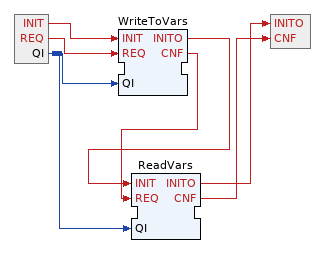
        [picture p71: application OpcUaBothWorking.WorkingWithoutSubscription.folderTestRemote_1]
        SUBAPPLICATION WriteToVars
          EVENT_INPUT
            INIT;
            REQ;
          END_EVENT
          EVENT_OUTPUT
            INITO;
            CNF;
          END_EVENT
          VAR_INPUT
            QI : BOOL;
          END_VAR
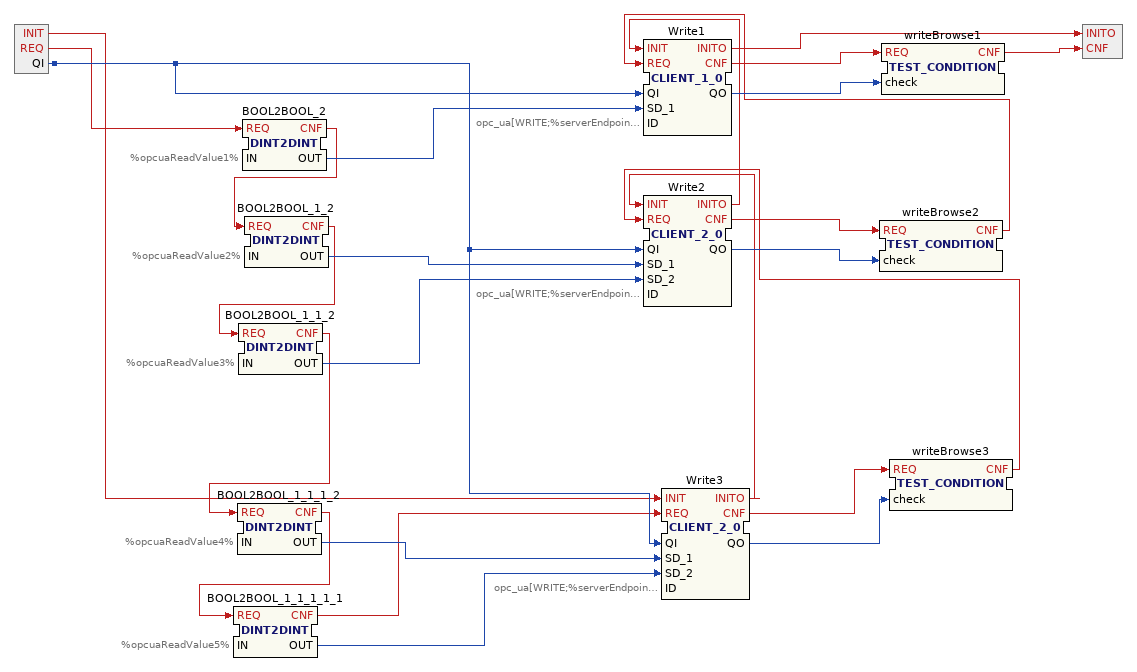
          FBS
            BOOL2BOOL_1_1_2 : DINT2DINT(IN := %opcuaReadValue3%);
            BOOL2BOOL_1_1_1_1_1 : DINT2DINT(IN := %opcuaReadValue5%);
            BOOL2BOOL_1_1_1_2 : DINT2DINT(IN := %opcuaReadValue4%);
            BOOL2BOOL_2 : DINT2DINT(IN := %opcuaReadValue1%);
            BOOL2BOOL_1_2 : DINT2DINT(IN := %opcuaReadValue2%);
            Write1 : CLIENT_1_0(ID := opc_ua[WRITE;%serverEndpoint%;%opcuaFolderTestOnlyBroseName1%]);
            Write3 : CLIENT_2_0(ID := opc_ua[WRITE;%serverEndpoint%;%opcuaFolderTestOnlyBroseName3%]);
            Write2 : CLIENT_2_0(ID := opc_ua[WRITE;%serverEndpoint%;%opcuaFolderTestOnlyBroseName2%]);
            writeBrowse1 : TEST_CONDITION;
            writeBrowse2 : TEST_CONDITION;
            writeBrowse3 : TEST_CONDITION;
          END_FBS
          EVENT_CONNECTIONS
            BOOL2BOOL_1_2.CNF TO BOOL2BOOL_1_1_2.REQ;
            BOOL2BOOL_1_1_2.CNF TO BOOL2BOOL_1_1_1_2.REQ;
            BOOL2BOOL_1_1_1_2.CNF TO BOOL2BOOL_1_1_1_1_1.REQ;
            BOOL2BOOL_2.CNF TO BOOL2BOOL_1_2.REQ;
            REQ TO BOOL2BOOL_2.REQ;
            Write1.INITO TO INITO;
            INIT TO Write3.INIT;
            BOOL2BOOL_1_1_1_1_1.CNF TO Write3.REQ;
            Write3.INITO TO Write2.INIT;
            Write2.INITO TO Write1.INIT;
            writeBrowse3.CNF TO Write2.REQ;
            Write3.CNF TO writeBrowse3.REQ;
            writeBrowse2.CNF TO Write1.REQ;
            Write2.CNF TO writeBrowse2.REQ;
            writeBrowse1.CNF TO CNF;
            Write1.CNF TO writeBrowse1.REQ;
          END_CONNECTIONS
          DATA_CONNECTIONS
            QI TO Write1.QI;
            BOOL2BOOL_2.OUT TO Write1.SD_1;
            QI TO Write3.QI;
            BOOL2BOOL_1_1_1_2.OUT TO Write3.SD_1;
            BOOL2BOOL_1_1_1_1_1.OUT TO Write3.SD_2;
            QI TO Write2.QI;
            BOOL2BOOL_1_2.OUT TO Write2.SD_1;
            BOOL2BOOL_1_1_2.OUT TO Write2.SD_2;
            Write1.QO TO writeBrowse1.check;
            Write2.QO TO writeBrowse2.check;
            Write3.QO TO writeBrowse3.check;
          END_CONNECTIONS
        END_SUBAPPLICATION
        SUBAPPLICATION ReadVars
          EVENT_INPUT
            INIT;
            REQ;
          END_EVENT
          EVENT_OUTPUT
            INITO;
            CNF;
          END_EVENT
          VAR_INPUT
            QI : BOOL;
          END_VAR
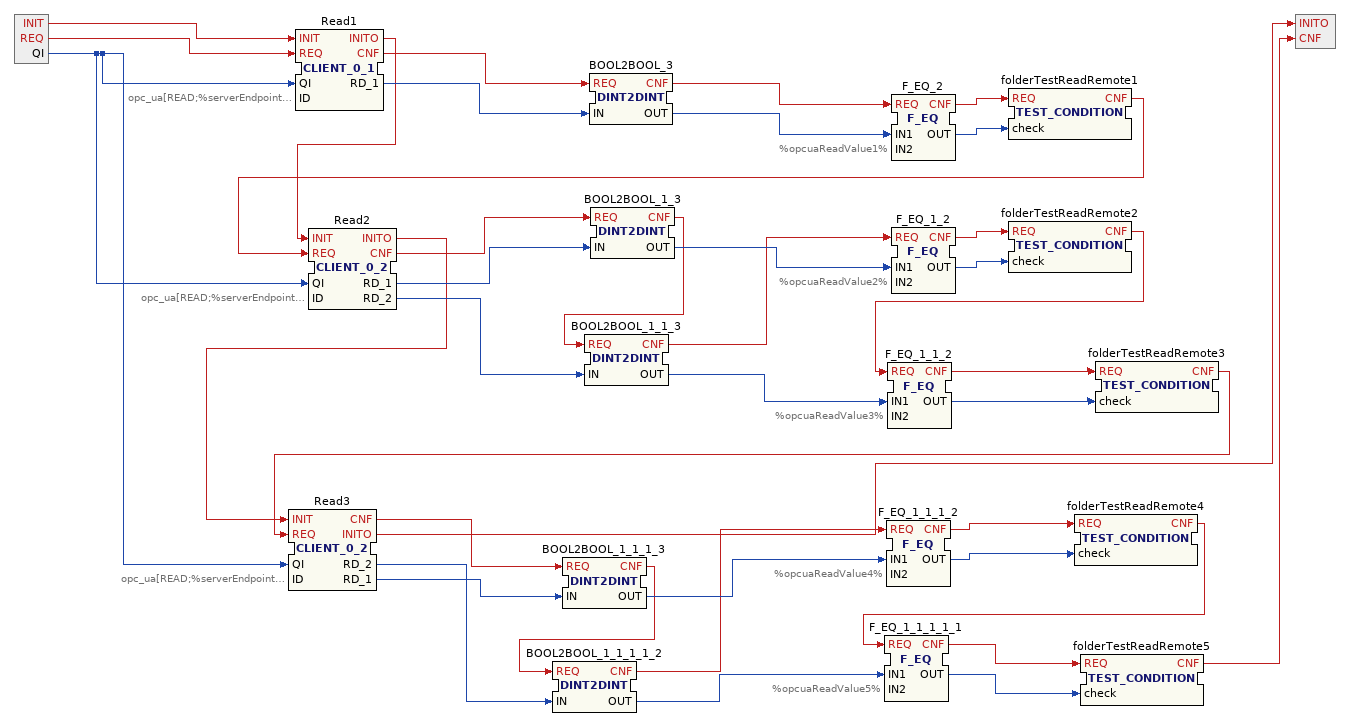
          FBS
            Read1 : CLIENT_0_1(ID := opc_ua[READ;%serverEndpoint%;%opcuaFolderTestOnlyBroseName1%]);
            Read2 : CLIENT_0_2(ID := opc_ua[READ;%serverEndpoint%;%opcuaFolderTestOnlyBroseName2%]);
            F_EQ_1_1_1_2 : F_EQ(IN2 := %opcuaReadValue4%);
            folderTestReadRemote4 : TEST_CONDITION;
            BOOL2BOOL_1_3 : DINT2DINT;
            F_EQ_1_1_1_1_1 : F_EQ(IN2 := %opcuaReadValue5%);
            folderTestReadRemote3 : TEST_CONDITION;
            BOOL2BOOL_1_1_3 : DINT2DINT;
            BOOL2BOOL_1_1_1_1_2 : DINT2DINT;
            BOOL2BOOL_1_1_1_3 : DINT2DINT;
            folderTestReadRemote2 : TEST_CONDITION;
            F_EQ_1_1_2 : F_EQ(IN2 := %opcuaReadValue3%);
            F_EQ_2 : F_EQ(IN2 := %opcuaReadValue1%);
            F_EQ_1_2 : F_EQ(IN2 := %opcuaReadValue2%);
            Read3 : CLIENT_0_2(ID := opc_ua[READ;%serverEndpoint%;%opcuaFolderTestOnlyBroseName3%]);
            folderTestReadRemote5 : TEST_CONDITION;
            folderTestReadRemote1 : TEST_CONDITION;
            BOOL2BOOL_3 : DINT2DINT;
          END_FBS
          EVENT_CONNECTIONS
            Read1.INITO TO Read2.INIT;
            Read1.CNF TO BOOL2BOOL_3.REQ;
            folderTestReadRemote1.CNF TO Read2.REQ;
            Read2.INITO TO Read3.INIT;
            Read2.CNF TO BOOL2BOOL_1_3.REQ;
            BOOL2BOOL_1_1_1_1_2.CNF TO F_EQ_1_1_1_2.REQ;
            F_EQ_1_1_1_2.CNF TO folderTestReadRemote4.REQ;
            folderTestReadRemote4.CNF TO F_EQ_1_1_1_1_1.REQ;
            BOOL2BOOL_1_3.CNF TO BOOL2BOOL_1_1_3.REQ;
            F_EQ_1_1_1_1_1.CNF TO folderTestReadRemote5.REQ;
            F_EQ_1_1_2.CNF TO folderTestReadRemote3.REQ;
            folderTestReadRemote3.CNF TO Read3.REQ;
            BOOL2BOOL_1_1_3.CNF TO F_EQ_1_2.REQ;
            BOOL2BOOL_1_1_1_3.CNF TO BOOL2BOOL_1_1_1_1_2.REQ;
            Read3.CNF TO BOOL2BOOL_1_1_1_3.REQ;
            F_EQ_1_2.CNF TO folderTestReadRemote2.REQ;
            folderTestReadRemote2.CNF TO F_EQ_1_1_2.REQ;
            BOOL2BOOL_3.CNF TO F_EQ_2.REQ;
            F_EQ_2.CNF TO folderTestReadRemote1.REQ;
            INIT TO Read1.INIT;
            REQ TO Read1.REQ;
            Read3.INITO TO INITO;
            folderTestReadRemote5.CNF TO CNF;
          END_CONNECTIONS
          DATA_CONNECTIONS
            Read1.RD_1 TO BOOL2BOOL_3.IN;
            Read2.RD_1 TO BOOL2BOOL_1_3.IN;
            Read2.RD_2 TO BOOL2BOOL_1_1_3.IN;
            BOOL2BOOL_1_1_1_3.OUT TO F_EQ_1_1_1_2.IN1;
            F_EQ_1_1_1_2.OUT TO folderTestReadRemote4.check;
            BOOL2BOOL_1_3.OUT TO F_EQ_1_2.IN1;
            BOOL2BOOL_1_1_1_1_2.OUT TO F_EQ_1_1_1_1_1.IN1;
            F_EQ_1_1_1_1_1.OUT TO folderTestReadRemote5.check;
            F_EQ_1_1_2.OUT TO folderTestReadRemote3.check;
            BOOL2BOOL_1_1_3.OUT TO F_EQ_1_1_2.IN1;
            Read3.RD_2 TO BOOL2BOOL_1_1_1_1_2.IN;
            Read3.RD_1 TO BOOL2BOOL_1_1_1_3.IN;
            F_EQ_1_2.OUT TO folderTestReadRemote2.check;
            BOOL2BOOL_3.OUT TO F_EQ_2.IN1;
            F_EQ_2.OUT TO folderTestReadRemote1.check;
            QI TO Read1.QI;
            QI TO Read2.QI;
            QI TO Read3.QI;
          END_CONNECTIONS
        END_SUBAPPLICATION
        EVENT_CONNECTIONS
          WriteToVars.INITO TO ReadVars.INIT;
          INIT TO WriteToVars.INIT;
          REQ TO WriteToVars.REQ;
          ReadVars.CNF TO CNF;
          WriteToVars.CNF TO ReadVars.REQ;
          ReadVars.INITO TO INITO;
        END_CONNECTIONS
        DATA_CONNECTIONS
          QI TO ReadVars.QI;
          QI TO WriteToVars.QI;
        END_CONNECTIONS
      END_SUBAPPLICATION
      SUBAPPLICATION bytestringNodeIdTestRemote_1
        EVENT_INPUT
          INIT;
          REQ;
        END_EVENT
        EVENT_OUTPUT
          INITO;
          CNF;
        END_EVENT
        VAR_INPUT
          QI : BOOL;
        END_VAR
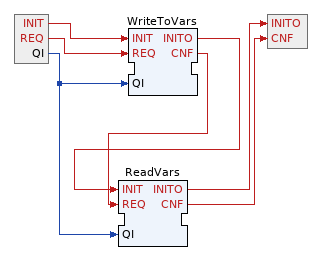
        SUBAPPLICATION WriteToVars
          EVENT_INPUT
            INIT;
            REQ;
          END_EVENT
          EVENT_OUTPUT
            INITO;
            CNF;
          END_EVENT
          VAR_INPUT
            QI : BOOL;
          END_VAR
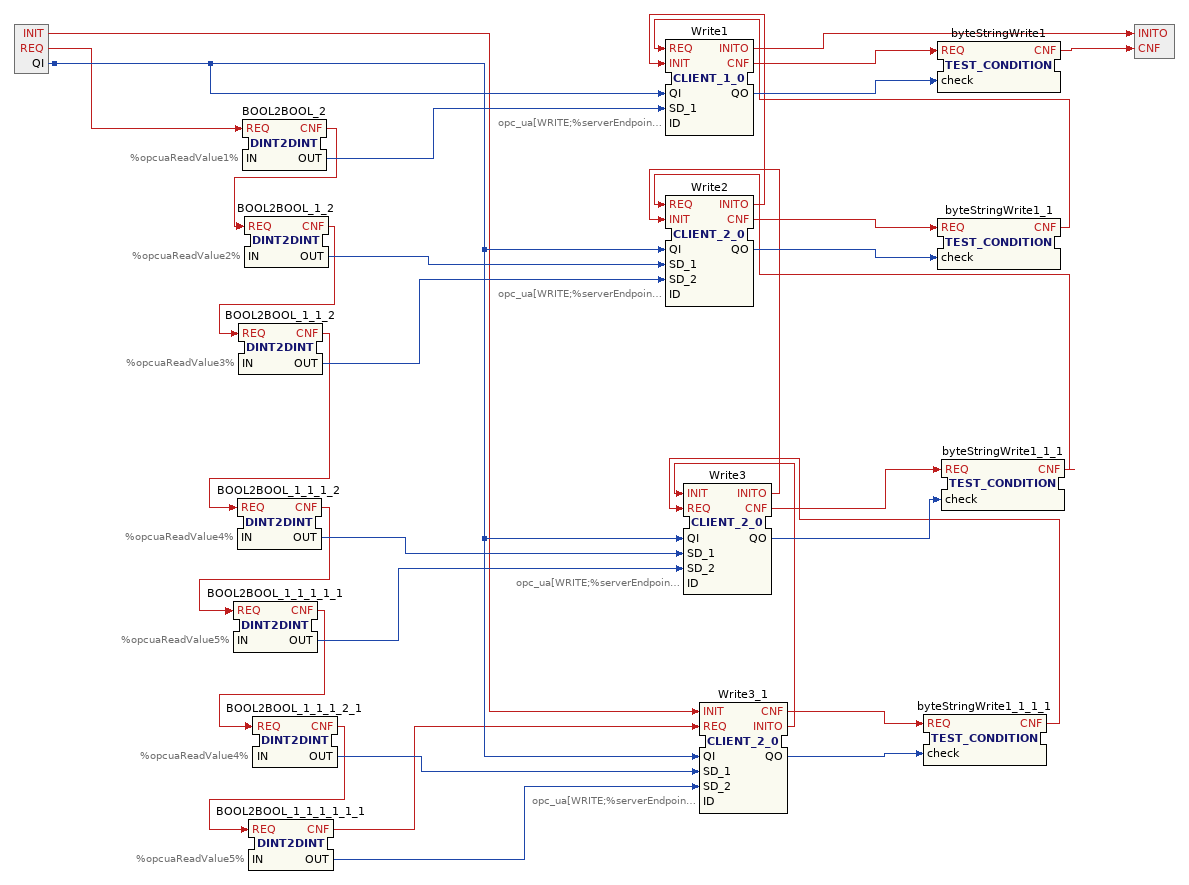
          FBS
            BOOL2BOOL_1_1_2 : DINT2DINT(IN := %opcuaReadValue3%);
            BOOL2BOOL_1_1_1_1_1 : DINT2DINT(IN := %opcuaReadValue5%);
            BOOL2BOOL_1_1_1_2 : DINT2DINT(IN := %opcuaReadValue4%);
            BOOL2BOOL_2 : DINT2DINT(IN := %opcuaReadValue1%);
            BOOL2BOOL_1_2 : DINT2DINT(IN := %opcuaReadValue2%);
            BOOL2BOOL_1_1_1_1_1_1 : DINT2DINT(IN := %opcuaReadValue5%);
            BOOL2BOOL_1_1_1_2_1 : DINT2DINT(IN := %opcuaReadValue4%);
            byteStringWrite1 : TEST_CONDITION;
            byteStringWrite1_1 : TEST_CONDITION;
            byteStringWrite1_1_1 : TEST_CONDITION;
            byteStringWrite1_1_1_1 : TEST_CONDITION;
            Write1 : CLIENT_1_0(ID := opc_ua[WRITE;%serverEndpoint%;%opcuaFolderTestWithNodeIdByteString1%]);
            Write2 : CLIENT_2_0(ID := opc_ua[WRITE;%serverEndpoint%;%opcuaFolderTestWithNodeIdByteString2%]);
            Write3_1 : CLIENT_2_0(ID := opc_ua[WRITE;%serverEndpoint%;,1:b=byteStringNodeId3;,1:b=byteStringNodeId4]);
            Write3 : CLIENT_2_0(ID := opc_ua[WRITE;%serverEndpoint%;%opcuaFolderTestWithNodeIdByteString3%]);
          END_FBS
          EVENT_CONNECTIONS
            BOOL2BOOL_1_2.CNF TO BOOL2BOOL_1_1_2.REQ;
            BOOL2BOOL_1_1_2.CNF TO BOOL2BOOL_1_1_1_2.REQ;
            BOOL2BOOL_1_1_1_2.CNF TO BOOL2BOOL_1_1_1_1_1.REQ;
            BOOL2BOOL_2.CNF TO BOOL2BOOL_1_2.REQ;
            REQ TO BOOL2BOOL_2.REQ;
            BOOL2BOOL_1_1_1_2_1.CNF TO BOOL2BOOL_1_1_1_1_1_1.REQ;
            BOOL2BOOL_1_1_1_1_1.CNF TO BOOL2BOOL_1_1_1_2_1.REQ;
            byteStringWrite1.CNF TO CNF;
            byteStringWrite1_1.CNF TO Write1.REQ;
            Write1.INITO TO INITO;
            Write1.CNF TO byteStringWrite1.REQ;
            byteStringWrite1_1_1.CNF TO Write2.REQ;
            Write2.INITO TO Write1.INIT;
            Write2.CNF TO byteStringWrite1_1.REQ;
            INIT TO Write3_1.INIT;
            BOOL2BOOL_1_1_1_1_1_1.CNF TO Write3_1.REQ;
            Write3_1.CNF TO byteStringWrite1_1_1_1.REQ;
            Write3_1.INITO TO Write3.INIT;
            byteStringWrite1_1_1_1.CNF TO Write3.REQ;
            Write3.INITO TO Write2.INIT;
            Write3.CNF TO byteStringWrite1_1_1.REQ;
          END_CONNECTIONS
          DATA_CONNECTIONS
            QI TO Write1.QI;
            BOOL2BOOL_2.OUT TO Write1.SD_1;
            Write1.QO TO byteStringWrite1.check;
            QI TO Write2.QI;
            BOOL2BOOL_1_2.OUT TO Write2.SD_1;
            BOOL2BOOL_1_1_2.OUT TO Write2.SD_2;
            Write2.QO TO byteStringWrite1_1.check;
            QI TO Write3_1.QI;
            BOOL2BOOL_1_1_1_2_1.OUT TO Write3_1.SD_1;
            BOOL2BOOL_1_1_1_1_1_1.OUT TO Write3_1.SD_2;
            Write3_1.QO TO byteStringWrite1_1_1_1.check;
            QI TO Write3.QI;
            BOOL2BOOL_1_1_1_2.OUT TO Write3.SD_1;
            BOOL2BOOL_1_1_1_1_1.OUT TO Write3.SD_2;
            Write3.QO TO byteStringWrite1_1_1.check;
          END_CONNECTIONS
        END_SUBAPPLICATION
        SUBAPPLICATION ReadVars
          EVENT_INPUT
            INIT;
            REQ;
          END_EVENT
          EVENT_OUTPUT
            INITO;
            CNF;
          END_EVENT
          VAR_INPUT
            QI : BOOL;
          END_VAR
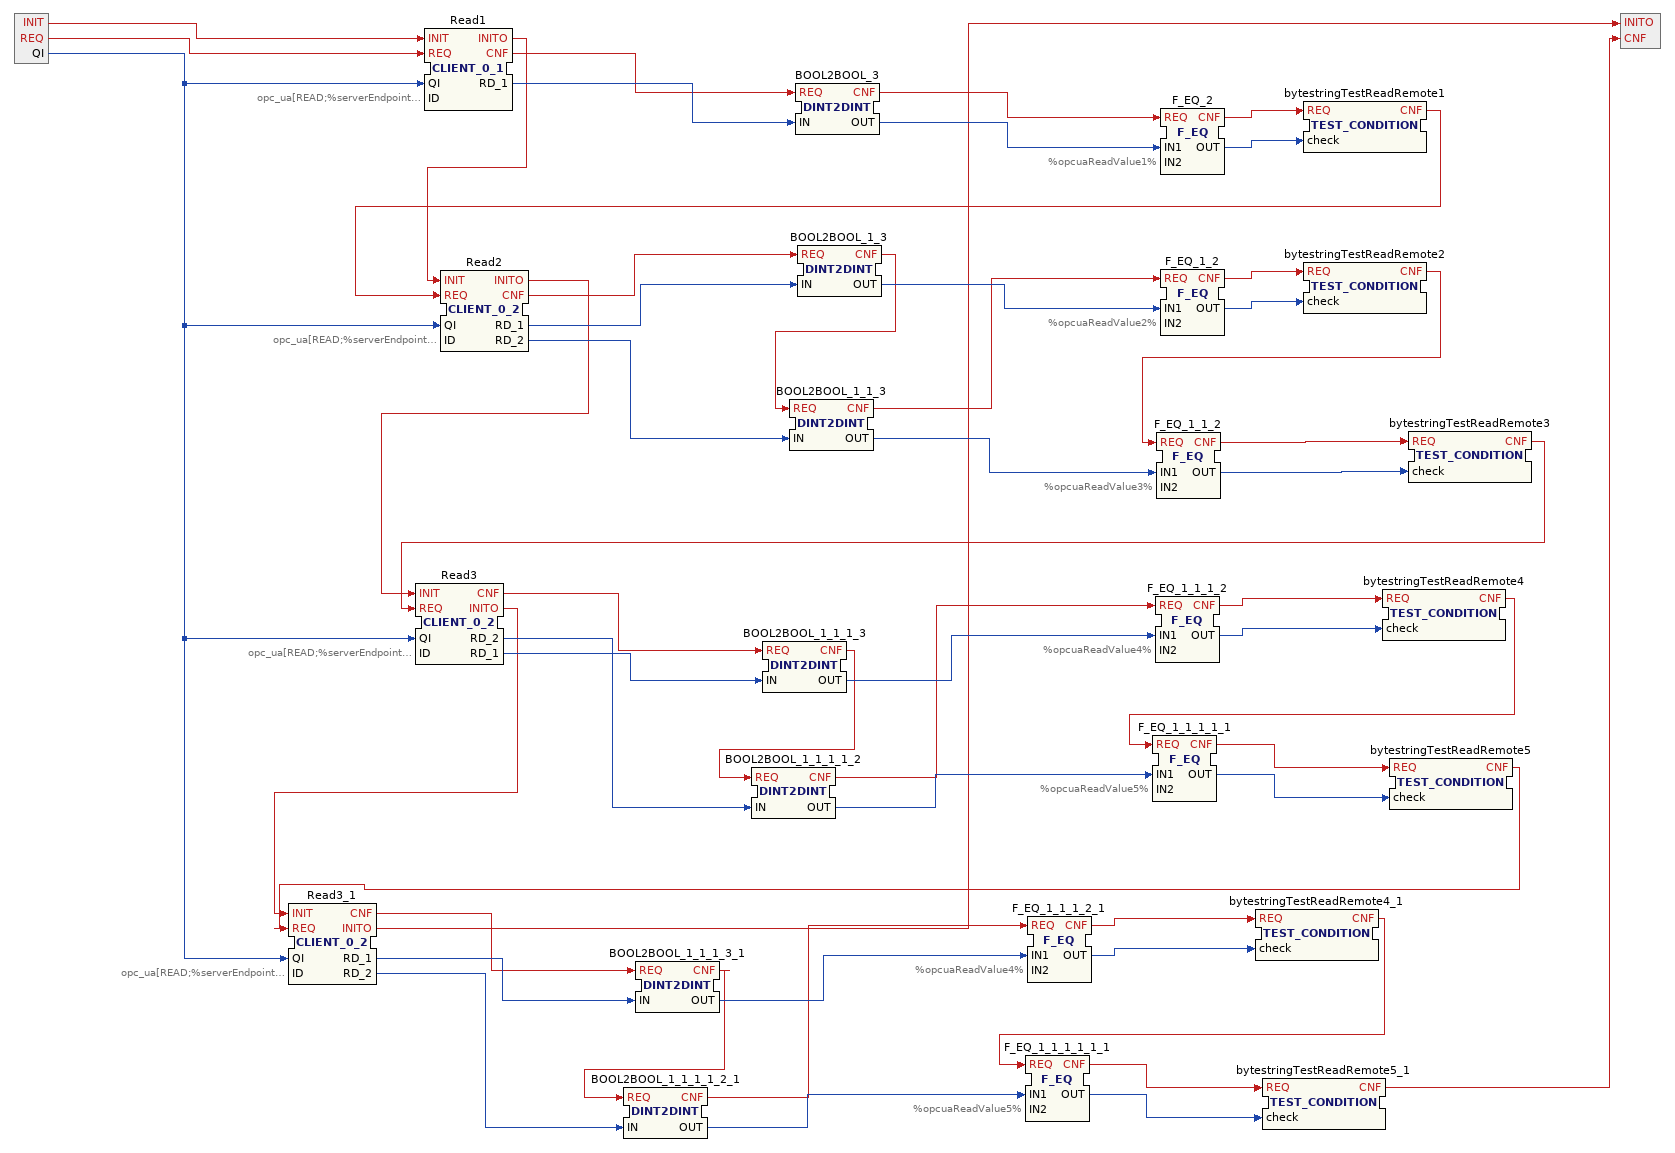
          FBS
            Read1 : CLIENT_0_1(ID := opc_ua[READ;%serverEndpoint%;%opcuaFolderTestWithNodeIdByteString1%]);
            Read2 : CLIENT_0_2(ID := opc_ua[READ;%serverEndpoint%;%opcuaFolderTestWithNodeIdByteString2%]);
            F_EQ_1_1_1_2 : F_EQ(IN2 := %opcuaReadValue4%);
            bytestringTestReadRemote4 : TEST_CONDITION;
            BOOL2BOOL_1_3 : DINT2DINT;
            F_EQ_1_1_1_1_1 : F_EQ(IN2 := %opcuaReadValue5%);
            bytestringTestReadRemote3 : TEST_CONDITION;
            BOOL2BOOL_1_1_3 : DINT2DINT;
            BOOL2BOOL_1_1_1_1_2 : DINT2DINT;
            BOOL2BOOL_1_1_1_3 : DINT2DINT;
            bytestringTestReadRemote2 : TEST_CONDITION;
            F_EQ_1_1_2 : F_EQ(IN2 := %opcuaReadValue3%);
            F_EQ_2 : F_EQ(IN2 := %opcuaReadValue1%);
            F_EQ_1_2 : F_EQ(IN2 := %opcuaReadValue2%);
            Read3 : CLIENT_0_2(ID := opc_ua[READ;%serverEndpoint%;%opcuaFolderTestWithNodeIdByteString3%]);
            bytestringTestReadRemote5 : TEST_CONDITION;
            bytestringTestReadRemote1 : TEST_CONDITION;
            BOOL2BOOL_3 : DINT2DINT;
            BOOL2BOOL_1_1_1_3_1 : DINT2DINT;
            Read3_1 : CLIENT_0_2(ID := opc_ua[READ;%serverEndpoint%;,1:b=byteStringNodeId3;,1:b=byteStringNodeId4]);
            bytestringTestReadRemote4_1 : TEST_CONDITION;
            F_EQ_1_1_1_2_1 : F_EQ(IN2 := %opcuaReadValue4%);
            BOOL2BOOL_1_1_1_1_2_1 : DINT2DINT;
            bytestringTestReadRemote5_1 : TEST_CONDITION;
            F_EQ_1_1_1_1_1_1 : F_EQ(IN2 := %opcuaReadValue5%);
          END_FBS
          EVENT_CONNECTIONS
            Read1.INITO TO Read2.INIT;
            Read1.CNF TO BOOL2BOOL_3.REQ;
            bytestringTestReadRemote1.CNF TO Read2.REQ;
            Read2.INITO TO Read3.INIT;
            Read2.CNF TO BOOL2BOOL_1_3.REQ;
            BOOL2BOOL_1_1_1_1_2.CNF TO F_EQ_1_1_1_2.REQ;
            F_EQ_1_1_1_2.CNF TO bytestringTestReadRemote4.REQ;
            bytestringTestReadRemote4.CNF TO F_EQ_1_1_1_1_1.REQ;
            BOOL2BOOL_1_3.CNF TO BOOL2BOOL_1_1_3.REQ;
            F_EQ_1_1_1_1_1.CNF TO bytestringTestReadRemote5.REQ;
            F_EQ_1_1_2.CNF TO bytestringTestReadRemote3.REQ;
            bytestringTestReadRemote3.CNF TO Read3.REQ;
            BOOL2BOOL_1_1_3.CNF TO F_EQ_1_2.REQ;
            BOOL2BOOL_1_1_1_3.CNF TO BOOL2BOOL_1_1_1_1_2.REQ;
            Read3.CNF TO BOOL2BOOL_1_1_1_3.REQ;
            F_EQ_1_2.CNF TO bytestringTestReadRemote2.REQ;
            bytestringTestReadRemote2.CNF TO F_EQ_1_1_2.REQ;
            BOOL2BOOL_3.CNF TO F_EQ_2.REQ;
            F_EQ_2.CNF TO bytestringTestReadRemote1.REQ;
            INIT TO Read1.INIT;
            REQ TO Read1.REQ;
            bytestringTestReadRemote4_1.CNF TO F_EQ_1_1_1_1_1_1.REQ;
            BOOL2BOOL_1_1_1_1_2_1.CNF TO F_EQ_1_1_1_2_1.REQ;
            F_EQ_1_1_1_1_1_1.CNF TO bytestringTestReadRemote5_1.REQ;
            F_EQ_1_1_1_2_1.CNF TO bytestringTestReadRemote4_1.REQ;
            BOOL2BOOL_1_1_1_3_1.CNF TO BOOL2BOOL_1_1_1_1_2_1.REQ;
            Read3_1.CNF TO BOOL2BOOL_1_1_1_3_1.REQ;
            Read3_1.INITO TO INITO;
            Read3.INITO TO Read3_1.INIT;
            bytestringTestReadRemote5_1.CNF TO CNF;
            bytestringTestReadRemote5.CNF TO Read3_1.REQ;
          END_CONNECTIONS
          DATA_CONNECTIONS
            Read1.RD_1 TO BOOL2BOOL_3.IN;
            Read2.RD_1 TO BOOL2BOOL_1_3.IN;
            Read2.RD_2 TO BOOL2BOOL_1_1_3.IN;
            BOOL2BOOL_1_1_1_3.OUT TO F_EQ_1_1_1_2.IN1;
            F_EQ_1_1_1_2.OUT TO bytestringTestReadRemote4.check;
            BOOL2BOOL_1_3.OUT TO F_EQ_1_2.IN1;
            BOOL2BOOL_1_1_1_1_2.OUT TO F_EQ_1_1_1_1_1.IN1;
            F_EQ_1_1_1_1_1.OUT TO bytestringTestReadRemote5.check;
            F_EQ_1_1_2.OUT TO bytestringTestReadRemote3.check;
            BOOL2BOOL_1_1_3.OUT TO F_EQ_1_1_2.IN1;
            Read3.RD_2 TO BOOL2BOOL_1_1_1_1_2.IN;
            Read3.RD_1 TO BOOL2BOOL_1_1_1_3.IN;
            F_EQ_1_2.OUT TO bytestringTestReadRemote2.check;
            BOOL2BOOL_3.OUT TO F_EQ_2.IN1;
            F_EQ_2.OUT TO bytestringTestReadRemote1.check;
            QI TO Read1.QI;
            QI TO Read2.QI;
            QI TO Read3.QI;
            BOOL2BOOL_1_1_1_1_2_1.OUT TO F_EQ_1_1_1_1_1_1.IN1;
            BOOL2BOOL_1_1_1_3_1.OUT TO F_EQ_1_1_1_2_1.IN1;
            F_EQ_1_1_1_2_1.OUT TO bytestringTestReadRemote4_1.check;
            Read3_1.RD_1 TO BOOL2BOOL_1_1_1_3_1.IN;
            F_EQ_1_1_1_1_1_1.OUT TO bytestringTestReadRemote5_1.check;
            Read3_1.RD_2 TO BOOL2BOOL_1_1_1_1_2_1.IN;
            QI TO Read3_1.QI;
          END_CONNECTIONS
        END_SUBAPPLICATION
        EVENT_CONNECTIONS
          WriteToVars.INITO TO ReadVars.INIT;
          INIT TO WriteToVars.INIT;
          REQ TO WriteToVars.REQ;
          ReadVars.CNF TO CNF;
          WriteToVars.CNF TO ReadVars.REQ;
          ReadVars.INITO TO INITO;
        END_CONNECTIONS
        DATA_CONNECTIONS
          QI TO ReadVars.QI;
          QI TO WriteToVars.QI;
        END_CONNECTIONS
      END_SUBAPPLICATION
      SUBAPPLICATION RemoteMethods_1
        EVENT_INPUT
          INIT;
          REQ;
        END_EVENT
        EVENT_OUTPUT
          INITO;
          CNF;
        END_EVENT
        VAR_INPUT
          QI : BOOL;
        END_VAR
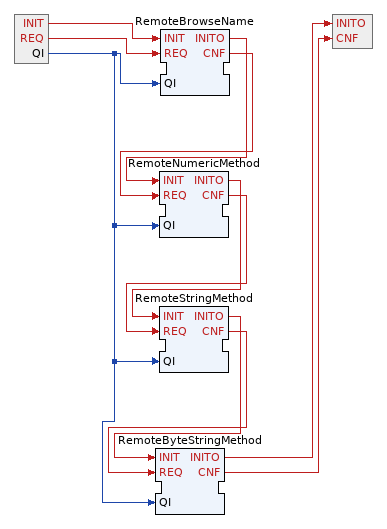
        SUBAPPLICATION RemoteBrowseName
          EVENT_INPUT
            INIT;
            REQ;
          END_EVENT
          EVENT_OUTPUT
            INITO;
            CNF;
          END_EVENT
          VAR_INPUT
            QI : BOOL;
          END_VAR
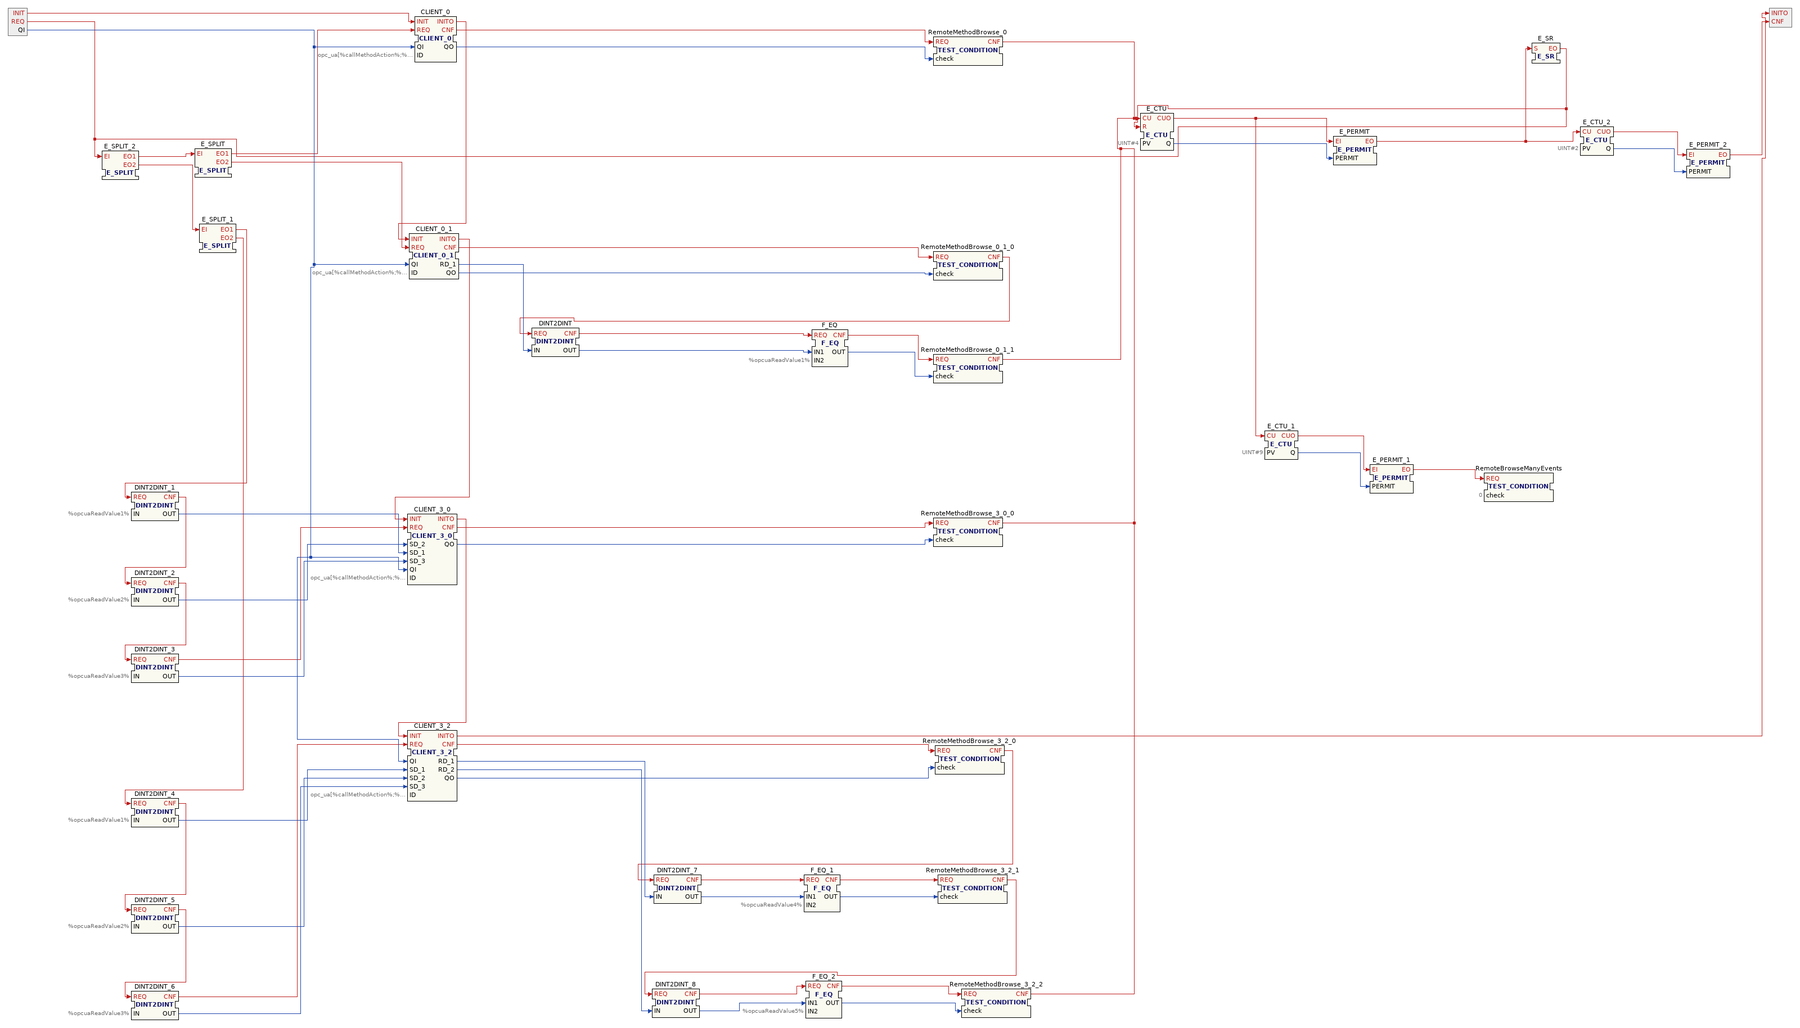
          FBS
            DINT2DINT_4 : DINT2DINT(IN := %opcuaReadValue1%);
            CLIENT_0 : CLIENT_0(ID := opc_ua[%callMethodAction%;%serverEndpoint%;%opcuaMethodCreation1%]);
            DINT2DINT_2 : DINT2DINT(IN := %opcuaReadValue2%);
            CLIENT_0_1 : CLIENT_0_1(ID := opc_ua[%callMethodAction%;%serverEndpoint%;%opcuaMethodCreation2%]);
            DINT2DINT : DINT2DINT;
            DINT2DINT_1 : DINT2DINT(IN := %opcuaReadValue1%);
            CLIENT_3_0 : CLIENT_3_0(ID := opc_ua[%callMethodAction%;%serverEndpoint%;%opcuaMethodCreation3%]);
            CLIENT_3_2 : CLIENT_3_2(ID := opc_ua[%callMethodAction%;%serverEndpoint%;%opcuaMethodCreation4%]);
            DINT2DINT_3 : DINT2DINT(IN := %opcuaReadValue3%);
            DINT2DINT_5 : DINT2DINT(IN := %opcuaReadValue2%);
            DINT2DINT_6 : DINT2DINT(IN := %opcuaReadValue3%);
            DINT2DINT_7 : DINT2DINT;
            DINT2DINT_8 : DINT2DINT;
            RemoteMethodBrowse_3_2_1 : TEST_CONDITION;
            RemoteMethodBrowse_3_2_2 : TEST_CONDITION;
            RemoteMethodBrowse_0 : TEST_CONDITION;
            RemoteMethodBrowse_0_1_0 : TEST_CONDITION;
            RemoteMethodBrowse_0_1_1 : TEST_CONDITION;
            RemoteMethodBrowse_3_2_0 : TEST_CONDITION;
            RemoteMethodBrowse_3_0_0 : TEST_CONDITION;
            F_EQ : F_EQ(IN2 := %opcuaReadValue1%);
            F_EQ_1 : F_EQ(IN2 := %opcuaReadValue4%);
            F_EQ_2 : F_EQ(IN2 := %opcuaReadValue5%);
            E_SPLIT : E_SPLIT;
            E_SPLIT_1 : E_SPLIT;
            E_CTU : E_CTU(PV := UINT#4);
            E_PERMIT : E_PERMIT;
            E_CTU_1 : E_CTU(PV := UINT#9);
            E_PERMIT_1 : E_PERMIT;
            RemoteBrowseManyEvents : TEST_CONDITION(check := 0);
            E_SPLIT_2 : E_SPLIT;
            E_PERMIT_2 : E_PERMIT;
            E_CTU_2 : E_CTU(PV := UINT#2);
            E_SR : E_SR;
          END_FBS
          EVENT_CONNECTIONS
            DINT2DINT_1.CNF TO DINT2DINT_2.REQ;
            DINT2DINT_2.CNF TO DINT2DINT_3.REQ;
            CLIENT_0_1.INITO TO CLIENT_3_0.INIT;
            INIT TO CLIENT_0.INIT;
            CLIENT_0.INITO TO CLIENT_0_1.INIT;
            CLIENT_3_0.INITO TO CLIENT_3_2.INIT;
            CLIENT_3_2.INITO TO INITO;
            CLIENT_0.CNF TO RemoteMethodBrowse_0.REQ;
            F_EQ.CNF TO RemoteMethodBrowse_0_1_1.REQ;
            CLIENT_3_0.CNF TO RemoteMethodBrowse_3_0_0.REQ;
            DINT2DINT_8.CNF TO F_EQ_2.REQ;
            DINT2DINT_7.CNF TO F_EQ_1.REQ;
            RemoteMethodBrowse_3_2_0.CNF TO DINT2DINT_7.REQ;
            F_EQ_1.CNF TO RemoteMethodBrowse_3_2_1.REQ;
            RemoteMethodBrowse_3_2_1.CNF TO DINT2DINT_8.REQ;
            F_EQ_2.CNF TO RemoteMethodBrowse_3_2_2.REQ;
            CLIENT_3_2.CNF TO RemoteMethodBrowse_3_2_0.REQ;
            DINT2DINT_4.CNF TO DINT2DINT_5.REQ;
            DINT2DINT_5.CNF TO DINT2DINT_6.REQ;
            DINT2DINT_6.CNF TO CLIENT_3_2.REQ;
            CLIENT_0_1.CNF TO RemoteMethodBrowse_0_1_0.REQ;
            RemoteMethodBrowse_0_1_0.CNF TO DINT2DINT.REQ;
            DINT2DINT.CNF TO F_EQ.REQ;
            DINT2DINT_3.CNF TO CLIENT_3_0.REQ;
            E_SPLIT.EO1 TO CLIENT_0.REQ;
            RemoteMethodBrowse_3_2_2.CNF TO E_CTU.CU;
            E_CTU.CUO TO E_CTU_1.CU;
            E_CTU.CUO TO E_PERMIT.EI;
            E_CTU_1.CUO TO E_PERMIT_1.EI;
            E_PERMIT_1.EO TO RemoteBrowseManyEvents.REQ;
            RemoteMethodBrowse_0.CNF TO E_CTU.CU;
            E_SPLIT.EO2 TO CLIENT_0_1.REQ;
            RemoteMethodBrowse_0_1_1.CNF TO E_CTU.CU;
            E_SPLIT_1.EO1 TO DINT2DINT_1.REQ;
            RemoteMethodBrowse_3_0_0.CNF TO E_CTU.CU;
            E_SPLIT_1.EO2 TO DINT2DINT_4.REQ;
            REQ TO E_SPLIT_2.EI;
            E_SPLIT_2.EO1 TO E_SPLIT.EI;
            E_SPLIT_2.EO2 TO E_SPLIT_1.EI;
            E_PERMIT.EO TO E_CTU_2.CU;
            E_CTU_2.CUO TO E_PERMIT_2.EI;
            E_PERMIT_2.EO TO CNF;
            E_PERMIT.EO TO E_SR.S;
            E_SR.EO TO E_CTU.R;
            E_SR.EO TO E_SPLIT_2.EI;
          END_CONNECTIONS
          DATA_CONNECTIONS
            DINT2DINT_2.OUT TO CLIENT_3_0.SD_2;
            CLIENT_0_1.RD_1 TO DINT2DINT.IN;
            DINT2DINT_1.OUT TO CLIENT_3_0.SD_1;
            DINT2DINT_3.OUT TO CLIENT_3_0.SD_3;
            QI TO CLIENT_0_1.QI;
            QI TO CLIENT_3_0.QI;
            QI TO CLIENT_3_2.QI;
            QI TO CLIENT_0.QI;
            DINT2DINT_4.OUT TO CLIENT_3_2.SD_1;
            DINT2DINT_5.OUT TO CLIENT_3_2.SD_2;
            CLIENT_3_2.RD_1 TO DINT2DINT_7.IN;
            CLIENT_3_2.RD_2 TO DINT2DINT_8.IN;
            DINT2DINT_6.OUT TO CLIENT_3_2.SD_3;
            CLIENT_0.QO TO RemoteMethodBrowse_0.check;
            CLIENT_0_1.QO TO RemoteMethodBrowse_0_1_0.check;
            F_EQ.OUT TO RemoteMethodBrowse_0_1_1.check;
            DINT2DINT.OUT TO F_EQ.IN1;
            CLIENT_3_0.QO TO RemoteMethodBrowse_3_0_0.check;
            DINT2DINT_7.OUT TO F_EQ_1.IN1;
            DINT2DINT_8.OUT TO F_EQ_2.IN1;
            F_EQ_1.OUT TO RemoteMethodBrowse_3_2_1.check;
            F_EQ_2.OUT TO RemoteMethodBrowse_3_2_2.check;
            CLIENT_3_2.QO TO RemoteMethodBrowse_3_2_0.check;
            E_CTU.Q TO E_PERMIT.PERMIT;
            E_CTU_1.Q TO E_PERMIT_1.PERMIT;
            E_CTU_2.Q TO E_PERMIT_2.PERMIT;
          END_CONNECTIONS
        END_SUBAPPLICATION
        SUBAPPLICATION RemoteNumericMethod
          EVENT_INPUT
            INIT;
            REQ;
          END_EVENT
          EVENT_OUTPUT
            INITO;
            CNF;
          END_EVENT
          VAR_INPUT
            QI : BOOL;
          END_VAR
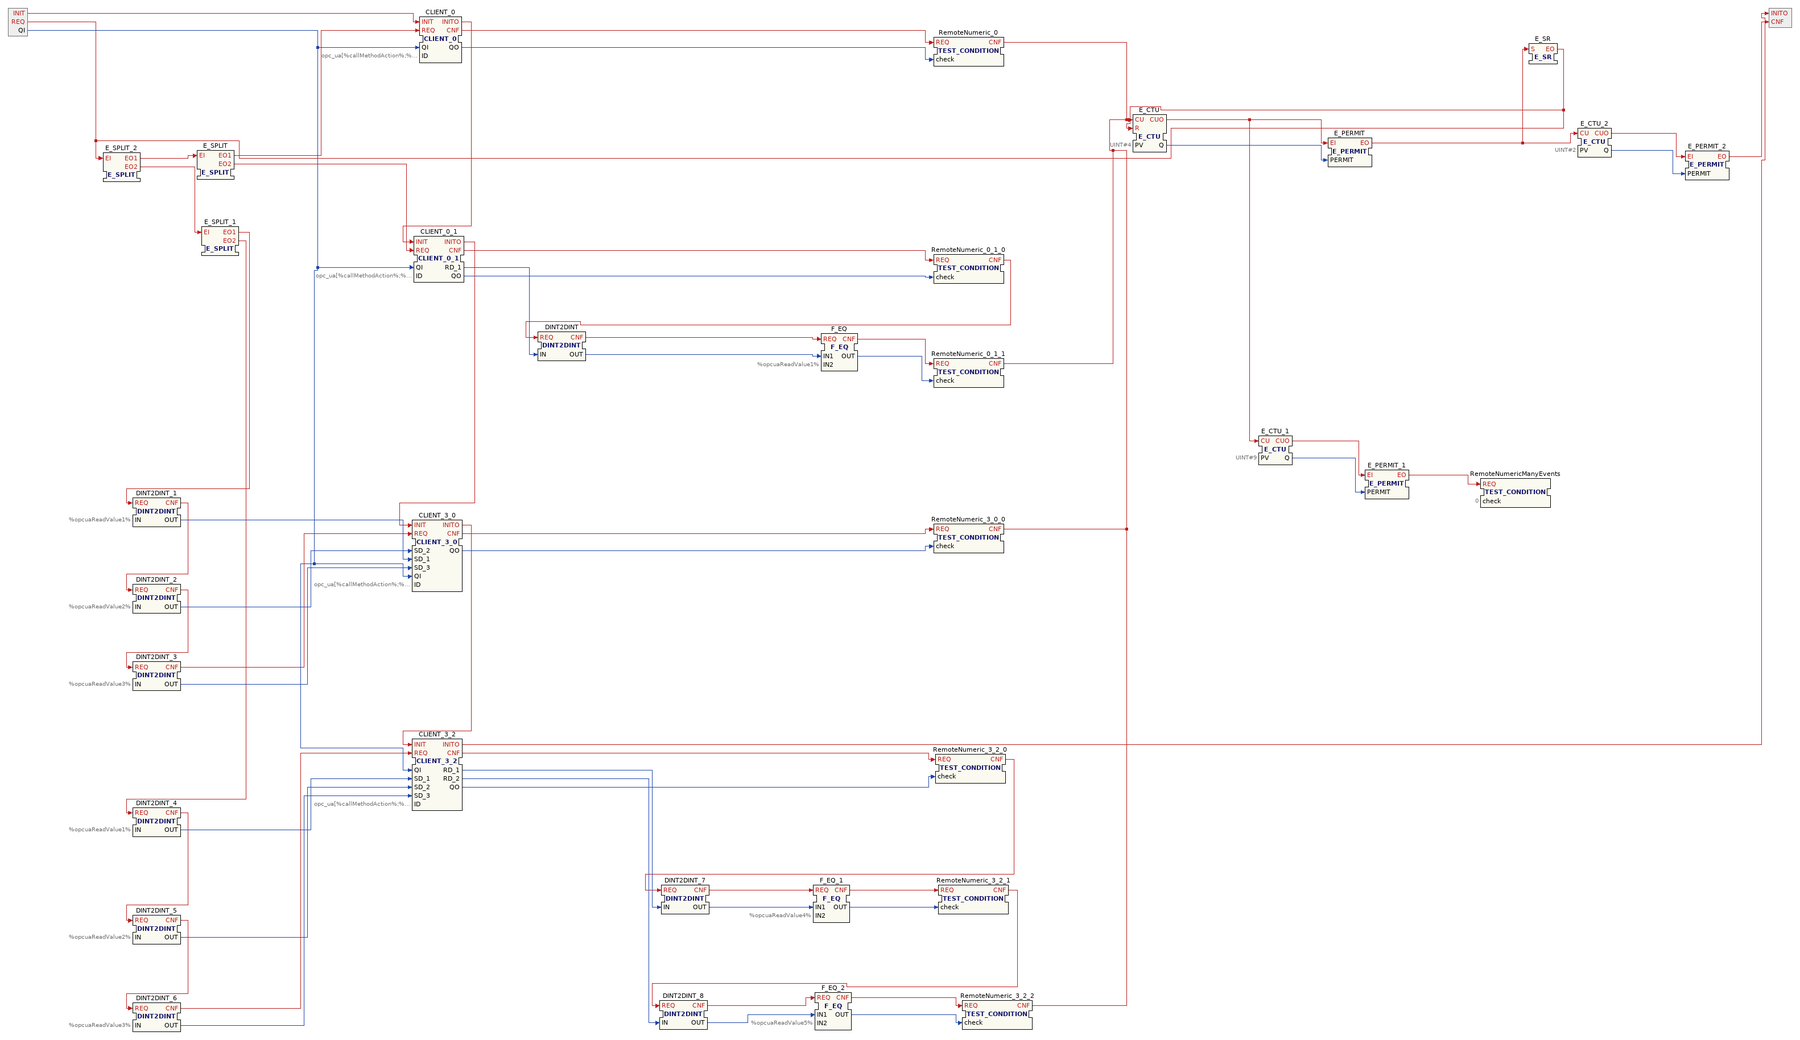
          FBS
            DINT2DINT_4 : DINT2DINT(IN := %opcuaReadValue1%);
            CLIENT_0 : CLIENT_0(ID := opc_ua[%callMethodAction%;%serverEndpoint%;%opcuaMethodCreation5%]);
            DINT2DINT_2 : DINT2DINT(IN := %opcuaReadValue2%);
            CLIENT_0_1 : CLIENT_0_1(ID := opc_ua[%callMethodAction%;%serverEndpoint%;%opcuaMethodCreation6%]);
            DINT2DINT : DINT2DINT;
            DINT2DINT_1 : DINT2DINT(IN := %opcuaReadValue1%);
            CLIENT_3_0 : CLIENT_3_0(ID := opc_ua[%callMethodAction%;%serverEndpoint%;%opcuaMethodCreation7%]);
            CLIENT_3_2 : CLIENT_3_2(ID := opc_ua[%callMethodAction%;%serverEndpoint%;%opcuaMethodCreation8%]);
            DINT2DINT_3 : DINT2DINT(IN := %opcuaReadValue3%);
            DINT2DINT_5 : DINT2DINT(IN := %opcuaReadValue2%);
            DINT2DINT_6 : DINT2DINT(IN := %opcuaReadValue3%);
            DINT2DINT_7 : DINT2DINT;
            DINT2DINT_8 : DINT2DINT;
            RemoteNumeric_3_2_1 : TEST_CONDITION;
            RemoteNumeric_3_2_2 : TEST_CONDITION;
            RemoteNumeric_0 : TEST_CONDITION;
            RemoteNumeric_0_1_0 : TEST_CONDITION;
            RemoteNumeric_0_1_1 : TEST_CONDITION;
            RemoteNumeric_3_2_0 : TEST_CONDITION;
            RemoteNumeric_3_0_0 : TEST_CONDITION;
            F_EQ : F_EQ(IN2 := %opcuaReadValue1%);
            F_EQ_1 : F_EQ(IN2 := %opcuaReadValue4%);
            F_EQ_2 : F_EQ(IN2 := %opcuaReadValue5%);
            E_SPLIT : E_SPLIT;
            E_SPLIT_1 : E_SPLIT;
            E_CTU : E_CTU(PV := UINT#4);
            E_PERMIT : E_PERMIT;
            E_CTU_1 : E_CTU(PV := UINT#9);
            E_PERMIT_1 : E_PERMIT;
            RemoteNumericManyEvents : TEST_CONDITION(check := 0);
            E_SPLIT_2 : E_SPLIT;
            E_PERMIT_2 : E_PERMIT;
            E_CTU_2 : E_CTU(PV := UINT#2);
            E_SR : E_SR;
          END_FBS
          EVENT_CONNECTIONS
            DINT2DINT_1.CNF TO DINT2DINT_2.REQ;
            DINT2DINT_2.CNF TO DINT2DINT_3.REQ;
            CLIENT_0_1.INITO TO CLIENT_3_0.INIT;
            INIT TO CLIENT_0.INIT;
            CLIENT_0.INITO TO CLIENT_0_1.INIT;
            CLIENT_3_0.INITO TO CLIENT_3_2.INIT;
            CLIENT_3_2.INITO TO INITO;
            CLIENT_0.CNF TO RemoteNumeric_0.REQ;
            F_EQ.CNF TO RemoteNumeric_0_1_1.REQ;
            CLIENT_3_0.CNF TO RemoteNumeric_3_0_0.REQ;
            DINT2DINT_8.CNF TO F_EQ_2.REQ;
            DINT2DINT_7.CNF TO F_EQ_1.REQ;
            RemoteNumeric_3_2_0.CNF TO DINT2DINT_7.REQ;
            F_EQ_1.CNF TO RemoteNumeric_3_2_1.REQ;
            RemoteNumeric_3_2_1.CNF TO DINT2DINT_8.REQ;
            F_EQ_2.CNF TO RemoteNumeric_3_2_2.REQ;
            CLIENT_3_2.CNF TO RemoteNumeric_3_2_0.REQ;
            DINT2DINT_4.CNF TO DINT2DINT_5.REQ;
            DINT2DINT_5.CNF TO DINT2DINT_6.REQ;
            DINT2DINT_6.CNF TO CLIENT_3_2.REQ;
            CLIENT_0_1.CNF TO RemoteNumeric_0_1_0.REQ;
            RemoteNumeric_0_1_0.CNF TO DINT2DINT.REQ;
            DINT2DINT.CNF TO F_EQ.REQ;
            DINT2DINT_3.CNF TO CLIENT_3_0.REQ;
            E_SPLIT.EO1 TO CLIENT_0.REQ;
            RemoteNumeric_3_2_2.CNF TO E_CTU.CU;
            E_CTU.CUO TO E_CTU_1.CU;
            E_CTU.CUO TO E_PERMIT.EI;
            E_CTU_1.CUO TO E_PERMIT_1.EI;
            E_PERMIT_1.EO TO RemoteNumericManyEvents.REQ;
            RemoteNumeric_0.CNF TO E_CTU.CU;
            E_SPLIT.EO2 TO CLIENT_0_1.REQ;
            RemoteNumeric_0_1_1.CNF TO E_CTU.CU;
            E_SPLIT_1.EO1 TO DINT2DINT_1.REQ;
            RemoteNumeric_3_0_0.CNF TO E_CTU.CU;
            E_SPLIT_1.EO2 TO DINT2DINT_4.REQ;
            REQ TO E_SPLIT_2.EI;
            E_SPLIT_2.EO1 TO E_SPLIT.EI;
            E_SPLIT_2.EO2 TO E_SPLIT_1.EI;
            E_PERMIT.EO TO E_CTU_2.CU;
            E_CTU_2.CUO TO E_PERMIT_2.EI;
            E_PERMIT_2.EO TO CNF;
            E_PERMIT.EO TO E_SR.S;
            E_SR.EO TO E_CTU.R;
            E_SR.EO TO E_SPLIT_2.EI;
          END_CONNECTIONS
          DATA_CONNECTIONS
            DINT2DINT_2.OUT TO CLIENT_3_0.SD_2;
            CLIENT_0_1.RD_1 TO DINT2DINT.IN;
            DINT2DINT_1.OUT TO CLIENT_3_0.SD_1;
            DINT2DINT_3.OUT TO CLIENT_3_0.SD_3;
            QI TO CLIENT_0_1.QI;
            QI TO CLIENT_3_0.QI;
            QI TO CLIENT_3_2.QI;
            QI TO CLIENT_0.QI;
            DINT2DINT_4.OUT TO CLIENT_3_2.SD_1;
            DINT2DINT_5.OUT TO CLIENT_3_2.SD_2;
            CLIENT_3_2.RD_1 TO DINT2DINT_7.IN;
            CLIENT_3_2.RD_2 TO DINT2DINT_8.IN;
            DINT2DINT_6.OUT TO CLIENT_3_2.SD_3;
            CLIENT_0.QO TO RemoteNumeric_0.check;
            CLIENT_0_1.QO TO RemoteNumeric_0_1_0.check;
            F_EQ.OUT TO RemoteNumeric_0_1_1.check;
            DINT2DINT.OUT TO F_EQ.IN1;
            CLIENT_3_0.QO TO RemoteNumeric_3_0_0.check;
            DINT2DINT_7.OUT TO F_EQ_1.IN1;
            DINT2DINT_8.OUT TO F_EQ_2.IN1;
            F_EQ_1.OUT TO RemoteNumeric_3_2_1.check;
            F_EQ_2.OUT TO RemoteNumeric_3_2_2.check;
            CLIENT_3_2.QO TO RemoteNumeric_3_2_0.check;
            E_CTU.Q TO E_PERMIT.PERMIT;
            E_CTU_1.Q TO E_PERMIT_1.PERMIT;
            E_CTU_2.Q TO E_PERMIT_2.PERMIT;
          END_CONNECTIONS
        END_SUBAPPLICATION
        SUBAPPLICATION RemoteStringMethod
          EVENT_INPUT
            INIT;
            REQ;
          END_EVENT
          EVENT_OUTPUT
            INITO;
            CNF;
          END_EVENT
          VAR_INPUT
            QI : BOOL;
          END_VAR
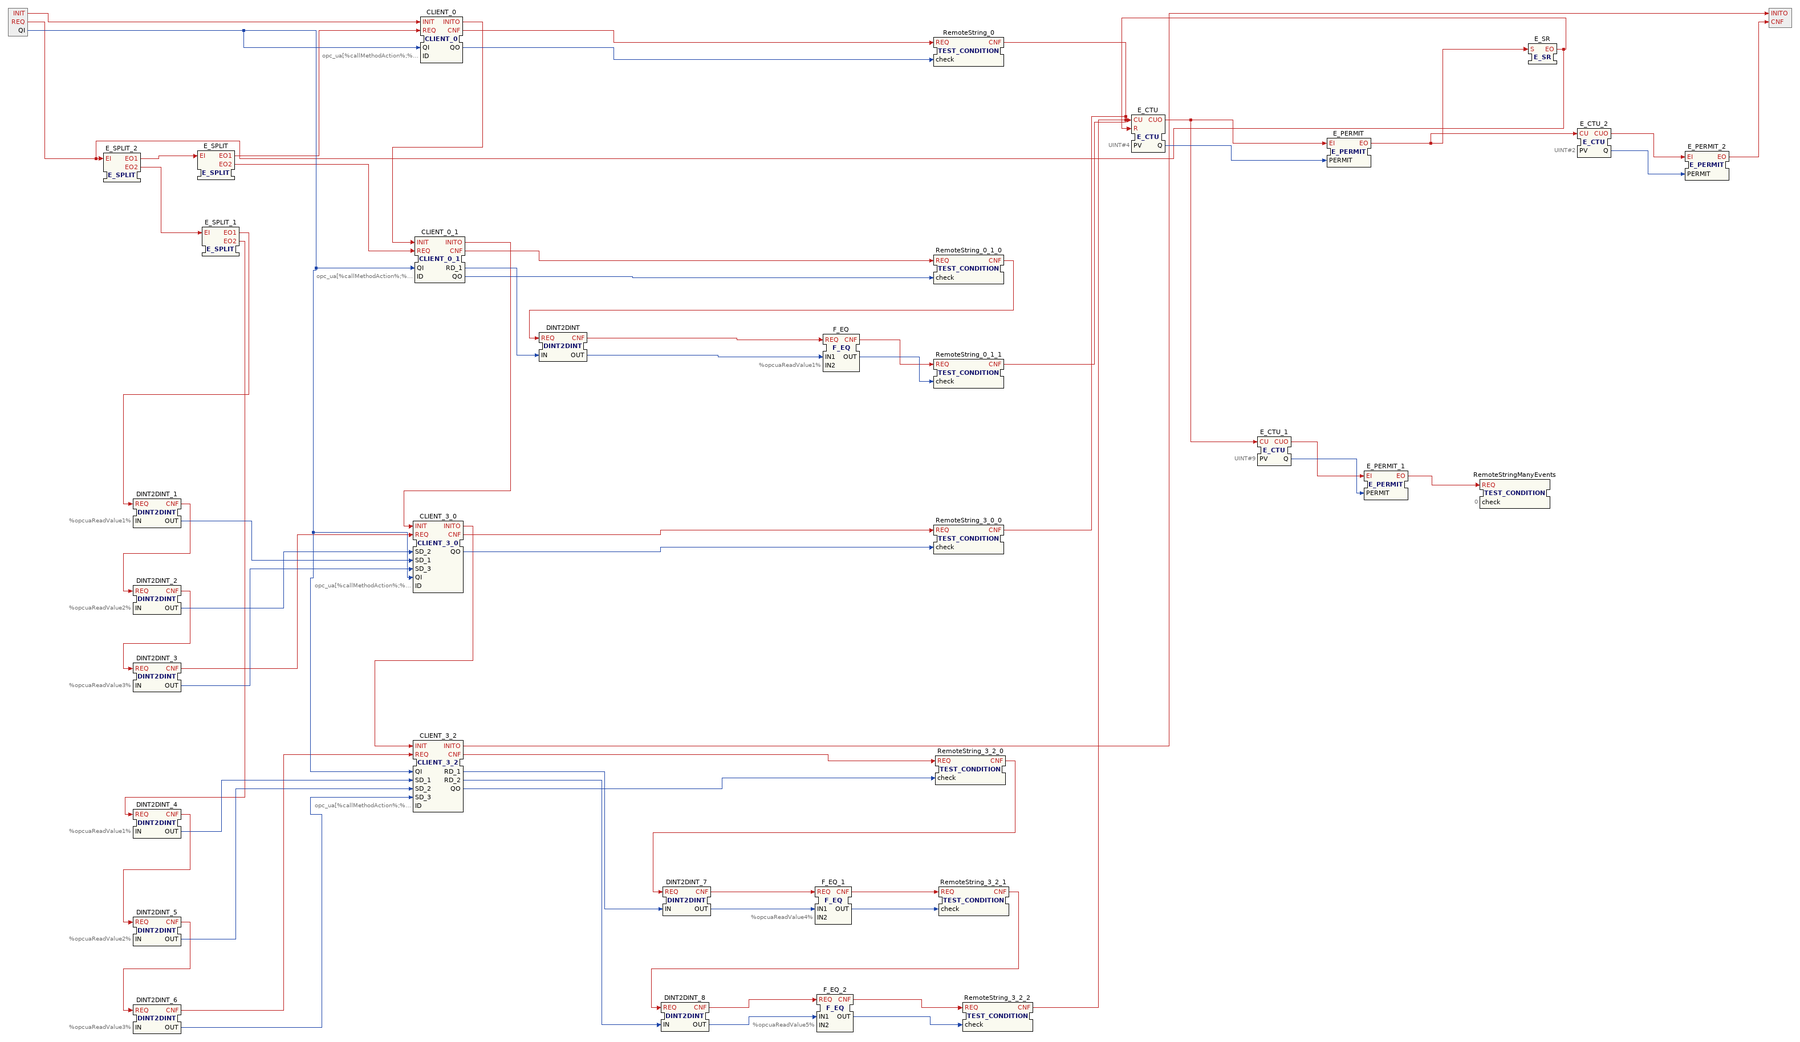
          FBS
            DINT2DINT_4 : DINT2DINT(IN := %opcuaReadValue1%);
            CLIENT_0 : CLIENT_0(ID := opc_ua[%callMethodAction%;%serverEndpoint%;%opcuaMethodCreation9%]);
            DINT2DINT_2 : DINT2DINT(IN := %opcuaReadValue2%);
            CLIENT_0_1 : CLIENT_0_1(ID := opc_ua[%callMethodAction%;%serverEndpoint%;%opcuaMethodCreation10%]);
            DINT2DINT : DINT2DINT;
            DINT2DINT_1 : DINT2DINT(IN := %opcuaReadValue1%);
            CLIENT_3_0 : CLIENT_3_0(ID := opc_ua[%callMethodAction%;%serverEndpoint%;%opcuaMethodCreation11%]);
            CLIENT_3_2 : CLIENT_3_2(ID := opc_ua[%callMethodAction%;%serverEndpoint%;%opcuaMethodCreation12%]);
            DINT2DINT_3 : DINT2DINT(IN := %opcuaReadValue3%);
            DINT2DINT_5 : DINT2DINT(IN := %opcuaReadValue2%);
            DINT2DINT_6 : DINT2DINT(IN := %opcuaReadValue3%);
            DINT2DINT_7 : DINT2DINT;
            DINT2DINT_8 : DINT2DINT;
            RemoteString_3_2_1 : TEST_CONDITION;
            RemoteString_3_2_2 : TEST_CONDITION;
            RemoteString_0 : TEST_CONDITION;
            RemoteString_0_1_0 : TEST_CONDITION;
            RemoteString_0_1_1 : TEST_CONDITION;
            RemoteString_3_2_0 : TEST_CONDITION;
            RemoteString_3_0_0 : TEST_CONDITION;
            F_EQ : F_EQ(IN2 := %opcuaReadValue1%);
            F_EQ_1 : F_EQ(IN2 := %opcuaReadValue4%);
            F_EQ_2 : F_EQ(IN2 := %opcuaReadValue5%);
            E_SPLIT : E_SPLIT;
            E_SPLIT_1 : E_SPLIT;
            E_CTU : E_CTU(PV := UINT#4);
            E_PERMIT : E_PERMIT;
            E_CTU_1 : E_CTU(PV := UINT#9);
            E_PERMIT_1 : E_PERMIT;
            RemoteStringManyEvents : TEST_CONDITION(check := 0);
            E_SPLIT_2 : E_SPLIT;
            E_PERMIT_2 : E_PERMIT;
            E_CTU_2 : E_CTU(PV := UINT#2);
            E_SR : E_SR;
          END_FBS
          EVENT_CONNECTIONS
            DINT2DINT_1.CNF TO DINT2DINT_2.REQ;
            DINT2DINT_2.CNF TO DINT2DINT_3.REQ;
            CLIENT_0_1.INITO TO CLIENT_3_0.INIT;
            INIT TO CLIENT_0.INIT;
            CLIENT_0.INITO TO CLIENT_0_1.INIT;
            CLIENT_3_0.INITO TO CLIENT_3_2.INIT;
            CLIENT_3_2.INITO TO INITO;
            CLIENT_0.CNF TO RemoteString_0.REQ;
            F_EQ.CNF TO RemoteString_0_1_1.REQ;
            CLIENT_3_0.CNF TO RemoteString_3_0_0.REQ;
            DINT2DINT_8.CNF TO F_EQ_2.REQ;
            DINT2DINT_7.CNF TO F_EQ_1.REQ;
            RemoteString_3_2_0.CNF TO DINT2DINT_7.REQ;
            F_EQ_1.CNF TO RemoteString_3_2_1.REQ;
            RemoteString_3_2_1.CNF TO DINT2DINT_8.REQ;
            F_EQ_2.CNF TO RemoteString_3_2_2.REQ;
            CLIENT_3_2.CNF TO RemoteString_3_2_0.REQ;
            DINT2DINT_4.CNF TO DINT2DINT_5.REQ;
            DINT2DINT_5.CNF TO DINT2DINT_6.REQ;
            DINT2DINT_6.CNF TO CLIENT_3_2.REQ;
            CLIENT_0_1.CNF TO RemoteString_0_1_0.REQ;
            RemoteString_0_1_0.CNF TO DINT2DINT.REQ;
            DINT2DINT.CNF TO F_EQ.REQ;
            DINT2DINT_3.CNF TO CLIENT_3_0.REQ;
            E_SPLIT.EO1 TO CLIENT_0.REQ;
            RemoteString_3_2_2.CNF TO E_CTU.CU;
            E_CTU.CUO TO E_CTU_1.CU;
            E_CTU.CUO TO E_PERMIT.EI;
            E_CTU_1.CUO TO E_PERMIT_1.EI;
            E_PERMIT_1.EO TO RemoteStringManyEvents.REQ;
            RemoteString_0.CNF TO E_CTU.CU;
            E_SPLIT.EO2 TO CLIENT_0_1.REQ;
            RemoteString_0_1_1.CNF TO E_CTU.CU;
            E_SPLIT_1.EO1 TO DINT2DINT_1.REQ;
            RemoteString_3_0_0.CNF TO E_CTU.CU;
            E_SPLIT_1.EO2 TO DINT2DINT_4.REQ;
            REQ TO E_SPLIT_2.EI;
            E_SPLIT_2.EO1 TO E_SPLIT.EI;
            E_SPLIT_2.EO2 TO E_SPLIT_1.EI;
            E_PERMIT.EO TO E_CTU_2.CU;
            E_CTU_2.CUO TO E_PERMIT_2.EI;
            E_PERMIT_2.EO TO CNF;
            E_PERMIT.EO TO E_SR.S;
            E_SR.EO TO E_CTU.R;
            E_SR.EO TO E_SPLIT_2.EI;
          END_CONNECTIONS
          DATA_CONNECTIONS
            DINT2DINT_2.OUT TO CLIENT_3_0.SD_2;
            CLIENT_0_1.RD_1 TO DINT2DINT.IN;
            DINT2DINT_1.OUT TO CLIENT_3_0.SD_1;
            DINT2DINT_3.OUT TO CLIENT_3_0.SD_3;
            QI TO CLIENT_0_1.QI;
            QI TO CLIENT_3_0.QI;
            QI TO CLIENT_3_2.QI;
            QI TO CLIENT_0.QI;
            DINT2DINT_4.OUT TO CLIENT_3_2.SD_1;
            DINT2DINT_5.OUT TO CLIENT_3_2.SD_2;
            CLIENT_3_2.RD_1 TO DINT2DINT_7.IN;
            CLIENT_3_2.RD_2 TO DINT2DINT_8.IN;
            DINT2DINT_6.OUT TO CLIENT_3_2.SD_3;
            CLIENT_0.QO TO RemoteString_0.check;
            CLIENT_0_1.QO TO RemoteString_0_1_0.check;
            F_EQ.OUT TO RemoteString_0_1_1.check;
            DINT2DINT.OUT TO F_EQ.IN1;
            CLIENT_3_0.QO TO RemoteString_3_0_0.check;
            DINT2DINT_7.OUT TO F_EQ_1.IN1;
            DINT2DINT_8.OUT TO F_EQ_2.IN1;
            F_EQ_1.OUT TO RemoteString_3_2_1.check;
            F_EQ_2.OUT TO RemoteString_3_2_2.check;
            CLIENT_3_2.QO TO RemoteString_3_2_0.check;
            E_CTU.Q TO E_PERMIT.PERMIT;
            E_CTU_1.Q TO E_PERMIT_1.PERMIT;
            E_CTU_2.Q TO E_PERMIT_2.PERMIT;
          END_CONNECTIONS
        END_SUBAPPLICATION
        SUBAPPLICATION RemoteByteStringMethod
          EVENT_INPUT
            INIT;
            REQ;
          END_EVENT
          EVENT_OUTPUT
            INITO;
            CNF;
          END_EVENT
          VAR_INPUT
            QI : BOOL;
          END_VAR
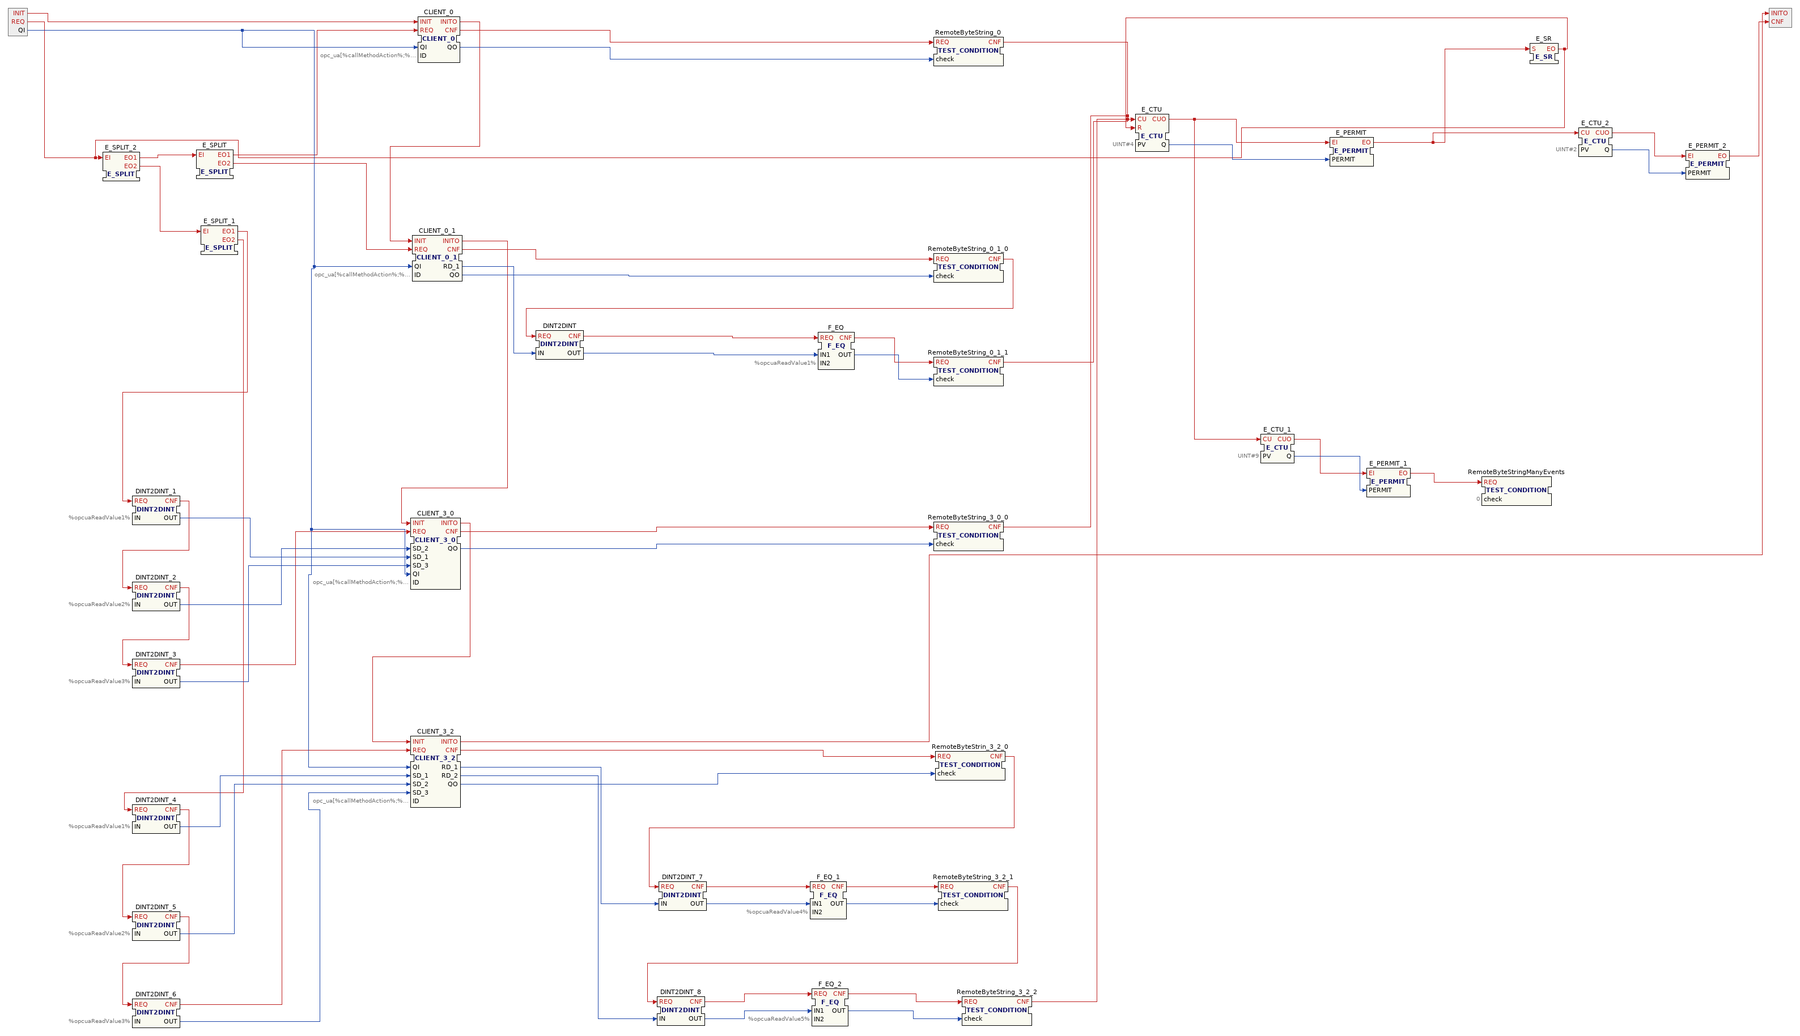
          FBS
            DINT2DINT_4 : DINT2DINT(IN := %opcuaReadValue1%);
            CLIENT_0 : CLIENT_0(ID := opc_ua[%callMethodAction%;%serverEndpoint%;%opcuaMethodCreation13%]);
            DINT2DINT_2 : DINT2DINT(IN := %opcuaReadValue2%);
            CLIENT_0_1 : CLIENT_0_1(ID := opc_ua[%callMethodAction%;%serverEndpoint%;%opcuaMethodCreation14%]);
            DINT2DINT : DINT2DINT;
            DINT2DINT_1 : DINT2DINT(IN := %opcuaReadValue1%);
            CLIENT_3_0 : CLIENT_3_0(ID := opc_ua[%callMethodAction%;%serverEndpoint%;%opcuaMethodCreation15%]);
            CLIENT_3_2 : CLIENT_3_2(ID := opc_ua[%callMethodAction%;%serverEndpoint%;%opcuaMethodCreation16%]);
            DINT2DINT_3 : DINT2DINT(IN := %opcuaReadValue3%);
            DINT2DINT_5 : DINT2DINT(IN := %opcuaReadValue2%);
            DINT2DINT_6 : DINT2DINT(IN := %opcuaReadValue3%);
            DINT2DINT_7 : DINT2DINT;
            DINT2DINT_8 : DINT2DINT;
            RemoteByteString_3_2_1 : TEST_CONDITION;
            RemoteByteString_3_2_2 : TEST_CONDITION;
            RemoteByteString_0 : TEST_CONDITION;
            RemoteByteString_0_1_0 : TEST_CONDITION;
            RemoteByteString_0_1_1 : TEST_CONDITION;
            RemoteByteStrin_3_2_0 : TEST_CONDITION;
            RemoteByteString_3_0_0 : TEST_CONDITION;
            F_EQ : F_EQ(IN2 := %opcuaReadValue1%);
            F_EQ_1 : F_EQ(IN2 := %opcuaReadValue4%);
            F_EQ_2 : F_EQ(IN2 := %opcuaReadValue5%);
            E_SPLIT : E_SPLIT;
            E_SPLIT_1 : E_SPLIT;
            E_CTU : E_CTU(PV := UINT#4);
            E_PERMIT : E_PERMIT;
            E_CTU_1 : E_CTU(PV := UINT#9);
            E_PERMIT_1 : E_PERMIT;
            RemoteByteStringManyEvents : TEST_CONDITION(check := 0);
            E_SPLIT_2 : E_SPLIT;
            E_PERMIT_2 : E_PERMIT;
            E_CTU_2 : E_CTU(PV := UINT#2);
            E_SR : E_SR;
          END_FBS
          EVENT_CONNECTIONS
            DINT2DINT_1.CNF TO DINT2DINT_2.REQ;
            DINT2DINT_2.CNF TO DINT2DINT_3.REQ;
            CLIENT_0_1.INITO TO CLIENT_3_0.INIT;
            INIT TO CLIENT_0.INIT;
            CLIENT_0.INITO TO CLIENT_0_1.INIT;
            CLIENT_3_0.INITO TO CLIENT_3_2.INIT;
            CLIENT_3_2.INITO TO INITO;
            CLIENT_0.CNF TO RemoteByteString_0.REQ;
            F_EQ.CNF TO RemoteByteString_0_1_1.REQ;
            CLIENT_3_0.CNF TO RemoteByteString_3_0_0.REQ;
            DINT2DINT_8.CNF TO F_EQ_2.REQ;
            DINT2DINT_7.CNF TO F_EQ_1.REQ;
            RemoteByteStrin_3_2_0.CNF TO DINT2DINT_7.REQ;
            F_EQ_1.CNF TO RemoteByteString_3_2_1.REQ;
            RemoteByteString_3_2_1.CNF TO DINT2DINT_8.REQ;
            F_EQ_2.CNF TO RemoteByteString_3_2_2.REQ;
            CLIENT_3_2.CNF TO RemoteByteStrin_3_2_0.REQ;
            DINT2DINT_4.CNF TO DINT2DINT_5.REQ;
            DINT2DINT_5.CNF TO DINT2DINT_6.REQ;
            DINT2DINT_6.CNF TO CLIENT_3_2.REQ;
            CLIENT_0_1.CNF TO RemoteByteString_0_1_0.REQ;
            RemoteByteString_0_1_0.CNF TO DINT2DINT.REQ;
            DINT2DINT.CNF TO F_EQ.REQ;
            DINT2DINT_3.CNF TO CLIENT_3_0.REQ;
            E_SPLIT.EO1 TO CLIENT_0.REQ;
            RemoteByteString_3_2_2.CNF TO E_CTU.CU;
            E_CTU.CUO TO E_CTU_1.CU;
            E_CTU.CUO TO E_PERMIT.EI;
            E_CTU_1.CUO TO E_PERMIT_1.EI;
            E_PERMIT_1.EO TO RemoteByteStringManyEvents.REQ;
            RemoteByteString_0.CNF TO E_CTU.CU;
            E_SPLIT.EO2 TO CLIENT_0_1.REQ;
            RemoteByteString_0_1_1.CNF TO E_CTU.CU;
            E_SPLIT_1.EO1 TO DINT2DINT_1.REQ;
            RemoteByteString_3_0_0.CNF TO E_CTU.CU;
            E_SPLIT_1.EO2 TO DINT2DINT_4.REQ;
            REQ TO E_SPLIT_2.EI;
            E_SPLIT_2.EO1 TO E_SPLIT.EI;
            E_SPLIT_2.EO2 TO E_SPLIT_1.EI;
            E_PERMIT.EO TO E_CTU_2.CU;
            E_CTU_2.CUO TO E_PERMIT_2.EI;
            E_PERMIT_2.EO TO CNF;
            E_PERMIT.EO TO E_SR.S;
            E_SR.EO TO E_CTU.R;
            E_SR.EO TO E_SPLIT_2.EI;
          END_CONNECTIONS
          DATA_CONNECTIONS
            DINT2DINT_2.OUT TO CLIENT_3_0.SD_2;
            CLIENT_0_1.RD_1 TO DINT2DINT.IN;
            DINT2DINT_1.OUT TO CLIENT_3_0.SD_1;
            DINT2DINT_3.OUT TO CLIENT_3_0.SD_3;
            QI TO CLIENT_0_1.QI;
            QI TO CLIENT_3_0.QI;
            QI TO CLIENT_3_2.QI;
            QI TO CLIENT_0.QI;
            DINT2DINT_4.OUT TO CLIENT_3_2.SD_1;
            DINT2DINT_5.OUT TO CLIENT_3_2.SD_2;
            CLIENT_3_2.RD_1 TO DINT2DINT_7.IN;
            CLIENT_3_2.RD_2 TO DINT2DINT_8.IN;
            DINT2DINT_6.OUT TO CLIENT_3_2.SD_3;
            CLIENT_0.QO TO RemoteByteString_0.check;
            CLIENT_0_1.QO TO RemoteByteString_0_1_0.check;
            F_EQ.OUT TO RemoteByteString_0_1_1.check;
            DINT2DINT.OUT TO F_EQ.IN1;
            CLIENT_3_0.QO TO RemoteByteString_3_0_0.check;
            DINT2DINT_7.OUT TO F_EQ_1.IN1;
            DINT2DINT_8.OUT TO F_EQ_2.IN1;
            F_EQ_1.OUT TO RemoteByteString_3_2_1.check;
            F_EQ_2.OUT TO RemoteByteString_3_2_2.check;
            CLIENT_3_2.QO TO RemoteByteStrin_3_2_0.check;
            E_CTU.Q TO E_PERMIT.PERMIT;
            E_CTU_1.Q TO E_PERMIT_1.PERMIT;
            E_CTU_2.Q TO E_PERMIT_2.PERMIT;
          END_CONNECTIONS
        END_SUBAPPLICATION
        EVENT_CONNECTIONS
          INIT TO RemoteBrowseName.INIT;
          REQ TO RemoteBrowseName.REQ;
          RemoteBrowseName.INITO TO RemoteNumericMethod.INIT;
          RemoteNumericMethod.INITO TO RemoteStringMethod.INIT;
          RemoteStringMethod.INITO TO RemoteByteStringMethod.INIT;
          RemoteByteStringMethod.CNF TO CNF;
          RemoteByteStringMethod.INITO TO INITO;
          RemoteStringMethod.CNF TO RemoteByteStringMethod.REQ;
          RemoteNumericMethod.CNF TO RemoteStringMethod.REQ;
          RemoteBrowseName.CNF TO RemoteNumericMethod.REQ;
        END_CONNECTIONS
        DATA_CONNECTIONS
          QI TO RemoteBrowseName.QI;
          QI TO RemoteNumericMethod.QI;
          QI TO RemoteStringMethod.QI;
          QI TO RemoteByteStringMethod.QI;
        END_CONNECTIONS
      END_SUBAPPLICATION
      SUBAPPLICATION stringNodeIdTestRemote_1
        EVENT_INPUT
          INIT;
          REQ;
        END_EVENT
        EVENT_OUTPUT
          INITO;
          CNF;
        END_EVENT
        VAR_INPUT
          QI : BOOL;
        END_VAR
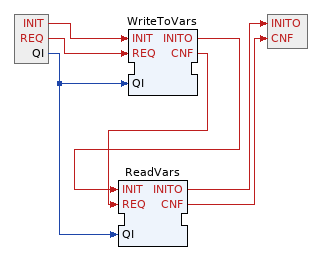
        SUBAPPLICATION WriteToVars
          EVENT_INPUT
            INIT;
            REQ;
          END_EVENT
          EVENT_OUTPUT
            INITO;
            CNF;
          END_EVENT
          VAR_INPUT
            QI : BOOL;
          END_VAR
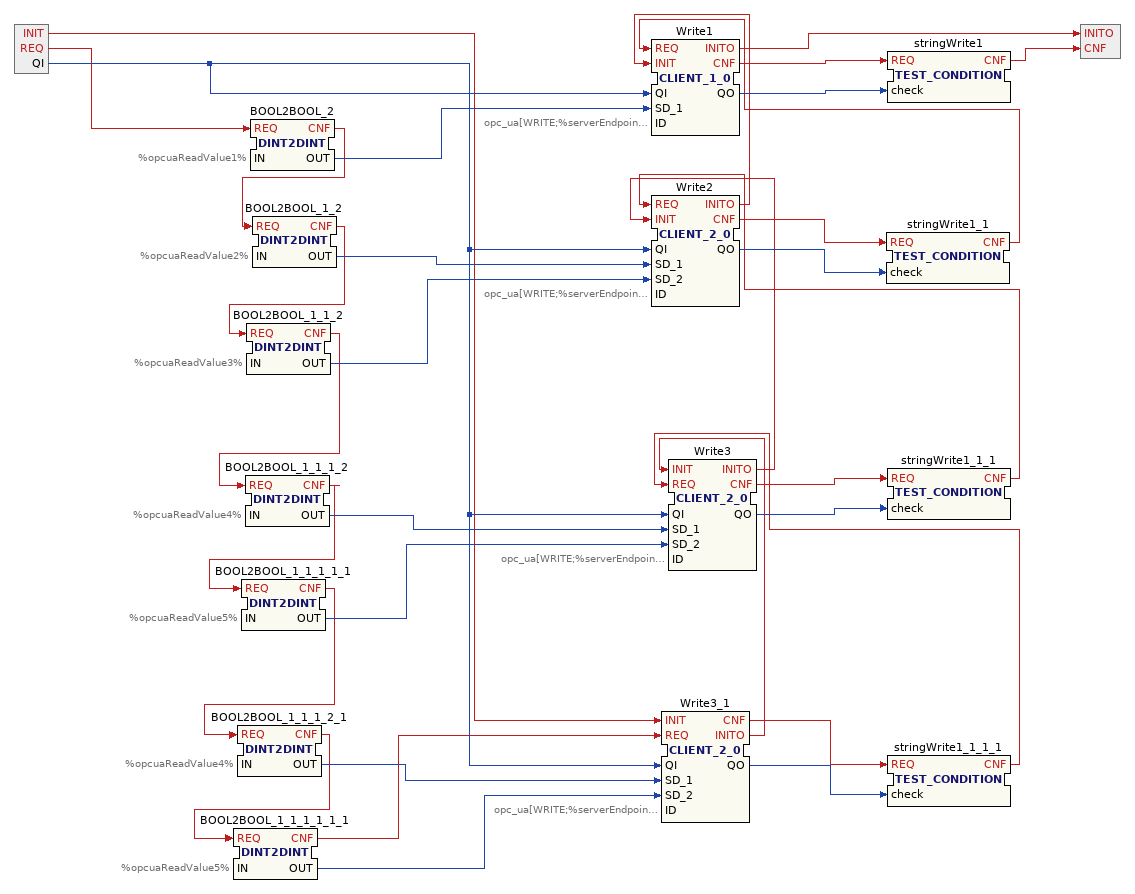
          FBS
            BOOL2BOOL_1_1_2 : DINT2DINT(IN := %opcuaReadValue3%);
            BOOL2BOOL_1_1_1_1_1 : DINT2DINT(IN := %opcuaReadValue5%);
            BOOL2BOOL_1_1_1_2 : DINT2DINT(IN := %opcuaReadValue4%);
            BOOL2BOOL_2 : DINT2DINT(IN := %opcuaReadValue1%);
            BOOL2BOOL_1_2 : DINT2DINT(IN := %opcuaReadValue2%);
            BOOL2BOOL_1_1_1_2_1 : DINT2DINT(IN := %opcuaReadValue4%);
            BOOL2BOOL_1_1_1_1_1_1 : DINT2DINT(IN := %opcuaReadValue5%);
            stringWrite1 : TEST_CONDITION;
            stringWrite1_1 : TEST_CONDITION;
            stringWrite1_1_1 : TEST_CONDITION;
            stringWrite1_1_1_1 : TEST_CONDITION;
            Write1 : CLIENT_1_0(ID := opc_ua[WRITE;%serverEndpoint%;%opcuaFolderTestWithNodeIdString1%]);
            Write2 : CLIENT_2_0(ID := opc_ua[WRITE;%serverEndpoint%;%opcuaFolderTestWithNodeIdString2%]);
            Write3_1 : CLIENT_2_0(ID := opc_ua[WRITE;%serverEndpoint%;,1:s=hello3;,1:s=hello4]);
            Write3 : CLIENT_2_0(ID := opc_ua[WRITE;%serverEndpoint%;%opcuaFolderTestWithNodeIdString3%]);
          END_FBS
          EVENT_CONNECTIONS
            BOOL2BOOL_1_2.CNF TO BOOL2BOOL_1_1_2.REQ;
            BOOL2BOOL_1_1_2.CNF TO BOOL2BOOL_1_1_1_2.REQ;
            BOOL2BOOL_1_1_1_2.CNF TO BOOL2BOOL_1_1_1_1_1.REQ;
            BOOL2BOOL_2.CNF TO BOOL2BOOL_1_2.REQ;
            REQ TO BOOL2BOOL_2.REQ;
            BOOL2BOOL_1_1_1_2_1.CNF TO BOOL2BOOL_1_1_1_1_1_1.REQ;
            BOOL2BOOL_1_1_1_1_1.CNF TO BOOL2BOOL_1_1_1_2_1.REQ;
            stringWrite1.CNF TO CNF;
            stringWrite1_1.CNF TO Write1.REQ;
            Write1.INITO TO INITO;
            Write1.CNF TO stringWrite1.REQ;
            stringWrite1_1_1.CNF TO Write2.REQ;
            Write2.INITO TO Write1.INIT;
            Write2.CNF TO stringWrite1_1.REQ;
            INIT TO Write3_1.INIT;
            BOOL2BOOL_1_1_1_1_1_1.CNF TO Write3_1.REQ;
            Write3_1.CNF TO stringWrite1_1_1_1.REQ;
            Write3_1.INITO TO Write3.INIT;
            stringWrite1_1_1_1.CNF TO Write3.REQ;
            Write3.INITO TO Write2.INIT;
            Write3.CNF TO stringWrite1_1_1.REQ;
          END_CONNECTIONS
          DATA_CONNECTIONS
            QI TO Write1.QI;
            BOOL2BOOL_2.OUT TO Write1.SD_1;
            Write1.QO TO stringWrite1.check;
            QI TO Write2.QI;
            BOOL2BOOL_1_2.OUT TO Write2.SD_1;
            BOOL2BOOL_1_1_2.OUT TO Write2.SD_2;
            Write2.QO TO stringWrite1_1.check;
            QI TO Write3_1.QI;
            BOOL2BOOL_1_1_1_2_1.OUT TO Write3_1.SD_1;
            BOOL2BOOL_1_1_1_1_1_1.OUT TO Write3_1.SD_2;
            Write3_1.QO TO stringWrite1_1_1_1.check;
            QI TO Write3.QI;
            BOOL2BOOL_1_1_1_2.OUT TO Write3.SD_1;
            BOOL2BOOL_1_1_1_1_1.OUT TO Write3.SD_2;
            Write3.QO TO stringWrite1_1_1.check;
          END_CONNECTIONS
        END_SUBAPPLICATION
        SUBAPPLICATION ReadVars
          EVENT_INPUT
            INIT;
            REQ;
          END_EVENT
          EVENT_OUTPUT
            INITO;
            CNF;
          END_EVENT
          VAR_INPUT
            QI : BOOL;
          END_VAR
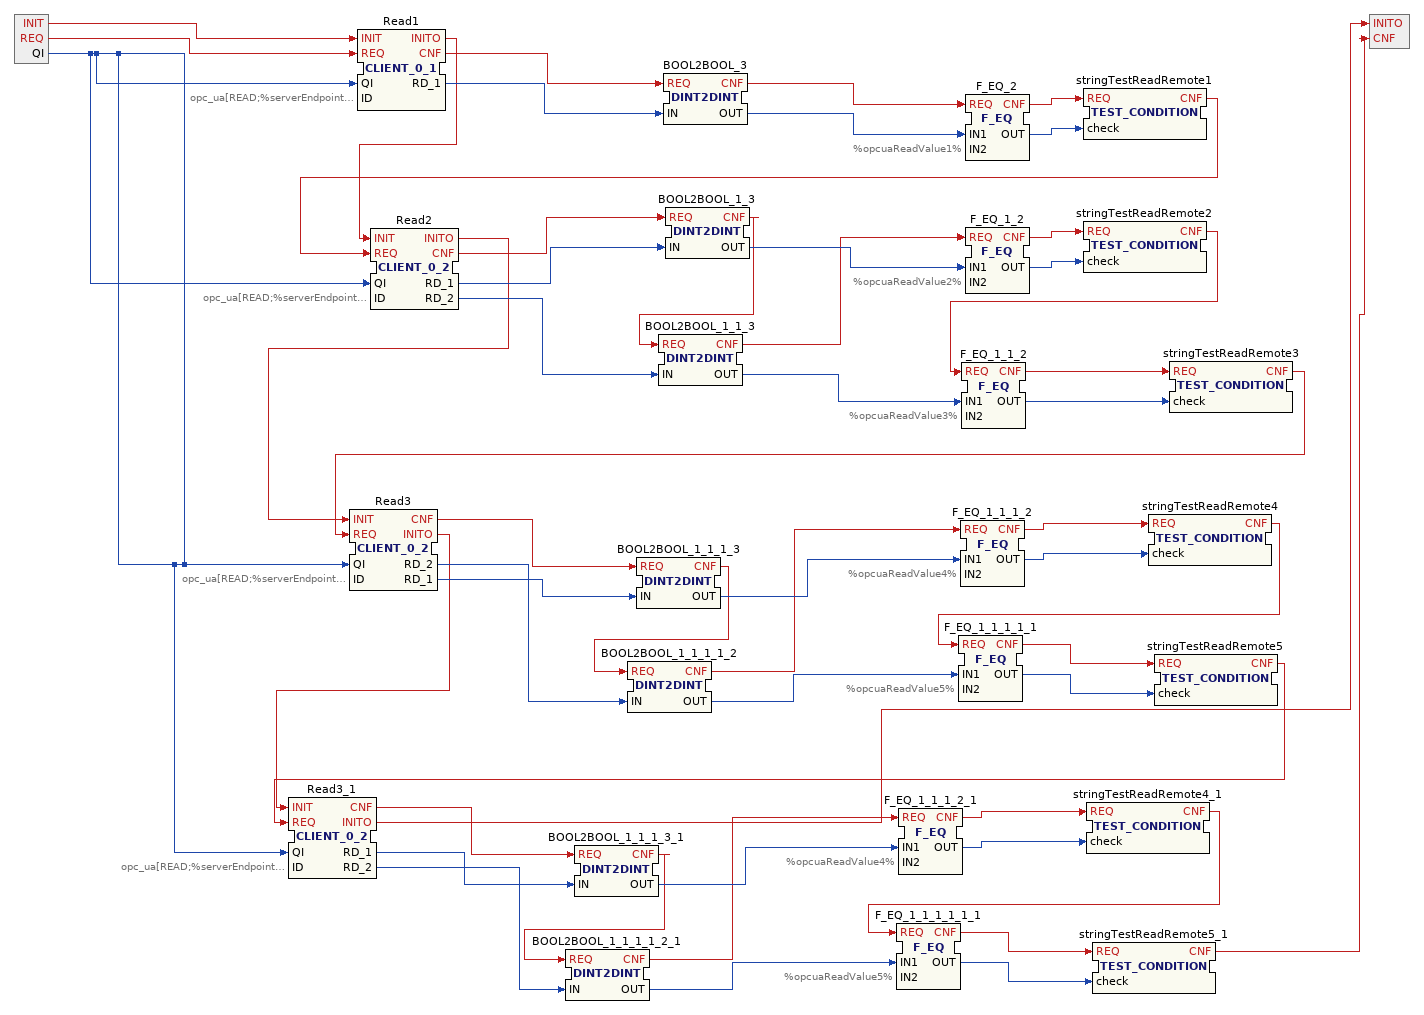
          FBS
            Read1 : CLIENT_0_1(ID := opc_ua[READ;%serverEndpoint%;%opcuaFolderTestWithNodeIdString1%]);
            Read2 : CLIENT_0_2(ID := opc_ua[READ;%serverEndpoint%;%opcuaFolderTestWithNodeIdString2%]);
            F_EQ_1_1_1_2 : F_EQ(IN2 := %opcuaReadValue4%);
            stringTestReadRemote4 : TEST_CONDITION;
            BOOL2BOOL_1_3 : DINT2DINT;
            F_EQ_1_1_1_1_1 : F_EQ(IN2 := %opcuaReadValue5%);
            stringTestReadRemote3 : TEST_CONDITION;
            BOOL2BOOL_1_1_3 : DINT2DINT;
            BOOL2BOOL_1_1_1_1_2 : DINT2DINT;
            BOOL2BOOL_1_1_1_3 : DINT2DINT;
            stringTestReadRemote2 : TEST_CONDITION;
            F_EQ_1_1_2 : F_EQ(IN2 := %opcuaReadValue3%);
            F_EQ_2 : F_EQ(IN2 := %opcuaReadValue1%);
            F_EQ_1_2 : F_EQ(IN2 := %opcuaReadValue2%);
            Read3 : CLIENT_0_2(ID := opc_ua[READ;%serverEndpoint%;%opcuaFolderTestWithNodeIdString3%]);
            stringTestReadRemote5 : TEST_CONDITION;
            stringTestReadRemote1 : TEST_CONDITION;
            BOOL2BOOL_3 : DINT2DINT;
            stringTestReadRemote5_1 : TEST_CONDITION;
            F_EQ_1_1_1_2_1 : F_EQ(IN2 := %opcuaReadValue4%);
            Read3_1 : CLIENT_0_2(ID := opc_ua[READ;%serverEndpoint%;,1:s=hello3;,1:s=hello4]);
            F_EQ_1_1_1_1_1_1 : F_EQ(IN2 := %opcuaReadValue5%);
            BOOL2BOOL_1_1_1_1_2_1 : DINT2DINT;
            BOOL2BOOL_1_1_1_3_1 : DINT2DINT;
            stringTestReadRemote4_1 : TEST_CONDITION;
          END_FBS
          EVENT_CONNECTIONS
            Read1.INITO TO Read2.INIT;
            Read1.CNF TO BOOL2BOOL_3.REQ;
            stringTestReadRemote1.CNF TO Read2.REQ;
            Read2.INITO TO Read3.INIT;
            Read2.CNF TO BOOL2BOOL_1_3.REQ;
            BOOL2BOOL_1_1_1_1_2.CNF TO F_EQ_1_1_1_2.REQ;
            F_EQ_1_1_1_2.CNF TO stringTestReadRemote4.REQ;
            stringTestReadRemote4.CNF TO F_EQ_1_1_1_1_1.REQ;
            BOOL2BOOL_1_3.CNF TO BOOL2BOOL_1_1_3.REQ;
            F_EQ_1_1_1_1_1.CNF TO stringTestReadRemote5.REQ;
            F_EQ_1_1_2.CNF TO stringTestReadRemote3.REQ;
            stringTestReadRemote3.CNF TO Read3.REQ;
            BOOL2BOOL_1_1_3.CNF TO F_EQ_1_2.REQ;
            BOOL2BOOL_1_1_1_3.CNF TO BOOL2BOOL_1_1_1_1_2.REQ;
            Read3.CNF TO BOOL2BOOL_1_1_1_3.REQ;
            F_EQ_1_2.CNF TO stringTestReadRemote2.REQ;
            stringTestReadRemote2.CNF TO F_EQ_1_1_2.REQ;
            BOOL2BOOL_3.CNF TO F_EQ_2.REQ;
            F_EQ_2.CNF TO stringTestReadRemote1.REQ;
            INIT TO Read1.INIT;
            REQ TO Read1.REQ;
            BOOL2BOOL_1_1_1_1_2_1.CNF TO F_EQ_1_1_1_2_1.REQ;
            BOOL2BOOL_1_1_1_3_1.CNF TO BOOL2BOOL_1_1_1_1_2_1.REQ;
            F_EQ_1_1_1_2_1.CNF TO stringTestReadRemote4_1.REQ;
            Read3_1.CNF TO BOOL2BOOL_1_1_1_3_1.REQ;
            F_EQ_1_1_1_1_1_1.CNF TO stringTestReadRemote5_1.REQ;
            stringTestReadRemote4_1.CNF TO F_EQ_1_1_1_1_1_1.REQ;
            Read3_1.INITO TO INITO;
            Read3.INITO TO Read3_1.INIT;
            stringTestReadRemote5_1.CNF TO CNF;
            stringTestReadRemote5.CNF TO Read3_1.REQ;
          END_CONNECTIONS
          DATA_CONNECTIONS
            Read1.RD_1 TO BOOL2BOOL_3.IN;
            Read2.RD_1 TO BOOL2BOOL_1_3.IN;
            Read2.RD_2 TO BOOL2BOOL_1_1_3.IN;
            BOOL2BOOL_1_1_1_3.OUT TO F_EQ_1_1_1_2.IN1;
            F_EQ_1_1_1_2.OUT TO stringTestReadRemote4.check;
            BOOL2BOOL_1_3.OUT TO F_EQ_1_2.IN1;
            BOOL2BOOL_1_1_1_1_2.OUT TO F_EQ_1_1_1_1_1.IN1;
            F_EQ_1_1_1_1_1.OUT TO stringTestReadRemote5.check;
            F_EQ_1_1_2.OUT TO stringTestReadRemote3.check;
            BOOL2BOOL_1_1_3.OUT TO F_EQ_1_1_2.IN1;
            Read3.RD_2 TO BOOL2BOOL_1_1_1_1_2.IN;
            Read3.RD_1 TO BOOL2BOOL_1_1_1_3.IN;
            F_EQ_1_2.OUT TO stringTestReadRemote2.check;
            BOOL2BOOL_3.OUT TO F_EQ_2.IN1;
            F_EQ_2.OUT TO stringTestReadRemote1.check;
            QI TO Read1.QI;
            QI TO Read2.QI;
            QI TO Read3.QI;
            Read3_1.RD_1 TO BOOL2BOOL_1_1_1_3_1.IN;
            Read3_1.RD_2 TO BOOL2BOOL_1_1_1_1_2_1.IN;
            F_EQ_1_1_1_2_1.OUT TO stringTestReadRemote4_1.check;
            F_EQ_1_1_1_1_1_1.OUT TO stringTestReadRemote5_1.check;
            BOOL2BOOL_1_1_1_3_1.OUT TO F_EQ_1_1_1_2_1.IN1;
            BOOL2BOOL_1_1_1_1_2_1.OUT TO F_EQ_1_1_1_1_1_1.IN1;
            QI TO Read3_1.QI;
          END_CONNECTIONS
        END_SUBAPPLICATION
        EVENT_CONNECTIONS
          WriteToVars.INITO TO ReadVars.INIT;
          INIT TO WriteToVars.INIT;
          REQ TO WriteToVars.REQ;
          WriteToVars.CNF TO ReadVars.REQ;
          ReadVars.CNF TO CNF;
          ReadVars.INITO TO INITO;
        END_CONNECTIONS
        DATA_CONNECTIONS
          QI TO ReadVars.QI;
          QI TO WriteToVars.QI;
        END_CONNECTIONS
      END_SUBAPPLICATION
      SUBAPPLICATION HandleInit_1
        EVENT_INPUT
          InitFinished;
        END_EVENT
        EVENT_OUTPUT
          Execute;
        END_EVENT
        VAR_INPUT
          QI : BOOL;
        END_VAR
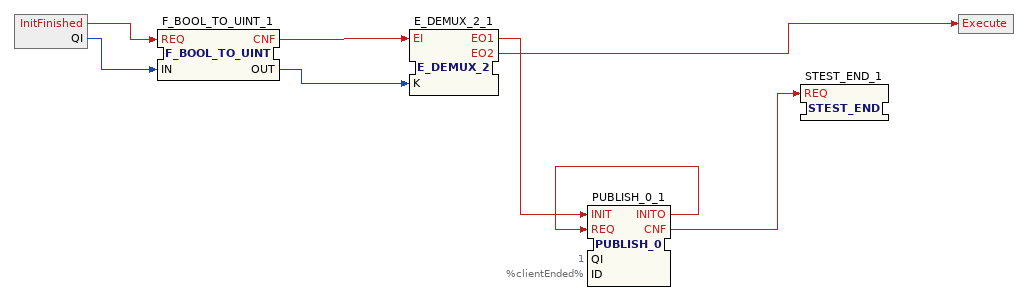
        FBS
          STEST_END_1 : STEST_END;
          E_DEMUX_2_1 : E_DEMUX_2;
          F_BOOL_TO_UINT_1 : F_BOOL_TO_UINT;
          PUBLISH_0_1 : PUBLISH_0(QI := 1, ID := %clientEnded%);
        END_FBS
        EVENT_CONNECTIONS
          F_BOOL_TO_UINT_1.CNF TO E_DEMUX_2_1.EI;
          E_DEMUX_2_1.EO1 TO PUBLISH_0_1.INIT;
          PUBLISH_0_1.INITO TO PUBLISH_0_1.REQ;
          E_DEMUX_2_1.EO2 TO Execute;
          InitFinished TO F_BOOL_TO_UINT_1.REQ;
          PUBLISH_0_1.CNF TO STEST_END_1.REQ;
        END_CONNECTIONS
        DATA_CONNECTIONS
          F_BOOL_TO_UINT_1.OUT TO E_DEMUX_2_1.K;
          QI TO F_BOOL_TO_UINT_1.IN;
        END_CONNECTIONS
      END_SUBAPPLICATION
      EVENT_CONNECTIONS
        InitFinishedSignal_1.INITO TO PUBLISH_0_1.INIT;
        InitFinishedSignal_1.IND TO PUBLISH_0_1.REQ;
        RemoteMethods_1.INITO TO RemoteIsolatedCases_1.INIT;
        RemoteMethods_1.CNF TO RemoteIsolatedCases_1.REQ;
        RemoteIsolatedCases_1.CNF TO E_SR_1_1.R;
        folderTestRemote_1.INITO TO numericNodeIdTestRemote_1.INIT;
        folderTestRemote_1.CNF TO numericNodeIdTestRemote_1.REQ;
        numericNodeIdTestRemote_1.INITO TO stringNodeIdTestRemote_1.INIT;
        numericNodeIdTestRemote_1.CNF TO stringNodeIdTestRemote_1.REQ;
        E_SR_2_1.EO TO E_PERMIT_1.EI;
        E_PERMIT_1.EO TO E_SR_1_1.S;
        E_SR_1_1.EO TO folderTestRemote_1.INIT;
        E_DELAY_1.EO TO folderTestRemote_1.REQ;
        stringNodeIdTestRemote_1.INITO TO bytestringNodeIdTestRemote_1.INIT;
        stringNodeIdTestRemote_1.CNF TO bytestringNodeIdTestRemote_1.REQ;
        bytestringNodeIdTestRemote_1.INITO TO RemoteMethods_1.INIT;
        bytestringNodeIdTestRemote_1.CNF TO RemoteMethods_1.REQ;
        PUBLISH_0_1.CNF TO E_SR_2_1.S;
        INIT TO InitFinishedSignal_1.INIT;
        HandleInit_1.Execute TO E_DELAY_1.START;
        RemoteIsolatedCases_1.INITO TO HandleInit_1.InitFinished;
      END_CONNECTIONS
      DATA_CONNECTIONS
        E_SR_1_1.Q TO RemoteIsolatedCases_1.QI;
        E_SR_1_1.Q TO numericNodeIdTestRemote_1.QI;
        E_SR_2_1.Q TO E_PERMIT_1.PERMIT;
        E_SR_1_1.Q TO folderTestRemote_1.QI;
        E_SR_1_1.Q TO bytestringNodeIdTestRemote_1.QI;
        E_SR_1_1.Q TO RemoteMethods_1.QI;
        E_SR_1_1.Q TO stringNodeIdTestRemote_1.QI;
        E_SR_1_1.Q TO HandleInit_1.QI;
      END_CONNECTIONS
    END_SUBAPPLICATION
    EVENT_CONNECTIONS
      SUBSCRIBE_0_1.IND TO E_SR.R;
      SUBSCRIBE_0_1.INITO TO E_SR.S;
      E_SR.EO TO folderTest.INIT;
      InitFinishedSignal.INITO TO PUBLISH_0.INIT;
      numericNodeIdTestRemote.INITO TO stringNodeIdTestRemote.INIT;
      stringNodeIdTestRemote.INITO TO bytestringNodeIdTestRemote.INIT;
      folderTestRemote.INITO TO numericNodeIdTestRemote.INIT;
      InitFinishedSignal.IND TO PUBLISH_0.REQ;
      E_SR_2.EO TO E_PERMIT.EI;
      PUBLISH_0.CNF TO E_SR_2.S;
      E_PERMIT.EO TO E_SR_1.S;
      E_DELAY.EO TO folderTestRemote.REQ;
      HandleInit.Execute TO E_DELAY.START;
      bytestringNodeIdTestRemote.INITO TO RemoteMethods.INIT;
      E_SR_1.EO TO folderTestRemote.INIT;
      bytestringNodeIdTestRemote.CNF TO RemoteMethods.REQ;
      stringNodeIdTestRemote.CNF TO bytestringNodeIdTestRemote.REQ;
      numericNodeIdTestRemote.CNF TO stringNodeIdTestRemote.REQ;
      folderTestRemote.CNF TO numericNodeIdTestRemote.REQ;
      numericNodeIdTest.INITO TO stringNodeIdTest.INIT;
      stringNodeIdTest.INITO TO byteStringNodeIdTest.INIT;
      byteStringNodeIdTest.INITO TO LocaMethods.INIT;
      folderTest.INITO TO numericNodeIdTest.INIT;
      LocaMethods.INITO TO IsolatedCases.INIT;
      IsolatedCases.INITO TO HandleInitLocal.InitFinished;
      RemoteIsolatedCases.INITO TO HandleInit.InitFinished;
      RemoteMethods.INITO TO RemoteIsolatedCases.INIT;
      RemoteIsolatedCases.CNF TO E_SR_1.R;
      RemoteMethods.CNF TO RemoteIsolatedCases.REQ;
    END_CONNECTIONS
    DATA_CONNECTIONS
      E_SR.Q TO folderTest.QI;
      E_SR.Q TO folderTest.QI;
      E_SR_1.Q TO folderTestRemote.QI;
      E_SR_1.Q TO HandleInit.QI;
      E_SR_1.Q TO HandleInit.QI;
      E_SR.Q TO HandleInitLocal.QI;
      E_SR.Q TO HandleInitLocal.QI;
      E_SR_1.Q TO numericNodeIdTestRemote.QI;
      E_SR_1.Q TO stringNodeIdTestRemote.QI;
      E_SR_1.Q TO bytestringNodeIdTestRemote.QI;
      E_SR_2.Q TO E_PERMIT.PERMIT;
      E_SR.Q TO numericNodeIdTest.QI;
      E_SR.Q TO stringNodeIdTest.QI;
      E_SR.Q TO byteStringNodeIdTest.QI;
      E_SR.Q TO LocaMethods.QI;
      E_SR_1.Q TO RemoteMethods.QI;
      E_SR.Q TO IsolatedCases.QI;
      E_SR_1.Q TO RemoteIsolatedCases.QI;
    END_CONNECTIONS
  END_APPLICATION
  APPLICATION OpcUaBothFailingCases
    FBS
      SUBSCRIBE_0_1 : SUBSCRIBE_0(QI := 1, ID := %clientEnded%);
      E_SR : E_SR;
      PUBLISH_0 : PUBLISH_0(QI := 1, ID := %serverInitCommIdACK%);
      E_DELAY : E_DELAY(DT := T#2s);
      InitFinishedSignal : SUBSCRIBE_0(QI := 1, ID := %serverInitCommId%);
      E_SR_2 : E_SR;
      GoodInputs : TEST_CONDITION;
      WorngInputs : TEST_CONDITION(check := 0);
      WorngInputsOutputs : TEST_CONDITION(check := 0);
      E_SWITCH : E_SWITCH;
      E_SWITCH_1 : E_SWITCH;
      Writable1 : PUBLISH_1(QI := 1, ID := opc_ua[WRITE;%opcuaFolderTestWithNodeIdNumeric1%/]);
      BOOL2BOOL_2_1 : DINT2DINT(IN := %opcuaReadValue1%);
      WorngInputsType : TEST_CONDITION(check := 0);
      SERVER_0 : SERVER_1(QI := 1, ID := opc_ua[%localMethodAction%;%opcuaMethodCreation5%]);
      SERVER_0_1 : SERVER_1(QI := 1, ID := opc_ua[%localMethodAction%;%opcuaMethodCreation6%]);
      SERVER_0_1_1 : SERVER_1(QI := 1, ID := opc_ua[%localMethodAction%;%opcuaMethodCreation7%]);
      DINT2DINT : DINT2DINT;
      DINT2DINT_1 : DINT2DINT;
      DINT2DINT_1_1 : DINT2DINT;
      SameNodeIdWrite : TEST_CONDITION;
      BOOL2BOOL_2_1_1 : DINT2DINT(IN := %opcuaReadValue1%);
      Writable1_1 : PUBLISH_1(QI := 1, ID := opc_ua[WRITE;/Objects/firstRead/NumericNodeId/folderTests/WithId1,1:i=12345]);
      BOOL2BOOL_2_1_1_1 : DINT2DINT(IN := %opcuaReadValue1%);
      Writable1_1_1 : PUBLISH_1(QI := 1, ID := opc_ua[WRITE;/Objects/firstRead/StringNodeId/folderTests/WithId,1:s=helloWrite]);
      SameNameDifferentNodeIdW : TEST_CONDITION;
      BOOL2BOOL_3 : DINT2DINT;
      SUBSCRIBE_1_1 : SUBSCRIBE_1(QI := 1, ID := opc_ua[READ;%opcuaFolderTestWithNodeIdNumeric1%]);
      SUBSCRIBE_1_1_1 : SUBSCRIBE_1(QI := 1, ID := opc_ua[READ;%opcuaFolderTestWithNodeIdNumeric1%]);
      BOOL2BOOL_3_1 : DINT2DINT;
      SameNodeSecondRead : TEST_CONDITION;
      ReadExistingWritable : TEST_CONDITION;
      F_NOT : F_NOT;
      F_NOT_1_1 : F_NOT;
      SUBSCRIBE_1_1_1_1 : SUBSCRIBE_1(QI := 1, ID := opc_ua[READ;/Objects/firstRead/StringNodeId/folderTests/WithId,1:s=hello]);
      ValidNode : TEST_CONDITION;
      WrongPath : TEST_CONDITION;
      SUBSCRIBE_wrongPath : SUBSCRIBE_1(QI := 1, ID := opc_ua[READ;///]);
      F_NOT_1_2_1 : F_NOT;
      SERVER_0_2 : SERVER_1(QI := 1, ID := opc_ua[%localMethodAction%;%opcuaMethodCreation5%]);
      DoubleMethod : TEST_CONDITION;
      F_NOT_1_2_1_1 : F_NOT;
      BOOL2BOOL_3_2 : DINT2DINT;
      BOOL2BOOL_3_1_1 : DINT2DINT;
      BOOL2BOOL_3_1_1_1 : DINT2DINT;
      F_NOT_1_2_1_1_1 : F_NOT;
      DifferentTypesOutput : TEST_CONDITION;
      BOOL2BOOL_3_2_1 : DINT2DINT;
      SUBSCRIBE_150 : SUBSCRIBE_1(QI := 1, ID := opc_ua[READ;%opcuaFolderTestWithNodeIdByteString1%]);
      BOOL2BOOL_3_2_1_1 : DINT2DINT;
      STRING2STRING_1 : STRING2STRING;
      F_NOT_1_2_1_1_1_1 : F_NOT;
      UnconnectedRD : TEST_CONDITION;
      F_NOT_1 : F_NOT;
      UnconnectedSD : TEST_CONDITION;
      SUBSCRIBE_140 : SUBSCRIBE_2(QI := 1, ID := opc_ua[READ;%opcuaFolderTestWithNodeIdString1%;%opcuaFolderTestWithNodeIdByteString2%]);
      SUBSCRIBE_1 : SUBSCRIBE_1(QI := 1, ID := opc_ua[READ;/Objects/firstRead/NumericNodeId/folderTests/WithId1,1:i=12345]);
      BOOL2BOOL_2_1_1_2 : DINT2DINT;
      SameNodeIdRead : TEST_CONDITION;
      F_NOT_2 : F_NOT;
      Writable1_1_2 : PUBLISH_2(QI := 1, ID := opc_ua[WRITE;%opcuaFolderTestWithNodeIdString1%;%opcuaFolderTestWithNodeIdByteString2%]);
      SameNameDifferentNodeIdR : TEST_CONDITION;
      F_EQ : F_EQ(IN2 := %opcuaReadValue1%);
      Writable1_2 : SUBSCRIBE_1(QI := 1, ID := opc_ua[READ;/Objects/firstRead/StringNodeId/folderTests/WithId,1:s=helloRead]);
      BOOL2BOOL_3_3 : DINT2DINT;
      STRING2STRING : INT2INT;
      WrongInputOutput : CLIENT_0(ID := opc_ua[%callMethodAction%;%unknownEndpoint%;%opcuaMethodCreation7%]);
      SameTypesOutput : TEST_CONDITION;
      SUBSCRIBE_150_1 : SUBSCRIBE_1(QI := 1, ID := opc_ua[READ;/Objects/firstRead/StringNodeId/folderTests/WithId,1:s=hello2]);
      BOOL2BOOL_3_2_1_2 : DINT2DINT;
      SUBSCRIBE_NoObject : SUBSCRIBE_1(QI := 1, ID := opc_ua[READ;/firstRead/Methods/byteStringNodeId/noOParameters]);
      F_NOT_1_2_1_2 : F_NOT;
      BOOL2BOOL_3_1_1_1_1 : DINT2DINT;
      BrowseWihtouObject : TEST_CONDITION;
      F_NOT_1_2_1_2_1 : F_NOT;
      BOOL2BOOL_3_1_1_1_1_1 : DINT2DINT;
      SUBSCRIBE_NoObject_1 : SUBSCRIBE_1(QI := 1, ID := opc_ua[READ;/Objects/firstRead/Methods/1:1:byteStringNodeId/noOParameters]);
      wrongNamespace1 : TEST_CONDITION;
      STRING2STRING_2 : DINT2DINT;
      Timeoutmethod : SERVER_0(QI := 1, ID := opc_ua[%localMethodAction%;%opcuaMethodCreation8%]);
      E_DELAY_1 : E_DELAY(DT := %methodValidDelay%);
      WrongInputOutput_1 : CLIENT_0(ID := opc_ua[%callMethodAction%;%unknownEndpoint%;%opcuaMethodCreation7%]);
      DINT2DINT_1_2 : DINT2DINT(IN := %opcuaReadValue2%);
      PUBLISH_1 : PUBLISH_1(QI := 1, ID := opc_ua[WRITE;%opcuaWRITEVariable%]);
      SERVER_0_3 : SERVER_0(QI := 1, ID := opc_ua[CREATE_METHOD;/Objects]);
      ObjectsFolder : TEST_CONDITION;
      F_NOT_1_2_1_2_1_1 : F_NOT;
      SERVER_0_4 : SERVER_0(QI := 1, ID := opc_ua[CREATE_METHOD;/Objects/notCalledMethod]);
    END_FBS
    SUBAPPLICATION HandleInitLocal
      EVENT_INPUT
        InitFinished;
      END_EVENT
      VAR_INPUT
        QI : BOOL;
      END_VAR
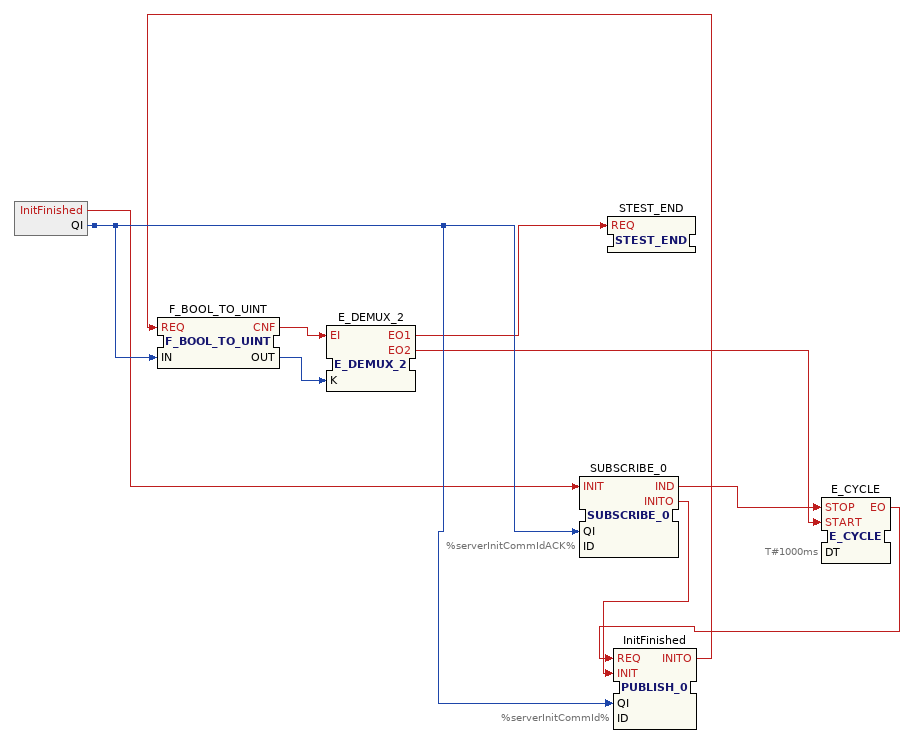
      FBS
        InitFinished : PUBLISH_0(ID := %serverInitCommId%);
        SUBSCRIBE_0 : SUBSCRIBE_0(ID := %serverInitCommIdACK%);
        E_CYCLE : E_CYCLE(DT := T#1000ms);
        E_DEMUX_2 : E_DEMUX_2;
        STEST_END : STEST_END;
        F_BOOL_TO_UINT : F_BOOL_TO_UINT;
      END_FBS
      EVENT_CONNECTIONS
        E_CYCLE.EO TO InitFinished.REQ;
        SUBSCRIBE_0.IND TO E_CYCLE.STOP;
        F_BOOL_TO_UINT.CNF TO E_DEMUX_2.EI;
        E_DEMUX_2.EO1 TO STEST_END.REQ;
        InitFinished TO SUBSCRIBE_0.INIT;
        SUBSCRIBE_0.INITO TO InitFinished.INIT;
        InitFinished.INITO TO F_BOOL_TO_UINT.REQ;
        E_DEMUX_2.EO2 TO E_CYCLE.START;
      END_CONNECTIONS
      DATA_CONNECTIONS
        F_BOOL_TO_UINT.OUT TO E_DEMUX_2.K;
        QI TO F_BOOL_TO_UINT.IN;
        QI TO InitFinished.QI;
        QI TO SUBSCRIBE_0.QI;
      END_CONNECTIONS
    END_SUBAPPLICATION
    SUBAPPLICATION HandleInit
      EVENT_INPUT
        InitFinished;
      END_EVENT
      EVENT_OUTPUT
        Execute;
      END_EVENT
      VAR_INPUT
        QI : BOOL;
      END_VAR
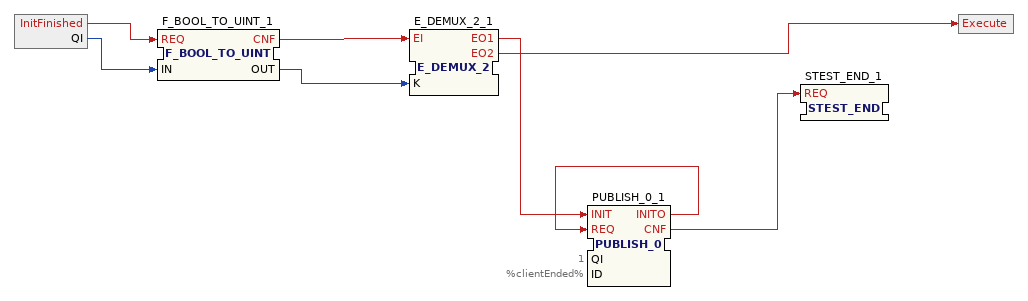
      FBS
        STEST_END_1 : STEST_END;
        E_DEMUX_2_1 : E_DEMUX_2;
        F_BOOL_TO_UINT_1 : F_BOOL_TO_UINT;
        PUBLISH_0_1 : PUBLISH_0(QI := 1, ID := %clientEnded%);
      END_FBS
      EVENT_CONNECTIONS
        F_BOOL_TO_UINT_1.CNF TO E_DEMUX_2_1.EI;
        E_DEMUX_2_1.EO1 TO PUBLISH_0_1.INIT;
        PUBLISH_0_1.INITO TO PUBLISH_0_1.REQ;
        E_DEMUX_2_1.EO2 TO Execute;
        InitFinished TO F_BOOL_TO_UINT_1.REQ;
        PUBLISH_0_1.CNF TO STEST_END_1.REQ;
      END_CONNECTIONS
      DATA_CONNECTIONS
        F_BOOL_TO_UINT_1.OUT TO E_DEMUX_2_1.K;
        QI TO F_BOOL_TO_UINT_1.IN;
      END_CONNECTIONS
    END_SUBAPPLICATION
    SUBAPPLICATION UnknownNode
      EVENT_INPUT
        INIT;
        REQ;
      END_EVENT
      EVENT_OUTPUT
        INITO;
        CNF;
      END_EVENT
      FBS
        dint : DINT2DINT;
        CallUnknown : CLIENT_0_1(QI := 1, ID := opc_ua[%callMethodAction%;%serverEndpoint%;%opcuaMethodCreation1%]);
        Read1 : CLIENT_0_1(QI := 1, ID := opc_ua[READ;%serverEndpoint%;%opcuaFolderTestOnlyBroseName1%]);
        ClientCallUnknown : TEST_CONDITION;
        dint_1 : DINT2DINT;
        F_NOT_2 : F_NOT;
        BOOL2BOOL_2 : DINT2DINT;
        ClienReadUnknown : TEST_CONDITION;
        F_NOT_2_1 : F_NOT;
        SubscribeUnknown : SUBSCRIBE_1(QI := 1, ID := opc_ua[SUBSCRIBE;%serverEndpoint%;/Objects/firstRead/NumericNodeId/folderTests/NotExisting,1:i=61499]);
        dint_2_1 : DINT2DINT;
        F_NOT_2_1_2 : F_NOT;
        ClienRead3_1Unknown : TEST_CONDITION;
        dint_3 : DINT2DINT;
        Read3_1Unknown : CLIENT_0_3(QI := 1, ID := opc_ua[READ;%serverEndpoint%;%opcuaFolderTestWithNodeIdNumeric1%;%opcuaFolderTestWithNodeIdString1%;opcuaFolderTestWithNodeIdByteString1]);
        dint_3_1 : DINT2DINT;
        dint_3_1_1 : DINT2DINT;
        F_NOT_2_1_3 : F_NOT;
        ClientWriteUnknown : TEST_CONDITION;
        ClienWrite3_1Unknown : TEST_CONDITION;
        F_NOT_2_1_3_1 : F_NOT;
        dint_3_1_1_1 : DINT2DINT;
        dint_3_2 : DINT2DINT;
        dint_3_1_2 : DINT2DINT;
        CLIENT_0 : CLIENT_0(QI := 1, ID := opc_ua[%callMethodAction%;%serverEndpoint%;%opcuaMethodCreation8%]);
        F_NOT_2_1_3_1_1 : F_NOT;
        ClientCallTimeoutMethod : TEST_CONDITION;
        F_NOT_2_1_3_1_1_1 : F_NOT;
        ClientWrongMethodNodeId : TEST_CONDITION;
        CLIENT_0_1 : CLIENT_0(QI := 1, ID := opc_ua[%callMethodAction%;%serverEndpoint%;/Objects/firstRead/Methods/numericNodeId/bothInputAndOutputParameters,1:i=61499]);
        F_NOT_2_1_3_1_1_1_1 : F_NOT;
        ClientWrongReadNodeId : TEST_CONDITION;
        ClientWrongWriteNodeId : TEST_CONDITION;
        F_NOT_2_1_3_1_1_1_1_1 : F_NOT;
        Subscribe3_1Unknown : SUBSCRIBE_3(QI := 1, ID := opc_ua[SUBSCRIBE;%serverEndpoint%;%opcuaFolderTestWithNodeIdNumeric1%;%opcuaFolderTestWithNodeIdString1%;opcuaFolderTestWithNodeIdByteString1]);
        dint_3_1_2_1 : DINT2DINT;
        dint_3_1_1_1_1 : DINT2DINT;
        dint_3_2_1 : DINT2DINT;
        CLIENT_0_1_1 : CLIENT_0_1(QI := 1, ID := opc_ua[READ;%serverEndpoint%;/Objects/firstRead/NumericNodeId/folderTests/WithId,1:i=61499]);
        DINT2DINT : DINT2DINT;
        DINT2DINT_1 : DINT2DINT;
        F_NOT_2_1_3_1_1_1_1_2 : F_NOT;
        DINT2DINT_2 : DINT2DINT;
        CLIENT_0_1_1_2 : CLIENT_0_1(QI := 1, ID := opc_ua[READ;%serverEndpoint%;,1:i=61499]);
        ClientWrongReadNodeId_NBN : TEST_CONDITION;
        DINT2DINT_1_1 : DINT2DINT;
        SubscribeUnknown_1 : SUBSCRIBE_1(QI := 1, ID := opc_ua[SUBSCRIBE;%serverEndpoint%;,1:i=61499]);
        dint_2_1_1 : DINT2DINT;
        Write1 : CLIENT_1_0(QI := 1, ID := opc_ua[WRITE;%serverEndpoint%;%opcuaFolderTestOnlyBroseName1%]);
        Write3_1Unknown : CLIENT_3_0(QI := 1, ID := opc_ua[WRITE;%serverEndpoint%;%opcuaFolderTestWithNodeIdNumeric1%;%opcuaFolderTestWithNodeIdString1%;opcuaFolderTestWithNodeIdByteString1]);
        CLIENT_0_1_1_1 : CLIENT_1_0(QI := 1, ID := opc_ua[WRITE;%serverEndpoint%;/Objects/firstRead/NumericNodeId/folderTests/WithId,1:i=61499]);
        CLIENT_0_1_1_1_1 : CLIENT_1_0(QI := 1, ID := opc_ua[WRITE;%serverEndpoint%;,1:i=61499]);
        ClientWrongWriteNodeId_NBN : TEST_CONDITION;
        F_NOT_2_1_3_1_1_1_1_2_1 : F_NOT;
      END_FBS
      EVENT_CONNECTIONS
        CallUnknown.INITO TO Read1.INIT;
        CallUnknown.CNF TO F_NOT_2.REQ;
        ClientCallUnknown.CNF TO Read1.REQ;
        Read1.CNF TO F_NOT_2_1.REQ;
        F_NOT_2.CNF TO ClientCallUnknown.REQ;
        F_NOT_2_1.CNF TO ClienReadUnknown.REQ;
        INIT TO CallUnknown.INIT;
        REQ TO CallUnknown.REQ;
        F_NOT_2_1_2.CNF TO ClienRead3_1Unknown.REQ;
        Read3_1Unknown.CNF TO F_NOT_2_1_2.REQ;
        SubscribeUnknown.INITO TO Read3_1Unknown.INIT;
        F_NOT_2_1_3.CNF TO ClientWriteUnknown.REQ;
        F_NOT_2_1_3_1.CNF TO ClienWrite3_1Unknown.REQ;
        ClienWrite3_1Unknown.CNF TO CLIENT_0.REQ;
        CLIENT_0.CNF TO F_NOT_2_1_3_1_1.REQ;
        F_NOT_2_1_3_1_1.CNF TO ClientCallTimeoutMethod.REQ;
        CLIENT_0.INITO TO CLIENT_0_1.INIT;
        ClientCallTimeoutMethod.CNF TO CLIENT_0_1.REQ;
        CLIENT_0_1.CNF TO F_NOT_2_1_3_1_1_1.REQ;
        F_NOT_2_1_3_1_1_1.CNF TO ClientWrongMethodNodeId.REQ;
        F_NOT_2_1_3_1_1_1_1.CNF TO ClientWrongReadNodeId.REQ;
        F_NOT_2_1_3_1_1_1_1_1.CNF TO ClientWrongWriteNodeId.REQ;
        ClientWriteUnknown.CNF TO Read3_1Unknown.REQ;
        CLIENT_0_1.INITO TO CLIENT_0_1_1.INIT;
        ClientWrongMethodNodeId.CNF TO CLIENT_0_1_1.REQ;
        CLIENT_0_1_1.CNF TO F_NOT_2_1_3_1_1_1_1.REQ;
        F_NOT_2_1_3_1_1_1_1_2.CNF TO ClientWrongReadNodeId_NBN.REQ;
        CLIENT_0_1_1_2.CNF TO F_NOT_2_1_3_1_1_1_1_2.REQ;
        ClientWrongWriteNodeId.CNF TO CLIENT_0_1_1_2.REQ;
        Subscribe3_1Unknown.INITO TO CLIENT_0_1_1_2.INIT;
        SubscribeUnknown_1.INITO TO INITO;
        Read1.INITO TO Write1.INIT;
        ClienReadUnknown.CNF TO Write1.REQ;
        Write1.INITO TO SubscribeUnknown.INIT;
        Write1.CNF TO F_NOT_2_1_3.REQ;
        Read3_1Unknown.INITO TO Write3_1Unknown.INIT;
        ClienRead3_1Unknown.CNF TO Write3_1Unknown.REQ;
        Write3_1Unknown.INITO TO CLIENT_0.INIT;
        Write3_1Unknown.CNF TO F_NOT_2_1_3_1.REQ;
        CLIENT_0_1_1.INITO TO CLIENT_0_1_1_1.INIT;
        ClientWrongReadNodeId.CNF TO CLIENT_0_1_1_1.REQ;
        CLIENT_0_1_1_1.INITO TO Subscribe3_1Unknown.INIT;
        CLIENT_0_1_1_1.CNF TO F_NOT_2_1_3_1_1_1_1_1.REQ;
        CLIENT_0_1_1_2.INITO TO CLIENT_0_1_1_1_1.INIT;
        ClientWrongReadNodeId_NBN.CNF TO CLIENT_0_1_1_1_1.REQ;
        CLIENT_0_1_1_1_1.INITO TO SubscribeUnknown_1.INIT;
        ClientWrongWriteNodeId_NBN.CNF TO CNF;
        F_NOT_2_1_3_1_1_1_1_2_1.CNF TO ClientWrongWriteNodeId_NBN.REQ;
        CLIENT_0_1_1_1_1.CNF TO F_NOT_2_1_3_1_1_1_1_2_1.REQ;
      END_CONNECTIONS
      DATA_CONNECTIONS
        Read1.RD_1 TO dint.IN;
        CallUnknown.QO TO F_NOT_2.IN;
        CallUnknown.RD_1 TO dint_1.IN;
        Read1.QO TO F_NOT_2_1.IN;
        F_NOT_2.OUT TO ClientCallUnknown.check;
        F_NOT_2_1.OUT TO ClienReadUnknown.check;
        SubscribeUnknown.RD_1 TO dint_2_1.IN;
        F_NOT_2_1_2.OUT TO ClienRead3_1Unknown.check;
        Read3_1Unknown.RD_1 TO dint_3.IN;
        Read3_1Unknown.RD_2 TO dint_3_1.IN;
        Read3_1Unknown.RD_3 TO dint_3_1_1.IN;
        Read3_1Unknown.QO TO F_NOT_2_1_2.IN;
        F_NOT_2_1_3.OUT TO ClientWriteUnknown.check;
        F_NOT_2_1_3_1.OUT TO ClienWrite3_1Unknown.check;
        CLIENT_0.QO TO F_NOT_2_1_3_1_1.IN;
        F_NOT_2_1_3_1_1.OUT TO ClientCallTimeoutMethod.check;
        CLIENT_0_1.QO TO F_NOT_2_1_3_1_1_1.IN;
        F_NOT_2_1_3_1_1_1.OUT TO ClientWrongMethodNodeId.check;
        F_NOT_2_1_3_1_1_1_1.OUT TO ClientWrongReadNodeId.check;
        F_NOT_2_1_3_1_1_1_1_1.OUT TO ClientWrongWriteNodeId.check;
        Subscribe3_1Unknown.RD_1 TO dint_3_2_1.IN;
        Subscribe3_1Unknown.RD_2 TO dint_3_1_2_1.IN;
        Subscribe3_1Unknown.RD_3 TO dint_3_1_1_1_1.IN;
        CLIENT_0_1_1.QO TO F_NOT_2_1_3_1_1_1_1.IN;
        CLIENT_0_1_1.RD_1 TO DINT2DINT.IN;
        F_NOT_2_1_3_1_1_1_1_2.OUT TO ClientWrongReadNodeId_NBN.check;
        CLIENT_0_1_1_2.QO TO F_NOT_2_1_3_1_1_1_1_2.IN;
        CLIENT_0_1_1_2.RD_1 TO DINT2DINT_2.IN;
        SubscribeUnknown_1.RD_1 TO dint_2_1_1.IN;
        BOOL2BOOL_2.OUT TO Write1.SD_1;
        Write1.QO TO F_NOT_2_1_3.IN;
        dint_3_2.OUT TO Write3_1Unknown.SD_1;
        dint_3_1_2.OUT TO Write3_1Unknown.SD_2;
        dint_3_1_1_1.OUT TO Write3_1Unknown.SD_3;
        Write3_1Unknown.QO TO F_NOT_2_1_3_1.IN;
        DINT2DINT_1.OUT TO CLIENT_0_1_1_1.SD_1;
        CLIENT_0_1_1_1.QO TO F_NOT_2_1_3_1_1_1_1_1.IN;
        DINT2DINT_1_1.OUT TO CLIENT_0_1_1_1_1.SD_1;
        F_NOT_2_1_3_1_1_1_1_2_1.OUT TO ClientWrongWriteNodeId_NBN.check;
        CLIENT_0_1_1_1_1.QO TO F_NOT_2_1_3_1_1_1_1_2_1.IN;
      END_CONNECTIONS
    END_SUBAPPLICATION
    SUBAPPLICATION WrongNoOfArguments
      EVENT_INPUT
        INIT;
        REQ;
      END_EVENT
      EVENT_OUTPUT
        INITO;
        CNF;
      END_EVENT
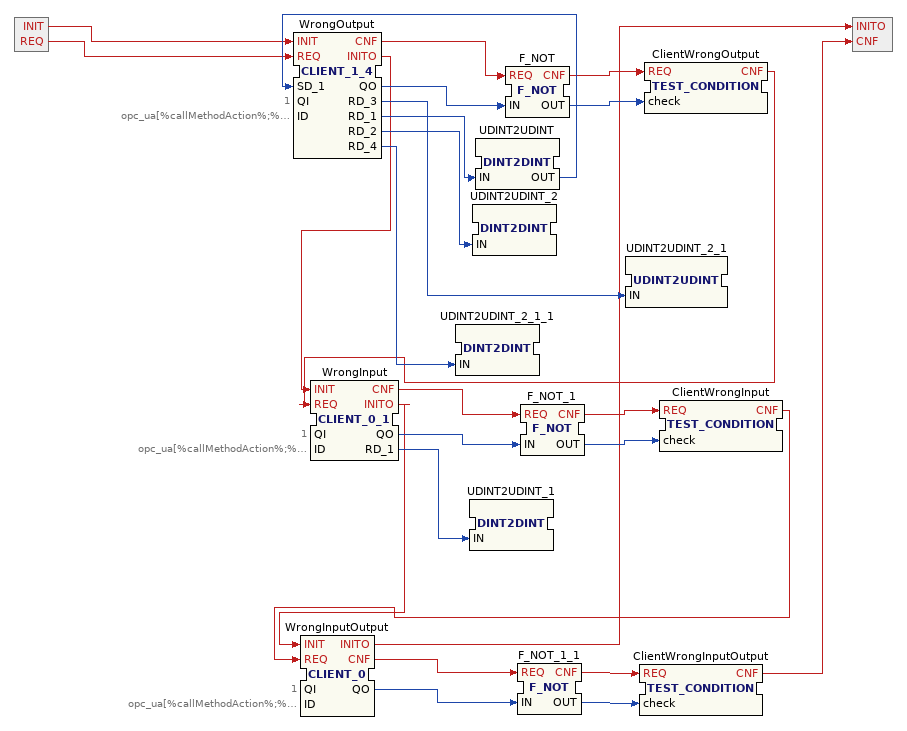
      FBS
        ClientWrongInputOutput : TEST_CONDITION;
        ClientWrongInput : TEST_CONDITION;
        F_NOT_1_1 : F_NOT;
        ClientWrongOutput : TEST_CONDITION;
        F_NOT_1 : F_NOT;
        F_NOT : F_NOT;
        WrongOutput : CLIENT_1_4(QI := 1, ID := opc_ua[%callMethodAction%;%serverEndpoint%;%opcuaMethodCreation5%]);
        UDINT2UDINT_2_1 : UDINT2UDINT;
        WrongInput : CLIENT_0_1(QI := 1, ID := opc_ua[%callMethodAction%;%serverEndpoint%;%opcuaMethodCreation6%]);
        WrongInputOutput : CLIENT_0(QI := 1, ID := opc_ua[%callMethodAction%;%serverEndpoint%;%opcuaMethodCreation7%]);
        UDINT2UDINT : DINT2DINT;
        UDINT2UDINT_2 : DINT2DINT;
        UDINT2UDINT_2_1_1 : DINT2DINT;
        UDINT2UDINT_1 : DINT2DINT;
      END_FBS
      EVENT_CONNECTIONS
        F_NOT_1_1.CNF TO ClientWrongInputOutput.REQ;
        F_NOT_1.CNF TO ClientWrongInput.REQ;
        F_NOT.CNF TO ClientWrongOutput.REQ;
        ClientWrongInputOutput.CNF TO CNF;
        INIT TO WrongOutput.INIT;
        REQ TO WrongOutput.REQ;
        WrongOutput.CNF TO F_NOT.REQ;
        WrongOutput.INITO TO WrongInput.INIT;
        ClientWrongOutput.CNF TO WrongInput.REQ;
        WrongInput.CNF TO F_NOT_1.REQ;
        WrongInput.INITO TO WrongInputOutput.INIT;
        ClientWrongInput.CNF TO WrongInputOutput.REQ;
        WrongInputOutput.INITO TO INITO;
        WrongInputOutput.CNF TO F_NOT_1_1.REQ;
      END_CONNECTIONS
      DATA_CONNECTIONS
        F_NOT_1_1.OUT TO ClientWrongInputOutput.check;
        F_NOT_1.OUT TO ClientWrongInput.check;
        F_NOT.OUT TO ClientWrongOutput.check;
        WrongOutput.QO TO F_NOT.IN;
        WrongOutput.RD_3 TO UDINT2UDINT_2_1.IN;
        WrongInput.QO TO F_NOT_1.IN;
        WrongInputOutput.QO TO F_NOT_1_1.IN;
        WrongOutput.RD_1 TO UDINT2UDINT.IN;
        UDINT2UDINT.OUT TO WrongOutput.SD_1;
        WrongOutput.RD_2 TO UDINT2UDINT_2.IN;
        WrongOutput.RD_4 TO UDINT2UDINT_2_1_1.IN;
        WrongInput.RD_1 TO UDINT2UDINT_1.IN;
      END_CONNECTIONS
    END_SUBAPPLICATION
    SUBAPPLICATION WrongType
      EVENT_INPUT
        INIT;
        REQ;
      END_EVENT
      EVENT_OUTPUT
        INITO;
        CNF;
      END_EVENT
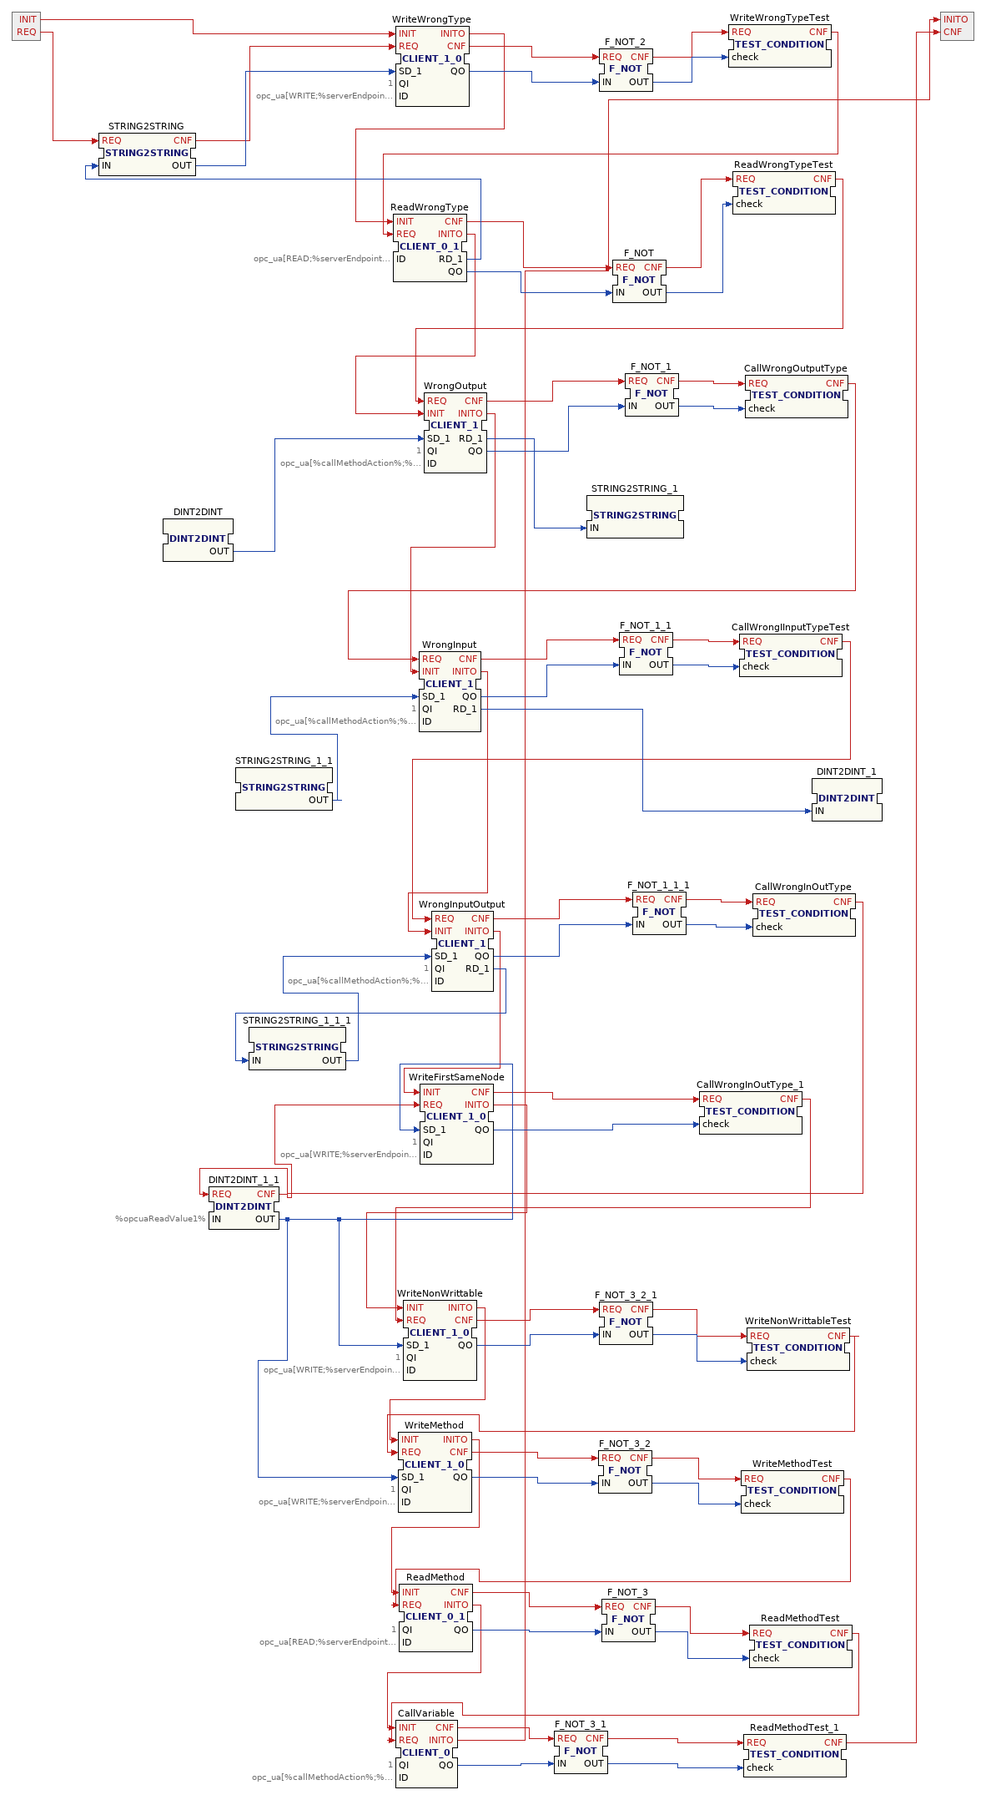
      FBS
        STRING2STRING : STRING2STRING;
        ReadWrongType : CLIENT_0_1(ID := opc_ua[READ;%serverEndpoint%;%opcuaFolderTestWithNodeIdNumeric1%]);
        ReadWrongTypeTest : TEST_CONDITION;
        F_NOT : F_NOT;
        WrongOutput : CLIENT_1(QI := 1, ID := opc_ua[%callMethodAction%;%serverEndpoint%;%opcuaMethodCreation5%]);
        DINT2DINT : DINT2DINT;
        STRING2STRING_1 : STRING2STRING;
        F_NOT_1 : F_NOT;
        CallWrongOutputType : TEST_CONDITION;
        STRING2STRING_1_1 : STRING2STRING;
        DINT2DINT_1 : DINT2DINT;
        CallWrongIInputTypeTest : TEST_CONDITION;
        F_NOT_1_1 : F_NOT;
        WrongInput : CLIENT_1(QI := 1, ID := opc_ua[%callMethodAction%;%serverEndpoint%;%opcuaMethodCreation6%]);
        STRING2STRING_1_1_1 : STRING2STRING;
        F_NOT_1_1_1 : F_NOT;
        CallWrongInOutType : TEST_CONDITION;
        WrongInputOutput : CLIENT_1(QI := 1, ID := opc_ua[%callMethodAction%;%serverEndpoint%;%opcuaMethodCreation6%]);
        DINT2DINT_1_1 : DINT2DINT(IN := %opcuaReadValue1%);
        F_NOT_3 : F_NOT;
        ReadMethod : CLIENT_0_1(QI := 1, ID := opc_ua[READ;%serverEndpoint%;%opcuaMethodCreation6%]);
        ReadMethodTest : TEST_CONDITION;
        CallVariable : CLIENT_0(QI := 1, ID := opc_ua[%callMethodAction%;%serverEndpoint%;%opcuaWRITEVariable%]);
        F_NOT_3_1 : F_NOT;
        ReadMethodTest_1 : TEST_CONDITION;
        WriteWrongType : CLIENT_1_0(QI := 1, ID := opc_ua[WRITE;%serverEndpoint%;%opcuaFolderTestWithNodeIdNumeric1%]);
        F_NOT_2 : F_NOT;
        WriteWrongTypeTest : TEST_CONDITION;
        WriteFirstSameNode : CLIENT_1_0(QI := 1, ID := opc_ua[WRITE;%serverEndpoint%;/Objects/firstRead/StringNodeId/folderTests/WithId]);
        CallWrongInOutType_1 : TEST_CONDITION;
        WriteMethod : CLIENT_1_0(QI := 1, ID := opc_ua[WRITE;%serverEndpoint%;%opcuaMethodCreation6%]);
        WriteNonWrittable : CLIENT_1_0(QI := 1, ID := opc_ua[WRITE;%serverEndpoint%;%opcuaWRITEVariable%]);
        F_NOT_3_2 : F_NOT;
        WriteMethodTest : TEST_CONDITION;
        WriteNonWrittableTest : TEST_CONDITION;
        F_NOT_3_2_1 : F_NOT;
      END_FBS
      EVENT_CONNECTIONS
        REQ TO STRING2STRING.REQ;
        ReadWrongType.CNF TO F_NOT.REQ;
        F_NOT.CNF TO ReadWrongTypeTest.REQ;
        WrongOutput.CNF TO F_NOT_1.REQ;
        F_NOT_1.CNF TO CallWrongOutputType.REQ;
        F_NOT_1_1.CNF TO CallWrongIInputTypeTest.REQ;
        WrongInput.CNF TO F_NOT_1_1.REQ;
        CallWrongOutputType.CNF TO WrongInput.REQ;
        WrongInputOutput.CNF TO F_NOT_1_1_1.REQ;
        F_NOT_1_1_1.CNF TO CallWrongInOutType.REQ;
        CallWrongIInputTypeTest.CNF TO WrongInputOutput.REQ;
        ReadWrongTypeTest.CNF TO WrongOutput.REQ;
        ReadWrongType.INITO TO WrongOutput.INIT;
        WrongOutput.INITO TO WrongInput.INIT;
        WrongInput.INITO TO WrongInputOutput.INIT;
        CallWrongInOutType.CNF TO DINT2DINT_1_1.REQ;
        ReadMethod.CNF TO F_NOT_3.REQ;
        F_NOT_3.CNF TO ReadMethodTest.REQ;
        ReadMethod.INITO TO CallVariable.INIT;
        CallVariable.CNF TO F_NOT_3_1.REQ;
        F_NOT_3_1.CNF TO ReadMethodTest_1.REQ;
        ReadMethodTest.CNF TO CallVariable.REQ;
        CallVariable.INITO TO INITO;
        ReadMethodTest_1.CNF TO CNF;
        INIT TO WriteWrongType.INIT;
        STRING2STRING.CNF TO WriteWrongType.REQ;
        WriteWrongType.INITO TO ReadWrongType.INIT;
        WriteWrongTypeTest.CNF TO ReadWrongType.REQ;
        F_NOT_2.CNF TO WriteWrongTypeTest.REQ;
        WriteWrongType.CNF TO F_NOT_2.REQ;
        WrongInputOutput.INITO TO WriteFirstSameNode.INIT;
        DINT2DINT_1_1.CNF TO WriteFirstSameNode.REQ;
        WriteFirstSameNode.CNF TO CallWrongInOutType_1.REQ;
        WriteMethod.INITO TO ReadMethod.INIT;
        WriteFirstSameNode.INITO TO WriteNonWrittable.INIT;
        CallWrongInOutType_1.CNF TO WriteNonWrittable.REQ;
        WriteNonWrittable.INITO TO WriteMethod.INIT;
        F_NOT_3_2_1.CNF TO WriteNonWrittableTest.REQ;
        WriteNonWrittableTest.CNF TO WriteMethod.REQ;
        WriteNonWrittable.CNF TO F_NOT_3_2_1.REQ;
        WriteMethodTest.CNF TO ReadMethod.REQ;
        F_NOT_3_2.CNF TO WriteMethodTest.REQ;
        WriteMethod.CNF TO F_NOT_3_2.REQ;
      END_CONNECTIONS
      DATA_CONNECTIONS
        ReadWrongType.RD_1 TO STRING2STRING.IN;
        F_NOT.OUT TO ReadWrongTypeTest.check;
        ReadWrongType.QO TO F_NOT.IN;
        DINT2DINT.OUT TO WrongOutput.SD_1;
        WrongOutput.RD_1 TO STRING2STRING_1.IN;
        WrongOutput.QO TO F_NOT_1.IN;
        F_NOT_1.OUT TO CallWrongOutputType.check;
        WrongInput.QO TO F_NOT_1_1.IN;
        F_NOT_1_1.OUT TO CallWrongIInputTypeTest.check;
        STRING2STRING_1_1.OUT TO WrongInput.SD_1;
        WrongInput.RD_1 TO DINT2DINT_1.IN;
        WrongInputOutput.QO TO F_NOT_1_1_1.IN;
        STRING2STRING_1_1_1.OUT TO WrongInputOutput.SD_1;
        F_NOT_1_1_1.OUT TO CallWrongInOutType.check;
        WrongInputOutput.RD_1 TO STRING2STRING_1_1_1.IN;
        ReadMethod.QO TO F_NOT_3.IN;
        F_NOT_3.OUT TO ReadMethodTest.check;
        CallVariable.QO TO F_NOT_3_1.IN;
        F_NOT_3_1.OUT TO ReadMethodTest_1.check;
        STRING2STRING.OUT TO WriteWrongType.SD_1;
        F_NOT_2.OUT TO WriteWrongTypeTest.check;
        WriteWrongType.QO TO F_NOT_2.IN;
        DINT2DINT_1_1.OUT TO WriteFirstSameNode.SD_1;
        WriteFirstSameNode.QO TO CallWrongInOutType_1.check;
        DINT2DINT_1_1.OUT TO WriteMethod.SD_1;
        DINT2DINT_1_1.OUT TO WriteNonWrittable.SD_1;
        F_NOT_3_2_1.OUT TO WriteNonWrittableTest.check;
        WriteNonWrittable.QO TO F_NOT_3_2_1.IN;
        F_NOT_3_2.OUT TO WriteMethodTest.check;
        WriteMethod.QO TO F_NOT_3_2.IN;
      END_CONNECTIONS
    END_SUBAPPLICATION
    EVENT_CONNECTIONS
      SUBSCRIBE_0_1.IND TO E_SR.R;
      SUBSCRIBE_0_1.INITO TO E_SR.S;
      InitFinishedSignal.IND TO PUBLISH_0.REQ;
      HandleInit.Execute TO E_DELAY.START;
      InitFinishedSignal.INITO TO PUBLISH_0.INIT;
      PUBLISH_0.CNF TO E_SR_2.S;
      E_SR.EO TO E_SWITCH.EI;
      E_SWITCH.EO0 TO HandleInitLocal.InitFinished;
      E_SWITCH_1.EO0 TO HandleInit.InitFinished;
      WrongNoOfArguments.CNF TO UnknownNode.REQ;
      WrongNoOfArguments.INITO TO UnknownNode.INIT;
      E_DELAY.EO TO WrongNoOfArguments.REQ;
      Writable1.CNF TO WorngInputsType.REQ;
      UnknownNode.CNF TO WrongType.REQ;
      WrongType.INITO TO HandleInit.InitFinished;
      WrongType.CNF TO E_SR_2.R;
      UnknownNode.INITO TO WrongType.INIT;
      E_SWITCH.EO1 TO SERVER_0.INIT;
      GoodInputs.CNF TO SERVER_0.RSP;
      SERVER_0.INITO TO SERVER_0_1.INIT;
      WorngInputs.CNF TO SERVER_0_1.RSP;
      SERVER_0_1.IND TO WorngInputs.REQ;
      SERVER_0_1.INITO TO SERVER_0_1_1.INIT;
      WorngInputsOutputs.CNF TO SERVER_0_1_1.RSP;
      SERVER_0_1_1.IND TO WorngInputsOutputs.REQ;
      ReadExistingWritable.CNF TO SUBSCRIBE_1_1_1.INIT;
      SUBSCRIBE_1_1.INITO TO ReadExistingWritable.REQ;
      F_NOT.CNF TO SameNodeIdWrite.REQ;
      Writable1_1.INITO TO F_NOT.REQ;
      SUBSCRIBE_1_1_1.INITO TO F_NOT_1_1.REQ;
      F_NOT_1_1.CNF TO SameNodeSecondRead.REQ;
      SUBSCRIBE_wrongPath.INITO TO F_NOT_1_2_1.REQ;
      F_NOT_1_2_1.CNF TO WrongPath.REQ;
      SERVER_0_2.INITO TO F_NOT_1_2_1_1.REQ;
      F_NOT_1_2_1_1.CNF TO DoubleMethod.REQ;
      Writable1_1_1.INITO TO SameNameDifferentNodeIdW.REQ;
      SUBSCRIBE_150.INITO TO F_NOT_1_2_1_1_1.REQ;
      F_NOT_1_2_1_1_1.CNF TO DifferentTypesOutput.REQ;
      DoubleMethod.CNF TO SUBSCRIBE_150.INIT;
      F_NOT_1.CNF TO UnconnectedSD.REQ;
      F_NOT_1_2_1_1_1_1.CNF TO UnconnectedRD.REQ;
      SUBSCRIBE_140.INITO TO F_NOT_1_2_1_1_1_1.REQ;
      SUBSCRIBE_1.INITO TO F_NOT_2.REQ;
      F_NOT_2.CNF TO SameNodeIdRead.REQ;
      SameNodeIdWrite.CNF TO SUBSCRIBE_1.INIT;
      UnconnectedRD.CNF TO Writable1_1_2.INIT;
      Writable1_1_2.INITO TO F_NOT_1.REQ;
      Writable1.INITO TO Writable1_1.INIT;
      SameNodeSecondRead.CNF TO SERVER_0_2.INIT;
      UnconnectedSD.CNF TO SUBSCRIBE_wrongPath.INIT;
      SameNodeIdRead.CNF TO SUBSCRIBE_1_1_1_1.INIT;
      SUBSCRIBE_1_1_1_1.INITO TO Writable1_2.INIT;
      F_EQ.CNF TO ValidNode.REQ;
      SUBSCRIBE_1_1_1_1.IND TO BOOL2BOOL_3_1_1.REQ;
      BOOL2BOOL_3_1_1.CNF TO F_EQ.REQ;
      Writable1_2.INITO TO SameNameDifferentNodeIdR.REQ;
      SameNameDifferentNodeIdR.CNF TO Writable1_1_1.INIT;
      SameNameDifferentNodeIdW.CNF TO SUBSCRIBE_1_1.INIT;
      DifferentTypesOutput.CNF TO SUBSCRIBE_150_1.INIT;
      SameTypesOutput.CNF TO SUBSCRIBE_140.INIT;
      SUBSCRIBE_150_1.INITO TO SameTypesOutput.REQ;
      SUBSCRIBE_NoObject.INITO TO F_NOT_1_2_1_2.REQ;
      F_NOT_1_2_1_2.CNF TO BrowseWihtouObject.REQ;
      WrongPath.CNF TO SUBSCRIBE_NoObject.INIT;
      BrowseWihtouObject.CNF TO SUBSCRIBE_NoObject_1.INIT;
      F_NOT_1_2_1_2_1.CNF TO wrongNamespace1.REQ;
      SUBSCRIBE_NoObject_1.INITO TO F_NOT_1_2_1_2_1.REQ;
      SERVER_0_1_1.INITO TO Timeoutmethod.INIT;
      Timeoutmethod.INITO TO Writable1.INIT;
      SERVER_0.IND TO E_DELAY_1.START;
      E_DELAY_1.EO TO GoodInputs.REQ;
      WrongInputOutput.INITO TO WrongInputOutput_1.INIT;
      E_SR_2.EO TO WrongInputOutput.INIT;
      E_SWITCH_1.EO1 TO WrongNoOfArguments.INIT;
      WrongInputOutput_1.INITO TO E_SWITCH_1.EI;
      wrongNamespace1.CNF TO PUBLISH_1.INIT;
      PUBLISH_1.INITO TO SERVER_0_3.INIT;
      SERVER_0_3.INITO TO F_NOT_1_2_1_2_1_1.REQ;
      F_NOT_1_2_1_2_1_1.CNF TO ObjectsFolder.REQ;
      ObjectsFolder.CNF TO SERVER_0_4.INIT;
      SERVER_0_4.INITO TO SERVER_0_4.RSP;
      SERVER_0_4.INITO TO HandleInitLocal.InitFinished;
    END_CONNECTIONS
    DATA_CONNECTIONS
      E_SR.Q TO E_SWITCH.G;
      E_SR_2.Q TO HandleInit.QI;
      E_SR_2.Q TO E_SWITCH_1.G;
      E_SR_2.Q TO HandleInit.QI;
      BOOL2BOOL_2_1.OUT TO Writable1.SD_1;
      SERVER_0.QO TO GoodInputs.check;
      DINT2DINT_1_1.OUT TO SERVER_0.SD_1;
      SERVER_0.RD_1 TO DINT2DINT_1_1.IN;
      SERVER_0_1.RD_1 TO DINT2DINT_1.IN;
      DINT2DINT_1.OUT TO SERVER_0_1.SD_1;
      SERVER_0_1_1.RD_1 TO DINT2DINT.IN;
      DINT2DINT.OUT TO SERVER_0_1_1.SD_1;
      BOOL2BOOL_2_1_1.OUT TO Writable1_1.SD_1;
      BOOL2BOOL_2_1_1_1.OUT TO Writable1_1_1.SD_1;
      SUBSCRIBE_1_1_1.RD_1 TO BOOL2BOOL_3_1.IN;
      SUBSCRIBE_1_1.RD_1 TO BOOL2BOOL_3.IN;
      SUBSCRIBE_1_1.QO TO ReadExistingWritable.check;
      F_NOT.OUT TO SameNodeIdWrite.check;
      Writable1_1.QO TO F_NOT.IN;
      SUBSCRIBE_1_1_1.QO TO F_NOT_1_1.IN;
      F_NOT_1_1.OUT TO SameNodeSecondRead.check;
      F_NOT_1_2_1.OUT TO WrongPath.check;
      SUBSCRIBE_wrongPath.QO TO F_NOT_1_2_1.IN;
      SERVER_0_2.QO TO F_NOT_1_2_1_1.IN;
      F_NOT_1_2_1_1.OUT TO DoubleMethod.check;
      SERVER_0_2.RD_1 TO BOOL2BOOL_3_2.IN;
      BOOL2BOOL_3_2.OUT TO SERVER_0_2.SD_1;
      SUBSCRIBE_wrongPath.RD_1 TO BOOL2BOOL_3_1_1_1.IN;
      SUBSCRIBE_1_1_1_1.RD_1 TO BOOL2BOOL_3_1_1.IN;
      Writable1_1_1.QO TO SameNameDifferentNodeIdW.check;
      SUBSCRIBE_150.QO TO F_NOT_1_2_1_1_1.IN;
      F_NOT_1_2_1_1_1.OUT TO DifferentTypesOutput.check;
      SUBSCRIBE_150.RD_1 TO BOOL2BOOL_3_2_1.IN;
      F_NOT_1.OUT TO UnconnectedSD.check;
      F_NOT_1_2_1_1_1_1.OUT TO UnconnectedRD.check;
      SUBSCRIBE_140.QO TO F_NOT_1_2_1_1_1_1.IN;
      SUBSCRIBE_140.RD_1 TO BOOL2BOOL_3_2_1_1.IN;
      SUBSCRIBE_1.RD_1 TO BOOL2BOOL_2_1_1_2.IN;
      SUBSCRIBE_1.QO TO F_NOT_2.IN;
      F_NOT_2.OUT TO SameNodeIdRead.check;
      STRING2STRING_1.OUT TO Writable1_1_2.SD_1;
      Writable1_1_2.QO TO F_NOT_1.IN;
      F_EQ.OUT TO ValidNode.check;
      BOOL2BOOL_3_1_1.OUT TO F_EQ.IN1;
      Writable1_2.QO TO SameNameDifferentNodeIdR.check;
      Writable1_2.RD_1 TO BOOL2BOOL_3_3.IN;
      SUBSCRIBE_150.RD_1 TO STRING2STRING.IN;
      E_SR.Q TO HandleInitLocal.QI;
      SUBSCRIBE_150_1.RD_1 TO BOOL2BOOL_3_2_1_2.IN;
      SUBSCRIBE_150_1.QO TO SameTypesOutput.check;
      SUBSCRIBE_NoObject.RD_1 TO BOOL2BOOL_3_1_1_1_1.IN;
      F_NOT_1_2_1_2.OUT TO BrowseWihtouObject.check;
      SUBSCRIBE_NoObject.QO TO F_NOT_1_2_1_2.IN;
      F_NOT_1_2_1_2_1.OUT TO wrongNamespace1.check;
      SUBSCRIBE_NoObject_1.RD_1 TO BOOL2BOOL_3_1_1_1_1_1.IN;
      SUBSCRIBE_NoObject_1.QO TO F_NOT_1_2_1_2_1.IN;
      SUBSCRIBE_150_1.RD_1 TO STRING2STRING_2.IN;
      E_SR_2.Q TO WrongInputOutput.QI;
      E_SR_2.Q TO WrongInputOutput_1.QI;
      DINT2DINT_1_2.OUT TO PUBLISH_1.SD_1;
      F_NOT_1_2_1_2_1_1.OUT TO ObjectsFolder.check;
      SERVER_0_3.QO TO F_NOT_1_2_1_2_1_1.IN;
    END_CONNECTIONS
  END_APPLICATION
  APPLICATION OpcUADelayedWorking
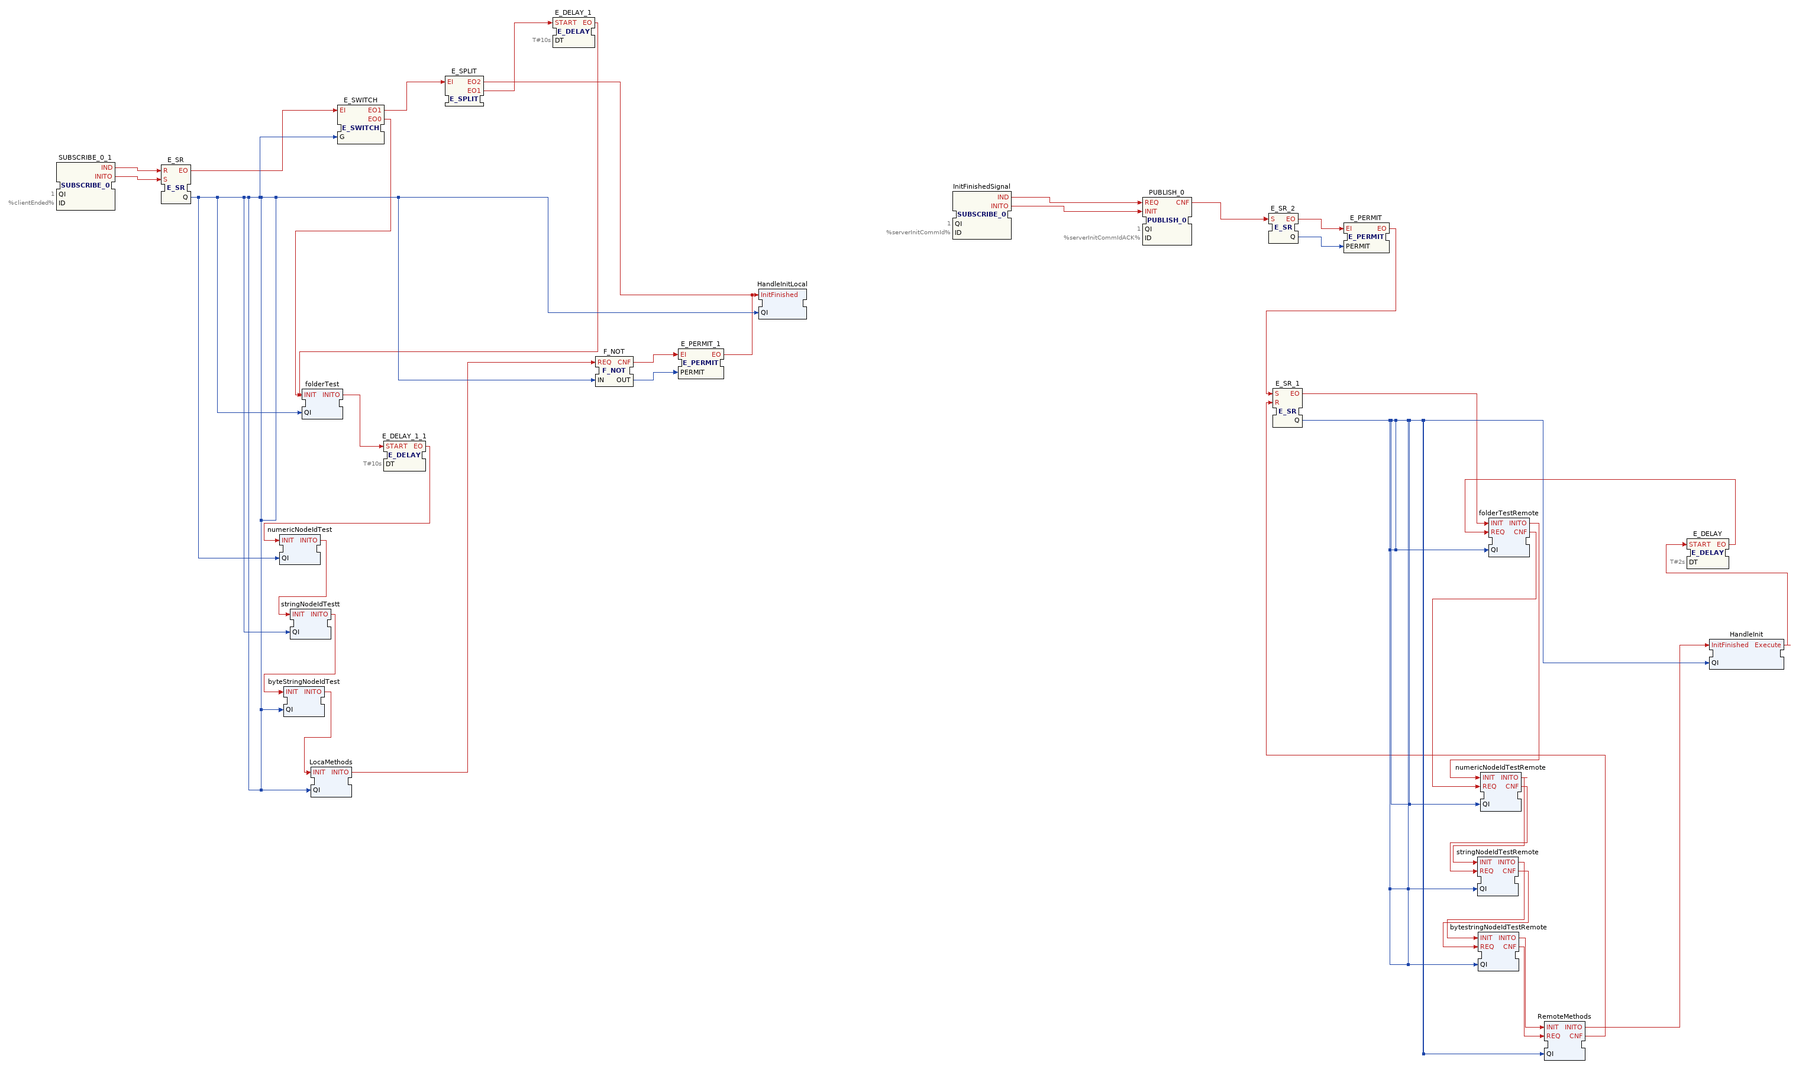
    FBS
      E_SR : E_SR;
      E_DELAY : E_DELAY(DT := T#2s);
      SUBSCRIBE_0_1 : SUBSCRIBE_0(QI := 1, ID := %clientEnded%);
      E_SR_2 : E_SR;
      PUBLISH_0 : PUBLISH_0(QI := 1, ID := %serverInitCommIdACK%);
      InitFinishedSignal : SUBSCRIBE_0(QI := 1, ID := %serverInitCommId%);
      E_PERMIT : E_PERMIT;
      E_SR_1 : E_SR;
      E_SWITCH : E_SWITCH;
      E_SPLIT : E_SPLIT;
      E_DELAY_1 : E_DELAY(DT := T#10s);
      E_DELAY_1_1 : E_DELAY(DT := T#10s);
      E_PERMIT_1 : E_PERMIT;
      F_NOT : F_NOT;
    END_FBS
    SUBAPPLICATION stringNodeIdTestRemote
      EVENT_INPUT
        INIT;
        REQ;
      END_EVENT
      EVENT_OUTPUT
        INITO;
        CNF;
      END_EVENT
      VAR_INPUT
        QI : BOOL;
      END_VAR
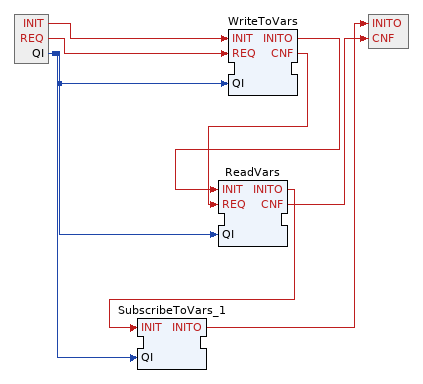
      SUBAPPLICATION WriteToVars
        EVENT_INPUT
          INIT;
          REQ;
        END_EVENT
        EVENT_OUTPUT
          INITO;
          CNF;
        END_EVENT
        VAR_INPUT
          QI : BOOL;
        END_VAR
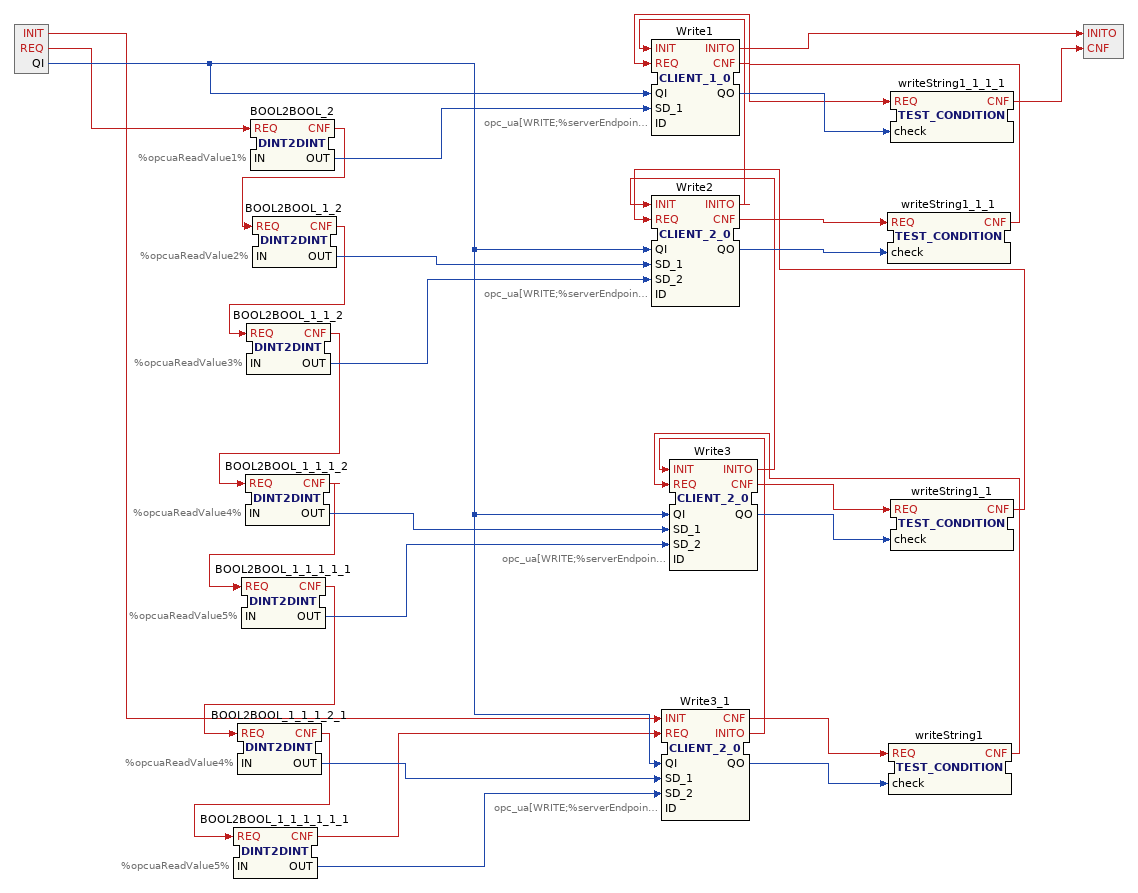
        FBS
          BOOL2BOOL_1_1_2 : DINT2DINT(IN := %opcuaReadValue3%);
          BOOL2BOOL_1_1_1_1_1 : DINT2DINT(IN := %opcuaReadValue5%);
          BOOL2BOOL_1_1_1_2 : DINT2DINT(IN := %opcuaReadValue4%);
          BOOL2BOOL_2 : DINT2DINT(IN := %opcuaReadValue1%);
          BOOL2BOOL_1_2 : DINT2DINT(IN := %opcuaReadValue2%);
          BOOL2BOOL_1_1_1_2_1 : DINT2DINT(IN := %opcuaReadValue4%);
          BOOL2BOOL_1_1_1_1_1_1 : DINT2DINT(IN := %opcuaReadValue5%);
          writeString1 : TEST_CONDITION;
          writeString1_1 : TEST_CONDITION;
          writeString1_1_1 : TEST_CONDITION;
          writeString1_1_1_1 : TEST_CONDITION;
          Write1 : CLIENT_1_0(ID := opc_ua[WRITE;%serverEndpoint%;%opcuaFolderTestWithNodeIdString1%]);
          Write2 : CLIENT_2_0(ID := opc_ua[WRITE;%serverEndpoint%;%opcuaFolderTestWithNodeIdString2%]);
          Write3_1 : CLIENT_2_0(ID := opc_ua[WRITE;%serverEndpoint%;,1:s=hello3;,1:s=hello4]);
          Write3 : CLIENT_2_0(ID := opc_ua[WRITE;%serverEndpoint%;%opcuaFolderTestWithNodeIdString3%]);
        END_FBS
        EVENT_CONNECTIONS
          BOOL2BOOL_1_2.CNF TO BOOL2BOOL_1_1_2.REQ;
          BOOL2BOOL_1_1_2.CNF TO BOOL2BOOL_1_1_1_2.REQ;
          BOOL2BOOL_1_1_1_2.CNF TO BOOL2BOOL_1_1_1_1_1.REQ;
          BOOL2BOOL_2.CNF TO BOOL2BOOL_1_2.REQ;
          REQ TO BOOL2BOOL_2.REQ;
          BOOL2BOOL_1_1_1_2_1.CNF TO BOOL2BOOL_1_1_1_1_1_1.REQ;
          BOOL2BOOL_1_1_1_1_1.CNF TO BOOL2BOOL_1_1_1_2_1.REQ;
          Write1.INITO TO INITO;
          Write2.INITO TO Write1.INIT;
          INIT TO Write3_1.INIT;
          BOOL2BOOL_1_1_1_1_1_1.CNF TO Write3_1.REQ;
          Write3_1.CNF TO writeString1.REQ;
          Write3_1.INITO TO Write3.INIT;
          writeString1.CNF TO Write3.REQ;
          Write3.INITO TO Write2.INIT;
          writeString1_1.CNF TO Write2.REQ;
          Write3.CNF TO writeString1_1.REQ;
          writeString1_1_1.CNF TO Write1.REQ;
          Write2.CNF TO writeString1_1_1.REQ;
          writeString1_1_1_1.CNF TO CNF;
          Write1.CNF TO writeString1_1_1_1.REQ;
        END_CONNECTIONS
        DATA_CONNECTIONS
          QI TO Write1.QI;
          BOOL2BOOL_2.OUT TO Write1.SD_1;
          QI TO Write2.QI;
          BOOL2BOOL_1_2.OUT TO Write2.SD_1;
          BOOL2BOOL_1_1_2.OUT TO Write2.SD_2;
          QI TO Write3_1.QI;
          BOOL2BOOL_1_1_1_2_1.OUT TO Write3_1.SD_1;
          BOOL2BOOL_1_1_1_1_1_1.OUT TO Write3_1.SD_2;
          Write3_1.QO TO writeString1.check;
          QI TO Write3.QI;
          BOOL2BOOL_1_1_1_2.OUT TO Write3.SD_1;
          BOOL2BOOL_1_1_1_1_1.OUT TO Write3.SD_2;
          Write3.QO TO writeString1_1.check;
          Write2.QO TO writeString1_1_1.check;
          Write1.QO TO writeString1_1_1_1.check;
        END_CONNECTIONS
      END_SUBAPPLICATION
      SUBAPPLICATION ReadVars
        EVENT_INPUT
          INIT;
          REQ;
        END_EVENT
        EVENT_OUTPUT
          INITO;
          CNF;
        END_EVENT
        VAR_INPUT
          QI : BOOL;
        END_VAR
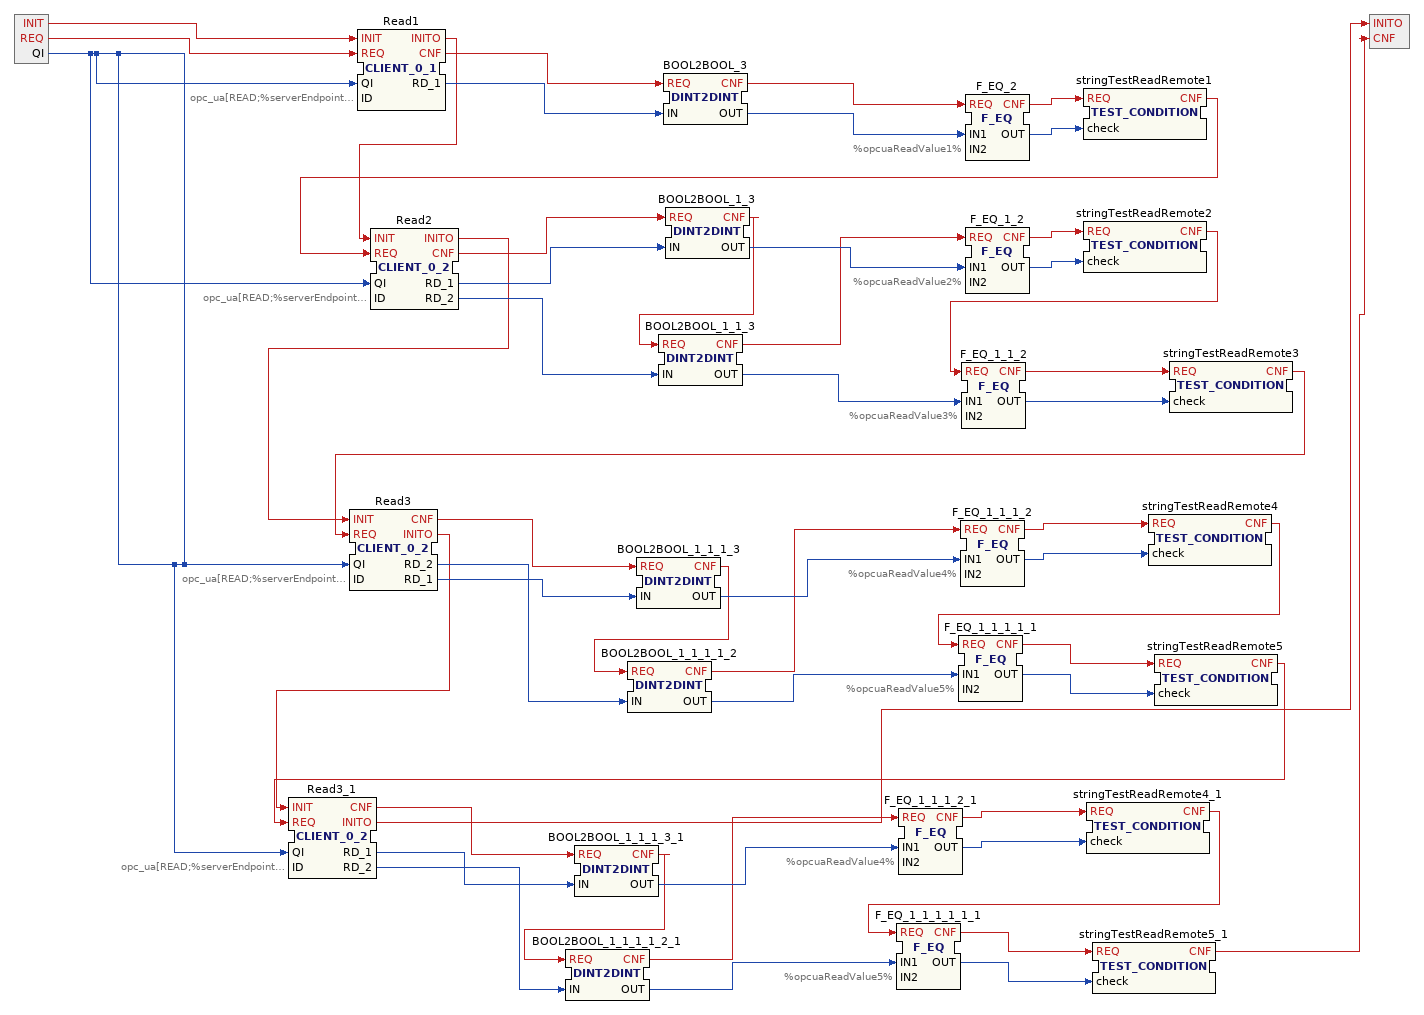
        FBS
          Read1 : CLIENT_0_1(ID := opc_ua[READ;%serverEndpoint%;%opcuaFolderTestWithNodeIdString1%]);
          Read2 : CLIENT_0_2(ID := opc_ua[READ;%serverEndpoint%;%opcuaFolderTestWithNodeIdString2%]);
          F_EQ_1_1_1_2 : F_EQ(IN2 := %opcuaReadValue4%);
          stringTestReadRemote4 : TEST_CONDITION;
          BOOL2BOOL_1_3 : DINT2DINT;
          F_EQ_1_1_1_1_1 : F_EQ(IN2 := %opcuaReadValue5%);
          stringTestReadRemote3 : TEST_CONDITION;
          BOOL2BOOL_1_1_3 : DINT2DINT;
          BOOL2BOOL_1_1_1_1_2 : DINT2DINT;
          BOOL2BOOL_1_1_1_3 : DINT2DINT;
          stringTestReadRemote2 : TEST_CONDITION;
          F_EQ_1_1_2 : F_EQ(IN2 := %opcuaReadValue3%);
          F_EQ_2 : F_EQ(IN2 := %opcuaReadValue1%);
          F_EQ_1_2 : F_EQ(IN2 := %opcuaReadValue2%);
          Read3 : CLIENT_0_2(ID := opc_ua[READ;%serverEndpoint%;%opcuaFolderTestWithNodeIdString3%]);
          stringTestReadRemote5 : TEST_CONDITION;
          stringTestReadRemote1 : TEST_CONDITION;
          BOOL2BOOL_3 : DINT2DINT;
          stringTestReadRemote5_1 : TEST_CONDITION;
          F_EQ_1_1_1_2_1 : F_EQ(IN2 := %opcuaReadValue4%);
          Read3_1 : CLIENT_0_2(ID := opc_ua[READ;%serverEndpoint%;,1:s=hello3;,1:s=hello4]);
          F_EQ_1_1_1_1_1_1 : F_EQ(IN2 := %opcuaReadValue5%);
          BOOL2BOOL_1_1_1_1_2_1 : DINT2DINT;
          BOOL2BOOL_1_1_1_3_1 : DINT2DINT;
          stringTestReadRemote4_1 : TEST_CONDITION;
        END_FBS
        EVENT_CONNECTIONS
          Read1.INITO TO Read2.INIT;
          Read1.CNF TO BOOL2BOOL_3.REQ;
          stringTestReadRemote1.CNF TO Read2.REQ;
          Read2.INITO TO Read3.INIT;
          Read2.CNF TO BOOL2BOOL_1_3.REQ;
          BOOL2BOOL_1_1_1_1_2.CNF TO F_EQ_1_1_1_2.REQ;
          F_EQ_1_1_1_2.CNF TO stringTestReadRemote4.REQ;
          stringTestReadRemote4.CNF TO F_EQ_1_1_1_1_1.REQ;
          BOOL2BOOL_1_3.CNF TO BOOL2BOOL_1_1_3.REQ;
          F_EQ_1_1_1_1_1.CNF TO stringTestReadRemote5.REQ;
          F_EQ_1_1_2.CNF TO stringTestReadRemote3.REQ;
          stringTestReadRemote3.CNF TO Read3.REQ;
          BOOL2BOOL_1_1_3.CNF TO F_EQ_1_2.REQ;
          BOOL2BOOL_1_1_1_3.CNF TO BOOL2BOOL_1_1_1_1_2.REQ;
          Read3.CNF TO BOOL2BOOL_1_1_1_3.REQ;
          F_EQ_1_2.CNF TO stringTestReadRemote2.REQ;
          stringTestReadRemote2.CNF TO F_EQ_1_1_2.REQ;
          BOOL2BOOL_3.CNF TO F_EQ_2.REQ;
          F_EQ_2.CNF TO stringTestReadRemote1.REQ;
          INIT TO Read1.INIT;
          REQ TO Read1.REQ;
          BOOL2BOOL_1_1_1_1_2_1.CNF TO F_EQ_1_1_1_2_1.REQ;
          BOOL2BOOL_1_1_1_3_1.CNF TO BOOL2BOOL_1_1_1_1_2_1.REQ;
          F_EQ_1_1_1_2_1.CNF TO stringTestReadRemote4_1.REQ;
          Read3_1.CNF TO BOOL2BOOL_1_1_1_3_1.REQ;
          F_EQ_1_1_1_1_1_1.CNF TO stringTestReadRemote5_1.REQ;
          stringTestReadRemote4_1.CNF TO F_EQ_1_1_1_1_1_1.REQ;
          Read3_1.INITO TO INITO;
          Read3.INITO TO Read3_1.INIT;
          stringTestReadRemote5_1.CNF TO CNF;
          stringTestReadRemote5.CNF TO Read3_1.REQ;
        END_CONNECTIONS
        DATA_CONNECTIONS
          Read1.RD_1 TO BOOL2BOOL_3.IN;
          Read2.RD_1 TO BOOL2BOOL_1_3.IN;
          Read2.RD_2 TO BOOL2BOOL_1_1_3.IN;
          BOOL2BOOL_1_1_1_3.OUT TO F_EQ_1_1_1_2.IN1;
          F_EQ_1_1_1_2.OUT TO stringTestReadRemote4.check;
          BOOL2BOOL_1_3.OUT TO F_EQ_1_2.IN1;
          BOOL2BOOL_1_1_1_1_2.OUT TO F_EQ_1_1_1_1_1.IN1;
          F_EQ_1_1_1_1_1.OUT TO stringTestReadRemote5.check;
          F_EQ_1_1_2.OUT TO stringTestReadRemote3.check;
          BOOL2BOOL_1_1_3.OUT TO F_EQ_1_1_2.IN1;
          Read3.RD_2 TO BOOL2BOOL_1_1_1_1_2.IN;
          Read3.RD_1 TO BOOL2BOOL_1_1_1_3.IN;
          F_EQ_1_2.OUT TO stringTestReadRemote2.check;
          BOOL2BOOL_3.OUT TO F_EQ_2.IN1;
          F_EQ_2.OUT TO stringTestReadRemote1.check;
          QI TO Read1.QI;
          QI TO Read2.QI;
          QI TO Read3.QI;
          Read3_1.RD_1 TO BOOL2BOOL_1_1_1_3_1.IN;
          Read3_1.RD_2 TO BOOL2BOOL_1_1_1_1_2_1.IN;
          F_EQ_1_1_1_2_1.OUT TO stringTestReadRemote4_1.check;
          F_EQ_1_1_1_1_1_1.OUT TO stringTestReadRemote5_1.check;
          BOOL2BOOL_1_1_1_3_1.OUT TO F_EQ_1_1_1_2_1.IN1;
          BOOL2BOOL_1_1_1_1_2_1.OUT TO F_EQ_1_1_1_1_1_1.IN1;
          QI TO Read3_1.QI;
        END_CONNECTIONS
      END_SUBAPPLICATION
      SUBAPPLICATION SubscribeToVars_1
        EVENT_INPUT
          INIT;
        END_EVENT
        EVENT_OUTPUT
          INITO;
        END_EVENT
        VAR_INPUT
          QI : BOOL;
        END_VAR
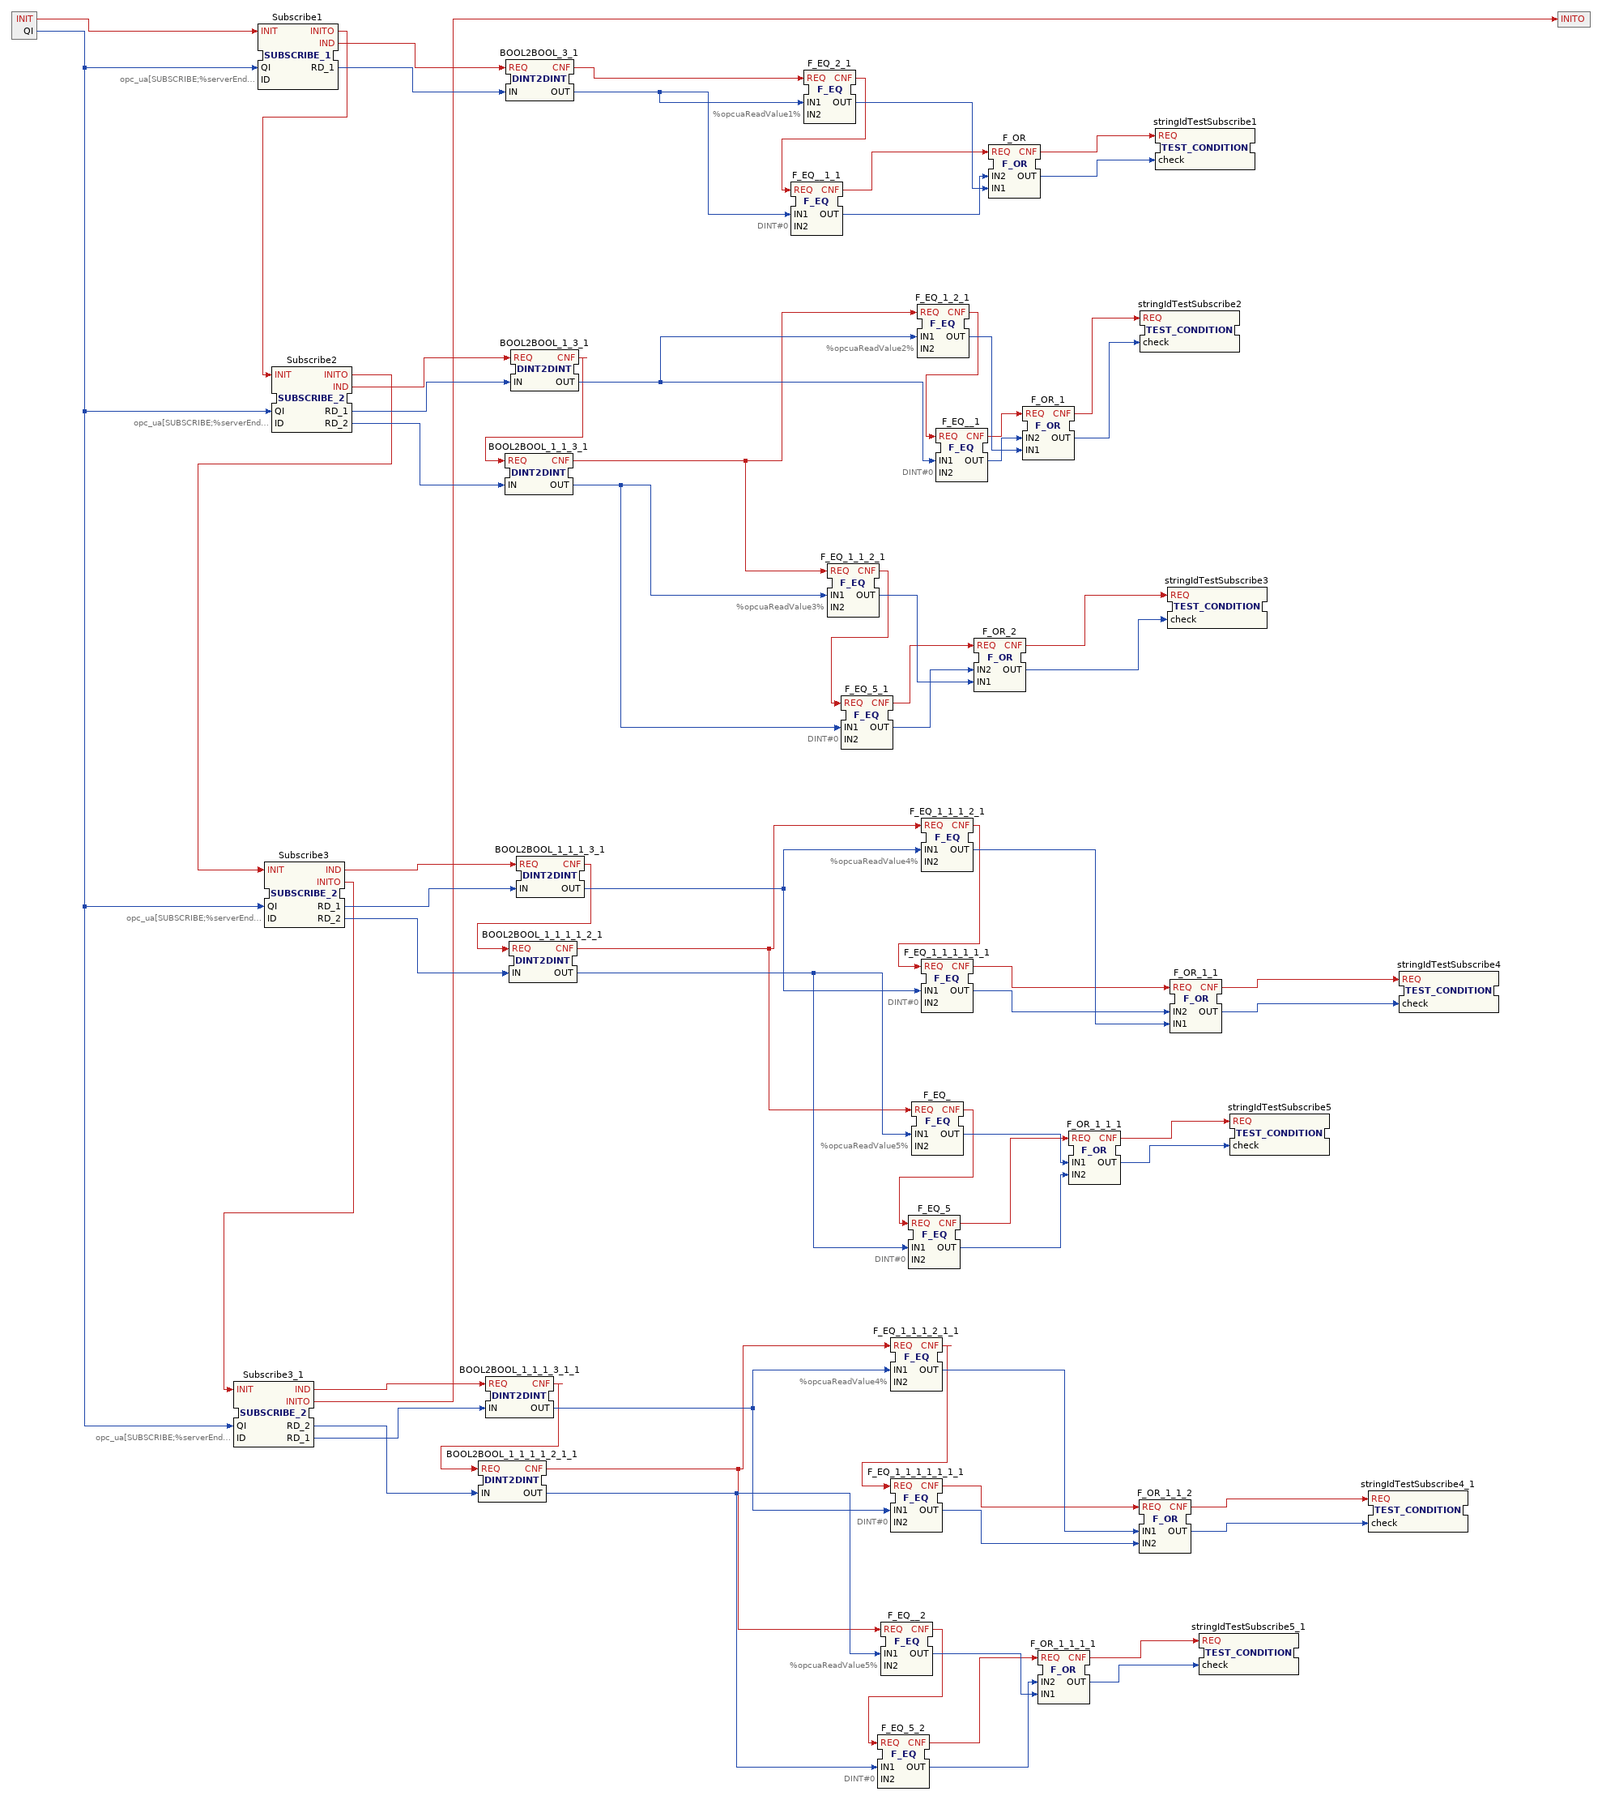
        FBS
          F_EQ_2_1 : F_EQ(IN2 := %opcuaReadValue1%);
          stringIdTestSubscribe4 : TEST_CONDITION;
          Subscribe3 : SUBSCRIBE_2(ID := opc_ua[SUBSCRIBE;%serverEndpoint%;%opcuaFolderTestWithNodeIdString3%]);
          F_EQ_1_1_1_2_1 : F_EQ(IN2 := %opcuaReadValue4%);
          stringIdTestSubscribe3 : TEST_CONDITION;
          F_EQ_1_1_1_1_1_1 : F_EQ(IN2 := DINT#0);
          F_EQ_1_1_2_1 : F_EQ(IN2 := %opcuaReadValue3%);
          stringIdTestSubscribe1 : TEST_CONDITION;
          stringIdTestSubscribe2 : TEST_CONDITION;
          Subscribe1 : SUBSCRIBE_1(ID := opc_ua[SUBSCRIBE;%serverEndpoint%;%opcuaFolderTestWithNodeIdString1%]);
          Subscribe2 : SUBSCRIBE_2(ID := opc_ua[SUBSCRIBE;%serverEndpoint%;%opcuaFolderTestWithNodeIdString2%]);
          BOOL2BOOL_1_1_3_1 : DINT2DINT;
          F_EQ_1_2_1 : F_EQ(IN2 := %opcuaReadValue2%);
          BOOL2BOOL_3_1 : DINT2DINT;
          BOOL2BOOL_1_1_1_3_1 : DINT2DINT;
          BOOL2BOOL_1_1_1_1_2_1 : DINT2DINT;
          BOOL2BOOL_1_3_1 : DINT2DINT;
          F_EQ_ : F_EQ(IN2 := %opcuaReadValue5%);
          stringIdTestSubscribe5 : TEST_CONDITION;
          F_EQ_5 : F_EQ(IN2 := DINT#0);
          F_EQ_5_1 : F_EQ(IN2 := DINT#0);
          F_EQ__1 : F_EQ(IN2 := DINT#0);
          F_EQ__1_1 : F_EQ(IN2 := DINT#0);
          F_OR : F_OR;
          F_OR_1 : F_OR;
          F_OR_2 : F_OR;
          F_OR_1_1 : F_OR;
          F_OR_1_1_1 : F_OR;
          BOOL2BOOL_1_1_1_1_2_1_1 : DINT2DINT;
          F_OR_1_1_2 : F_OR;
          BOOL2BOOL_1_1_1_3_1_1 : DINT2DINT;
          F_EQ__2 : F_EQ(IN2 := %opcuaReadValue5%);
          stringIdTestSubscribe5_1 : TEST_CONDITION;
          stringIdTestSubscribe4_1 : TEST_CONDITION;
          F_OR_1_1_1_1 : F_OR;
          Subscribe3_1 : SUBSCRIBE_2(ID := opc_ua[SUBSCRIBE;%serverEndpoint%;,1:s=hello3;,1:s=hello4]);
          F_EQ_1_1_1_1_1_1_1 : F_EQ(IN2 := DINT#0);
          F_EQ_5_2 : F_EQ(IN2 := DINT#0);
          F_EQ_1_1_1_2_1_1 : F_EQ(IN2 := %opcuaReadValue4%);
        END_FBS
        EVENT_CONNECTIONS
          Subscribe2.INITO TO Subscribe3.INIT;
          Subscribe3.IND TO BOOL2BOOL_1_1_1_3_1.REQ;
          Subscribe1.INITO TO Subscribe2.INIT;
          Subscribe1.IND TO BOOL2BOOL_3_1.REQ;
          Subscribe2.IND TO BOOL2BOOL_1_3_1.REQ;
          BOOL2BOOL_1_3_1.CNF TO BOOL2BOOL_1_1_3_1.REQ;
          BOOL2BOOL_1_1_1_3_1.CNF TO BOOL2BOOL_1_1_1_1_2_1.REQ;
          INIT TO Subscribe1.INIT;
          F_EQ__1_1.CNF TO F_OR.REQ;
          BOOL2BOOL_3_1.CNF TO F_EQ_2_1.REQ;
          F_EQ_2_1.CNF TO F_EQ__1_1.REQ;
          F_OR.CNF TO stringIdTestSubscribe1.REQ;
          F_OR_2.CNF TO stringIdTestSubscribe3.REQ;
          F_OR_1.CNF TO stringIdTestSubscribe2.REQ;
          F_EQ__1.CNF TO F_OR_1.REQ;
          F_EQ_1_2_1.CNF TO F_EQ__1.REQ;
          BOOL2BOOL_1_1_3_1.CNF TO F_EQ_1_2_1.REQ;
          BOOL2BOOL_1_1_3_1.CNF TO F_EQ_1_1_2_1.REQ;
          F_EQ_1_1_2_1.CNF TO F_EQ_5_1.REQ;
          F_EQ_5_1.CNF TO F_OR_2.REQ;
          F_OR_1_1.CNF TO stringIdTestSubscribe4.REQ;
          F_EQ_1_1_1_1_1_1.CNF TO F_OR_1_1.REQ;
          F_EQ_1_1_1_2_1.CNF TO F_EQ_1_1_1_1_1_1.REQ;
          BOOL2BOOL_1_1_1_1_2_1.CNF TO F_EQ_1_1_1_2_1.REQ;
          F_OR_1_1_1.CNF TO stringIdTestSubscribe5.REQ;
          BOOL2BOOL_1_1_1_1_2_1.CNF TO F_EQ_.REQ;
          F_EQ_.CNF TO F_EQ_5.REQ;
          F_EQ_5.CNF TO F_OR_1_1_1.REQ;
          F_EQ_1_1_1_2_1_1.CNF TO F_EQ_1_1_1_1_1_1_1.REQ;
          Subscribe3_1.IND TO BOOL2BOOL_1_1_1_3_1_1.REQ;
          BOOL2BOOL_1_1_1_1_2_1_1.CNF TO F_EQ__2.REQ;
          F_OR_1_1_1_1.CNF TO stringIdTestSubscribe5_1.REQ;
          BOOL2BOOL_1_1_1_1_2_1_1.CNF TO F_EQ_1_1_1_2_1_1.REQ;
          BOOL2BOOL_1_1_1_3_1_1.CNF TO BOOL2BOOL_1_1_1_1_2_1_1.REQ;
          F_EQ_1_1_1_1_1_1_1.CNF TO F_OR_1_1_2.REQ;
          F_EQ__2.CNF TO F_EQ_5_2.REQ;
          F_OR_1_1_2.CNF TO stringIdTestSubscribe4_1.REQ;
          F_EQ_5_2.CNF TO F_OR_1_1_1_1.REQ;
          Subscribe3_1.INITO TO INITO;
          Subscribe3.INITO TO Subscribe3_1.INIT;
        END_CONNECTIONS
        DATA_CONNECTIONS
          BOOL2BOOL_3_1.OUT TO F_EQ_2_1.IN1;
          Subscribe3.RD_1 TO BOOL2BOOL_1_1_1_3_1.IN;
          Subscribe3.RD_2 TO BOOL2BOOL_1_1_1_1_2_1.IN;
          BOOL2BOOL_1_1_3_1.OUT TO F_EQ_1_1_2_1.IN1;
          Subscribe1.RD_1 TO BOOL2BOOL_3_1.IN;
          Subscribe2.RD_1 TO BOOL2BOOL_1_3_1.IN;
          Subscribe2.RD_2 TO BOOL2BOOL_1_1_3_1.IN;
          BOOL2BOOL_1_3_1.OUT TO F_EQ_1_2_1.IN1;
          QI TO Subscribe3.QI;
          QI TO Subscribe1.QI;
          QI TO Subscribe2.QI;
          BOOL2BOOL_1_1_1_1_2_1.OUT TO F_EQ_5.IN1;
          BOOL2BOOL_1_3_1.OUT TO F_EQ__1.IN1;
          BOOL2BOOL_1_1_3_1.OUT TO F_EQ_5_1.IN1;
          BOOL2BOOL_3_1.OUT TO F_EQ__1_1.IN1;
          BOOL2BOOL_1_1_1_3_1.OUT TO F_EQ_1_1_1_2_1.IN1;
          F_EQ__1_1.OUT TO F_OR.IN2;
          F_EQ_2_1.OUT TO F_OR.IN1;
          F_OR.OUT TO stringIdTestSubscribe1.check;
          F_EQ_5_1.OUT TO F_OR_2.IN2;
          F_EQ__1.OUT TO F_OR_1.IN2;
          F_EQ_1_2_1.OUT TO F_OR_1.IN1;
          F_OR_1.OUT TO stringIdTestSubscribe2.check;
          F_OR_2.OUT TO stringIdTestSubscribe3.check;
          F_OR_1_1.OUT TO stringIdTestSubscribe4.check;
          F_EQ_1_1_1_1_1_1.OUT TO F_OR_1_1.IN2;
          F_EQ_1_1_1_2_1.OUT TO F_OR_1_1.IN1;
          F_OR_1_1_1.OUT TO stringIdTestSubscribe5.check;
          F_EQ_.OUT TO F_OR_1_1_1.IN1;
          F_EQ_5.OUT TO F_OR_1_1_1.IN2;
          BOOL2BOOL_1_1_1_1_2_1.OUT TO F_EQ_.IN1;
          F_EQ_1_1_2_1.OUT TO F_OR_2.IN1;
          BOOL2BOOL_1_1_1_3_1.OUT TO F_EQ_1_1_1_1_1_1.IN1;
          BOOL2BOOL_1_1_1_3_1_1.OUT TO F_EQ_1_1_1_1_1_1_1.IN1;
          F_EQ_5_2.OUT TO F_OR_1_1_1_1.IN2;
          F_EQ_1_1_1_2_1_1.OUT TO F_OR_1_1_2.IN1;
          F_EQ__2.OUT TO F_OR_1_1_1_1.IN1;
          F_OR_1_1_1_1.OUT TO stringIdTestSubscribe5_1.check;
          Subscribe3_1.RD_2 TO BOOL2BOOL_1_1_1_1_2_1_1.IN;
          BOOL2BOOL_1_1_1_1_2_1_1.OUT TO F_EQ__2.IN1;
          Subscribe3_1.RD_1 TO BOOL2BOOL_1_1_1_3_1_1.IN;
          BOOL2BOOL_1_1_1_3_1_1.OUT TO F_EQ_1_1_1_2_1_1.IN1;
          F_OR_1_1_2.OUT TO stringIdTestSubscribe4_1.check;
          F_EQ_1_1_1_1_1_1_1.OUT TO F_OR_1_1_2.IN2;
          BOOL2BOOL_1_1_1_1_2_1_1.OUT TO F_EQ_5_2.IN1;
          QI TO Subscribe3_1.QI;
        END_CONNECTIONS
      END_SUBAPPLICATION
      EVENT_CONNECTIONS
        WriteToVars.INITO TO ReadVars.INIT;
        INIT TO WriteToVars.INIT;
        REQ TO WriteToVars.REQ;
        SubscribeToVars_1.INITO TO INITO;
        ReadVars.INITO TO SubscribeToVars_1.INIT;
        WriteToVars.CNF TO ReadVars.REQ;
        ReadVars.CNF TO CNF;
      END_CONNECTIONS
      DATA_CONNECTIONS
        QI TO ReadVars.QI;
        QI TO WriteToVars.QI;
        QI TO SubscribeToVars_1.QI;
      END_CONNECTIONS
    END_SUBAPPLICATION
    SUBAPPLICATION RemoteMethods
      EVENT_INPUT
        INIT;
        REQ;
      END_EVENT
      EVENT_OUTPUT
        INITO;
        CNF;
      END_EVENT
      VAR_INPUT
        QI : BOOL;
      END_VAR
